// TIA Portal V20 export
// export: Created 2025-12-01T14:56:44.9442204Z, ExportSetting None, DisplayName Totally Integrated Automation Portal, DisplayVersion V20 Update 3, DisplayName TIA Portal Openness, DisplayVersion V20 Update 3, DisplayName TIA Portal Version Control Interface, DisplayVersion V20 Update 3, DisplayName STEP 7 Professional, DisplayVersion V20 Update 3, DisplayName STEP 7 Safety, DisplayVersion V20 Update 2, DisplayName WinCC Basic/Comfort/Advanced, DisplayVersion V20 Update 3, DisplayName WinCC Professional, DisplayVersion V20 Update 3, DisplayName WinCC Unified, DisplayVersion V20 Update 3
FUNCTION_BLOCK "FB261_M_FSS_Carga_V0"   // FB261, LAD
TITLE = FSS_Carga
{ S7_Optimized_Access := 'FALSE' }
AUTHOR : TE_FSS
FAMILY : FSS
NAME : 20160509
VERSION : 3.3
// stored: AutoNumber false, SetENOAutomatically false
   VAR_INPUT
      Mesa : UInt;   // Mesa de la FB
      Error_Tx : Bool;   // Error en el Tx
      EnTension : Bool;   // Existe Tension en la Mesa
      Termico_T1 : Bool;   // Proteccion del T1
      Termico_T2 : Bool;   // Proteccion del T2
      Termico_T3 : Bool;   // Proteccion del T3
      Termico_T4 : Bool;   // Proteccion del T4
      pHsMx_1 : Bool;   // pHs 1 de la Mesa
      pHsMx_2 : Bool;   // pHs 2 de la Mesa
      pHsMx_3 : Bool;   // pHs 3 de la Mesa
      pHsMx_4 : Bool;   // pHs 4 de la Mesa
      Avance_T1 : Bool;   // Avance del T1
      Avance_T2 : Bool;   // Avance del T2
      Avance_T3 : Bool;   // Avance del T3
      Avance_T4 : Bool;   // Avance del T4
      Termico_TR1 : Bool;   // Proteccion del TR1
      Termico_TR2 : Bool;   // Proteccion del TR1
      Avance_TR1 : Bool;   // Avance del TR1
      Avance_TR2 : Bool;   // Avance del TR2
      TR1_Arriba : Bool;   // TR1 >> Arriba
      TR1_Abajo : Bool;   // TR1 >> Abajo
      TR1_EnMovimiento : Bool;   // TR1 >> En Movimiento
      TR2_Arriba : Bool;   // TR2 >> Arriba
      TR2_Abajo : Bool;   // TR2 >> Abajo
      TR2_EnMovimiento : Bool;   // TR2 >> En Movimiento
      TP1_Arriba : Bool;   // TP1 >> Arriba
      TP1_Abajo : Bool;   // TP1 >> Abajo
      TP1_EnMovimiento : Bool;   // TP1 >> En Movimiento
      TP2_Arriba : Bool;   // TP2 >> Arriba
      TP2_Abajo : Bool;   // TP2 >> Abajo
      TP2_EnMovimiento : Bool;   // TP2 >> En Movimiento
      TPS1_Arriba : Bool;   // TPS1 >> Arriba
      TPS1_Abajo : Bool;   // TPS1 >> Abajo
      TPS1_EnMovimiento : Bool;   // TPS1 >> En Movimiento
      TPS3_Arriba : Bool;   // TPS2 >> Arriba
      TPS3_Abajo : Bool;   // TPS2 >> Abajo
      TPS3_EnMovimiento : Bool;   // TPS2 >> En Movimiento
      MAnt_DescargaAct : Bool;   // E2 >> Mesa Anterior DescargaAct
      AVTF_MAnt_Mx_BGrande : Bool;   // E2 >> Mesa Anterior AVTF - Grande
      AVTF_MAnt_Mx_BPequena : Bool;   // E2 >> Mesa Anterior AVTF - Pequeña
      P_Mens_MAnt_Mx : Bool;   // E2 >> Mesa Anterior P_Mens
      S1_Arrival : Bool;   // S1 a FSS >> Arrival
      S1_Rotative : Bool;   // S1 a FSS >> Rotative
      S1_Complete : Bool;   // S1 a FSS >> Complete
      S3_Arrival : Bool;   // S3 a FSS >> Arrival
      S3_Rotative : Bool;   // S3 a FSS >> Rotative
      S3_Complete : Bool;   // S3 a FSS >> Complete
      MAnt_MSig_DesCargaAct : Bool;   // Pasarela >> Descarga Act
      AVTF_MAnt_MSig_BGrande : Bool;   // Pasarela >> AVTF - Grande
      AVTF_MAnt_MSig_BPequena : Bool;   // Pasarela >> AVTF - Pequeña
      PTF_MAnt_MSig : Bool;   // Pasarela >> PTF
      FTF_MAnt_MSig : Bool;   // Pasarela >> FTF
      F_EnvMens_Mx : Bool;   // Fin de Envio de Mensaje
      OrdSal_S01 : Bool;   // Orden de Salida por S1
      OrdSal_S03 : Bool;   // Orden de Salida por S3
      V_CNT_pHsMx : Int := 1000;   // Valor de Presencia
      V_CNT_pHsMx_FTF : Int := 250;   // Valor para activar FTF. Nota: < = V_CNT_pHsMx.
      V_CNTSeg_pHsMx : Int := 2000;   // Valor de Seguriadad para Presencia
      V_CNT_ApHsMx : Int := 200;   // Valor de Ausencia
      V_CNTSeg_ApHsMx : Int := 2000;   // Valor de Seguriadad para Ausencia
      V_TOut_Tx_Mx : Int := 7000;   // TimeOut de Entrada por E2
      V_TOut_TR : Int := 3000;   // TimeOut de Transfer
      V_TOut_TP : Int := 3000;   // TimeOut de Tope
      V_TOut_Interlock : Int := 5000;   // TimeOut de Interlock con el FSS
      V_CNT_PerdidapHs : Int := 1000;   // CNT de Perdida de pHs
      V_CNT_PosicionarCarga : Int := 500;   // Valor de Posicionar la Carga despues de la Entrada
      V_CNT_PresenciaPasarela : Int := 500;   // Valor de Posiconado para Pasarela
      V_TIM_EstabilidadCarga : Time := T#100MS;   // Valor de Eastabilidad de Carga por DCC
   END_VAR
   VAR_OUTPUT
      P_EnvMens_PMx : Bool;   // Permiso de Enviar Mensaje de Presencia
      P_EnvMens_AMx : Bool;   // Permiso de Enviar Mensaje de Ausencia
      P_RecepOK_Mx : Bool;   // Recepcion OK
      PTF_MAnt_Mx : Bool;   // E2 >> Mesa Anterior PTF
      FTF_MAnt_Mx : Bool;   // E2 >> Mesa Anterior FTF
      PMAnt_MSig_DescagaAct : Bool;   // Pasarela >> Descarga Act
      PAVTF_MAnt_MSig_BPequena : Bool;   // Pasarela >> AVTF - Grande
      PAVTF_MAnt_MSig_BGrande : Bool;   // Pasarela >> AVTF - Pequeña
      PPTF_MAnt_MSig : Bool;   // Pasarela >> PTF
      PFTF_MAnt_MSig : Bool;   // Pasarela >> FTF
   END_VAR
   VAR
      Mx_ET00 : Bool;
      Mx_ET01 : Bool;
      Mx_ET02 : Bool;
      Mx_ET07_1PRE : Bool;
      Mx_ET07_1FIN : Bool;
      Mx_ET07_2PRE : Bool;
      Mx_ET07_2FIN : Bool;
      Mx_ET07_3PRE : Bool;
      Mx_ET07_3FIN : Bool;
      Mx_ET07_4PRE : Bool;
      Mx_ET07_4FIN : Bool;
      Mx_ET08 : Bool;
      Mx_ET09 : Bool;
      Mx_ET10 : Bool;
      Mx_ET11 : Bool;
      Mx_ET12 : Bool;
      Mx_ET110 : Bool;
      Mx_ET111 : Bool;
      Mx_ET13 : Bool;
      Mx_ET14 : Bool;
      Mx_ET15 : Bool;
      Mx_ET40 : Bool;
      Mx_ET41 : Bool;
      Mx_ET42 : Bool;
      Mx_ET50 : Bool;
      Mx_ET51 : Bool;
      Mx_ET150 : Bool;
      Mx_ET151 : Bool;
      Mx_ET152 : Bool;
      Mx_ET250 : Bool;
      Mx_ET251 : Bool;
      Mx_ET60 : Bool;
      Mx_ET61 : Bool;
      Mx_ET160 : Bool;
      Mx_ET161 : Bool;
      Mx_ET162 : Bool;
      Mx_ET260 : Bool;
      Mx_ET261 : Bool;
      Mx_ET90 : Bool;
      Mx_ET91 : Bool;
      Mx_ET92 : Bool;
      Mx_AutoArranque : Bool;   // Config >> Fin carga del FSS - Automatico
      FinCargaFSS_Auto : Bool;   // Intena >> AutoRearme Fin Carga del FSS
      Entrando_BGrande : Bool;   // Interna >> Bandeja Grande en Entrada
      Activado_Pasarela : Bool;   // Pasarela >> Activada
      Permiso_Pasarela : Bool;   // Pasarela >> Permiso de Movimiento
      S1_DesCargaAct : Bool;   // Interna >> DesCarga Activa de Salida por S1
      S3_DesCargaAct : Bool;   // Interna >> DesCarga Activa de Salida por S3
      Pos_TROK : Bool;   // Interna >> Posicion Correcta de los TRs
      Pos_TPOK : Bool;   // Interna >> Posicion Correcta de los TPs
      Select_S1 : Bool;   // Interna >> Selecionado Salida por S1
      Select_S3 : Bool;   // Interna >> Selecionado Salida por S3
      MemoriaPos_01 : Bool;   // Interna >> Memoria de Posicion Ocupada pHs_1
      MemoriaPos_02 : Bool;   // Interna >> Memoria de Posicion Ocupada pHs_2
      MemoriaPos_03 : Bool;   // Interna >> Memoria de Posicion Ocupada pHs_3
      MemoriaPos_04 : Bool;   // Interna >> Memoria de Posicion Ocupada pHs_4
      ProtocoloInciado : Bool;   // Iniciado el Envio del Mensaje de Presencia
      CNT_pHsMx_FTF_OK : Bool;   // Enviar ya FTF
      STAT_EnvMens_PMx : Bool;   // Interna >> Envio del Mensaje de Presencia
      STAT_EnvMens_AMx : Bool;   // Interna >> Envio de Mensaje de Ausencia
      STAT_AVTF_MAnt_Mx : Bool;   // Interna >> Aviso de Entrada
      STAT_FTF_MAnt_Mx : Bool;   // Interna >> FTF de MAnt >> Mx
      STAT_AvanceCarga : Bool;   // Interna >> Avance de Entrada de Carga
      STAT_AvanceDescarga : Bool;   // Interna >> Avance de Salida de Carga
      STAT_AvancePasarela : Bool;   // Interna >> Avance de Pasarela
      STAT_Velocidad_TxBO : Bool;   // Interna >> Velocidad Bit 0 de los Rodillos
      STAT_Velocidad_TxB1 : Bool;   // Interna >> Velocidad Bit 1 de los Rodillos
      MA_Avance_T1 : Bool;
      MA_Avance_T2 : Bool;
      MA_Avance_T3 : Bool;
      MA_Avance_T4 : Bool;
      MA_Inversion_Tx : Bool;
      MA_VelocidadAnalogica : Int;
      MA_Avance_TR1 : Bool;
      MA_Avance_TR2 : Bool;
      MA_VelocidaLenta_TRx : Bool;
      MA_Subir_TR1 : Bool;
      MA_Bajar_TR1 : Bool;
      MA_Subir_TR2 : Bool;
      MA_Bajar_TR2 : Bool;
      MA_Subir_TP1 : Bool;
      MA_Bajar_TP1 : Bool;
      MA_Subir_TP2 : Bool;
      MA_Bajar_TP2 : Bool;
      MA_Subir_TPS1 : Bool;
      MA_Bajar_TPS1 : Bool;
      MA_Subir_TPS3 : Bool;
      MA_Bajar_TPS3 : Bool;
      MA_PickUpOK_S1 : Bool;
      MA_PickUpOK_S3 : Bool;
      TIM_Estabilidad_Entrada { S7_SetPoint := 'True'} : TON_TIME;   // TIM De Estabilidad de Carga en la Entrada
      TIM_Estabilidad_S1 { S7_SetPoint := 'True'} : TON_TIME;   // TIM De Estabilidad de Carga en la Salida por S1
      TIM_Estabilidad_S3 { S7_SetPoint := 'True'} : TON_TIME;   // TIM De Estabilidad de Carga en la Salida por S3
      CNT_pHsMx { S7_SetPoint := 'True'} : "FB910_CNT_UHS";   // CNT de la Presencia
      CNTSeg_pHsMx { S7_SetPoint := 'True'} : "FB910_CNT_UHS";   // CNT de Seguridad de la Presencia
      CNT_ApHsMx { S7_SetPoint := 'True'} : "FB910_CNT_UHS";   // CNT de la Ausencia
      CNTSeg_ApHsMx { S7_SetPoint := 'True'} : "FB910_CNT_UHS";   // CNT de Seguridad de la Ausencia
      TMP_EnTension { S7_SetPoint := 'True'} : "FB910_CNT_UHS";
      TOut_Av_Tx { S7_SetPoint := 'True'} : "FB910_CNT_UHS";   // Time Out de Posicionado de la Carga
      TOut_Av_TRx { S7_SetPoint := 'True'} : "FB910_CNT_UHS";   // Time Out de Entrada de E2
      TOut_Subir_TR { S7_SetPoint := 'True'} : "FB910_CNT_UHS";   // Time Out de Subida del TR
      TOut_Bajar_TR { S7_SetPoint := 'True'} : "FB910_CNT_UHS";   // Time Out de Bajada del TR
      TOut_Subir_TP_E1E3 { S7_SetPoint := 'True'} : "FB910_CNT_UHS";   // Time Out de Subida del TP >> E1E3
      TOut_Bajar_TP_E1E3 { S7_SetPoint := 'True'} : "FB910_CNT_UHS";   // Time Out de Bajada del TP >> E1E3
      TOut_Subir_TP_E2E4 { S7_SetPoint := 'True'} : "FB910_CNT_UHS";   // Time Out de Subida del TP >> E2E4
      TOut_Bajar_TP_E2E4 { S7_SetPoint := 'True'} : "FB910_CNT_UHS";   // Time Out de Bajada del TP >> E2E4
      TOut_Interlock { S7_SetPoint := 'True'} : "FB910_CNT_UHS";   // Time Out de Interlock con el FSS
      CNT_PerdidapHs { S7_SetPoint := 'True'} : "FB910_CNT_UHS";   // CNT de Perdida de pHs
      CNT_PosicionarCarga { S7_SetPoint := 'True'} : "FB910_CNT_UHS";   // CNT Posicionar la Carga en la Mesa a la Entrada
      CNT_PrepararS1 { S7_SetPoint := 'True'} : "FB910_CNT_UHS";   // CNT Prepar la Carga en la Mesa en Salida S1
      CNT_PrepararS3 { S7_SetPoint := 'True'} : "FB910_CNT_UHS";   // CNT Prepar la Carga en la Mesa en Salida S3
      CNT_PresenciaPasarela { S7_SetPoint := 'True'} : "FB910_CNT_UHS";   // CNT Presencia de Carga en la Pasarela
      Interlock_manual { S7_SetPoint := 'True'} : "UDT_Interlock_manual_TE_FSS";
      Manual : "MoviManualMesa_FSS";
   END_VAR
   VAR_TEMP
      EstadoZona : "EstadoZona";   // Estado de Zona de la Mesa
      EstadoVI : "EstadosMesa_FSS";   // Estado del Vehiculo Inteliguente de la Mesa
      ConfigFB : "UDT_ConfigFB";   // Configuracion de la FB de la Mesa
      Interlock : "UDT_Interlock_TE_FSS";
      Aux_ET00 : Bool;
      cero : USInt;
      retval : Int;
   END_VAR
   VAR_TEMP   // added for the SCL form of the ladder/FBD networks
      _w1 : Bool;
   END_VAR
BEGIN

REGION Network 1: CONFIGURACION ESPECIAL DE LA FB
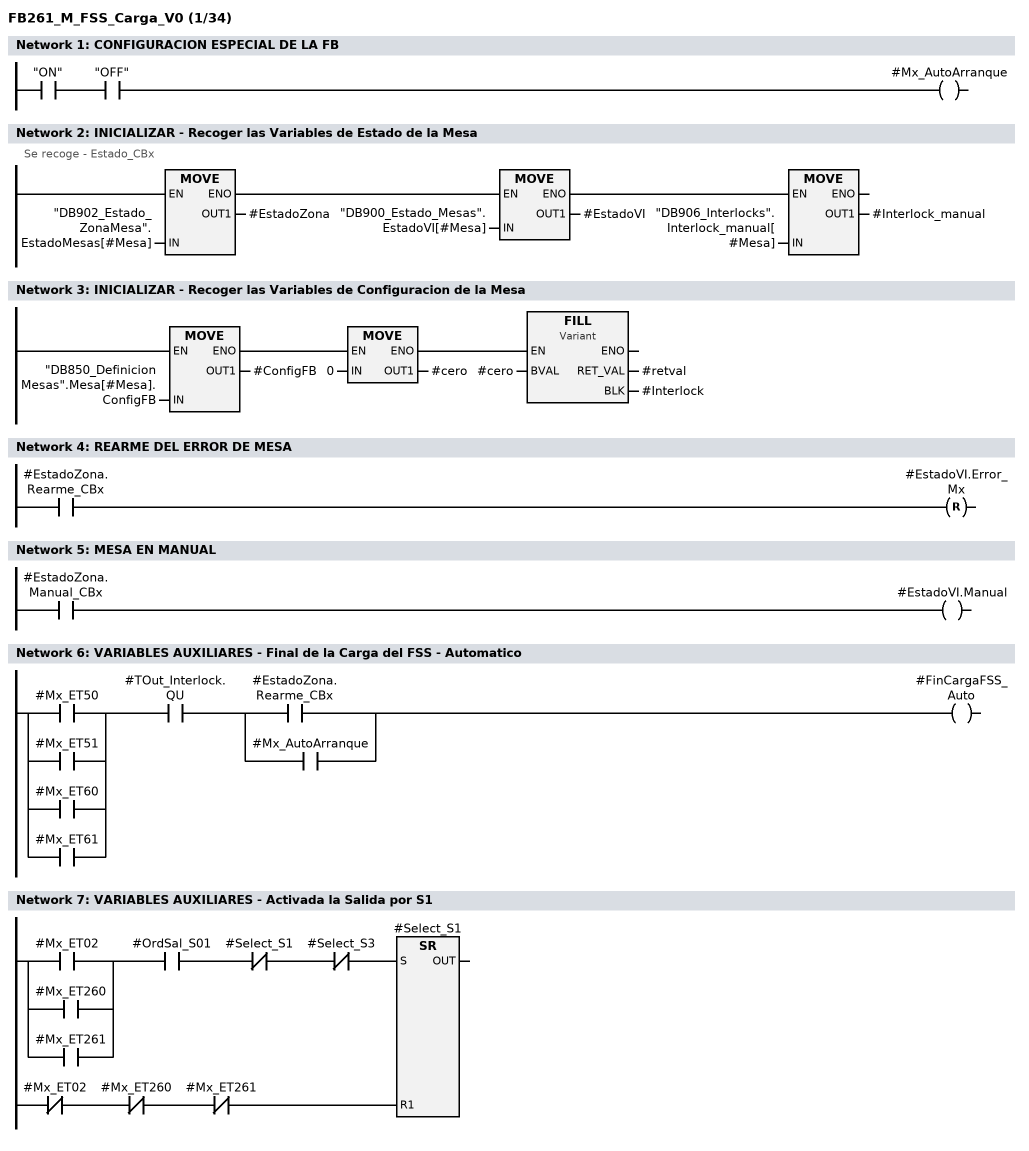
   RUNG wire#powerrail
      Contact( "ON" )
      Contact( "OFF" )
      Coil( #Mx_AutoArranque )
   END_RUNG
   // the same network as SCL:
   #Mx_AutoArranque := "ON" AND "OFF";
END_REGION

REGION Network 2: INICIALIZAR - Recoger las Variables de Estado de la Mesa
   // Se recoge - Estado_CBx
   RUNG wire#powerrail
      Move(in := "DB902_Estado_ZonaMesa".EstadoMesas[#Mesa], out1 => #EstadoZona)
      Move(in := "DB900_Estado_Mesas".EstadoVI[#Mesa], out1 => #EstadoVI)
      Move(in := "DB906_Interlocks".Interlock_manual[#Mesa], out1 => #Interlock_manual)
   END_RUNG
   // the same network as SCL:
   #EstadoZona := "DB902_Estado_ZonaMesa".EstadoMesas[#Mesa];
   #EstadoVI := "DB900_Estado_Mesas".EstadoVI[#Mesa];
   #Interlock_manual := "DB906_Interlocks".Interlock_manual[#Mesa];
END_REGION

REGION Network 3: INICIALIZAR - Recoger las Variables de Configuracion de la Mesa
   RUNG wire#powerrail
      Move(in := "DB850_DefinicionMesas".Mesa[#Mesa].ConfigFB, out1 => #ConfigFB)
      Move(in := 0, out1 => #cero)
      { S7_Templates := "ptr_type := Variant" } FILL(BVAL := #cero, RET_VAL => #retval, BLK => #Interlock)
   END_RUNG
   // the same network as SCL:
   #ConfigFB := "DB850_DefinicionMesas".Mesa[#Mesa].ConfigFB;
   #cero := 0;
   #retval := FILL(BVAL := #cero, BLK => #Interlock);
END_REGION

REGION Network 4: REARME DEL ERROR DE MESA
   RUNG wire#powerrail
      Contact( #EstadoZona.Rearme_CBx )
      R_Coil( #EstadoVI.Error_Mx )
   END_RUNG
   // the same network as SCL:
   IF #EstadoZona.Rearme_CBx THEN #EstadoVI.Error_Mx := FALSE; END_IF;
END_REGION

REGION Network 5: MESA EN MANUAL
   RUNG wire#powerrail
      Contact( #EstadoZona.Manual_CBx )
      Coil( #EstadoVI.Manual )
   END_RUNG
   // the same network as SCL:
   #EstadoVI.Manual := #EstadoZona.Manual_CBx;
END_REGION

REGION Network 6: VARIABLES AUXILIARES - Final de la Carga del FSS - Automatico
   RUNG wire#powerrail
      Contact( #Mx_ET50 )
      wire#w1
      Contact( #TOut_Interlock.QU )
      wire#w2
      Contact( #EstadoZona.Rearme_CBx )
      wire#w3
      Coil( #FinCargaFSS_Auto )
   END_RUNG
   RUNG wire#powerrail
      Contact( #Mx_ET51 )
   END_RUNG wire#w1
   RUNG wire#powerrail
      Contact( #Mx_ET60 )
   END_RUNG wire#w1
   RUNG wire#powerrail
      Contact( #Mx_ET61 )
   END_RUNG wire#w1
   RUNG wire#w2
      Contact( #Mx_AutoArranque )
   END_RUNG wire#w3
   // the same network as SCL:
   #FinCargaFSS_Auto := (#Mx_ET50 OR #Mx_ET51 OR #Mx_ET60 OR #Mx_ET61) AND #TOut_Interlock.QU AND (#EstadoZona.Rearme_CBx OR #Mx_AutoArranque);
END_REGION

REGION Network 7: VARIABLES AUXILIARES - Activada la Salida por S1
   RUNG wire#powerrail
      Contact( #Mx_ET02 )
      wire#w1
      Contact( #OrdSal_S01 )
      I_Contact( #Select_S1 )
      I_Contact( #Select_S3 )
      S_SR(operand := #Select_S1, r1 := wire#w2)
   END_RUNG
   RUNG wire#powerrail
      Contact( #Mx_ET260 )
   END_RUNG wire#w1
   RUNG wire#powerrail
      Contact( #Mx_ET261 )
   END_RUNG wire#w1
   RUNG wire#powerrail
      I_Contact( #Mx_ET02 )
      I_Contact( #Mx_ET260 )
      I_Contact( #Mx_ET261 )
   END_RUNG wire#w2
   // the same network as SCL:
   IF (#Mx_ET02 OR #Mx_ET260 OR #Mx_ET261) AND #OrdSal_S01 AND NOT #Select_S1 AND NOT #Select_S3 THEN
       #Select_S1 := TRUE;   // SR flip-flop
   END_IF;
   IF NOT #Mx_ET02 AND NOT #Mx_ET260 AND NOT #Mx_ET261 THEN #Select_S1 := FALSE; END_IF;
END_REGION

REGION Network 8: VARIABLES AUXILIARES - activada la Salida por S3
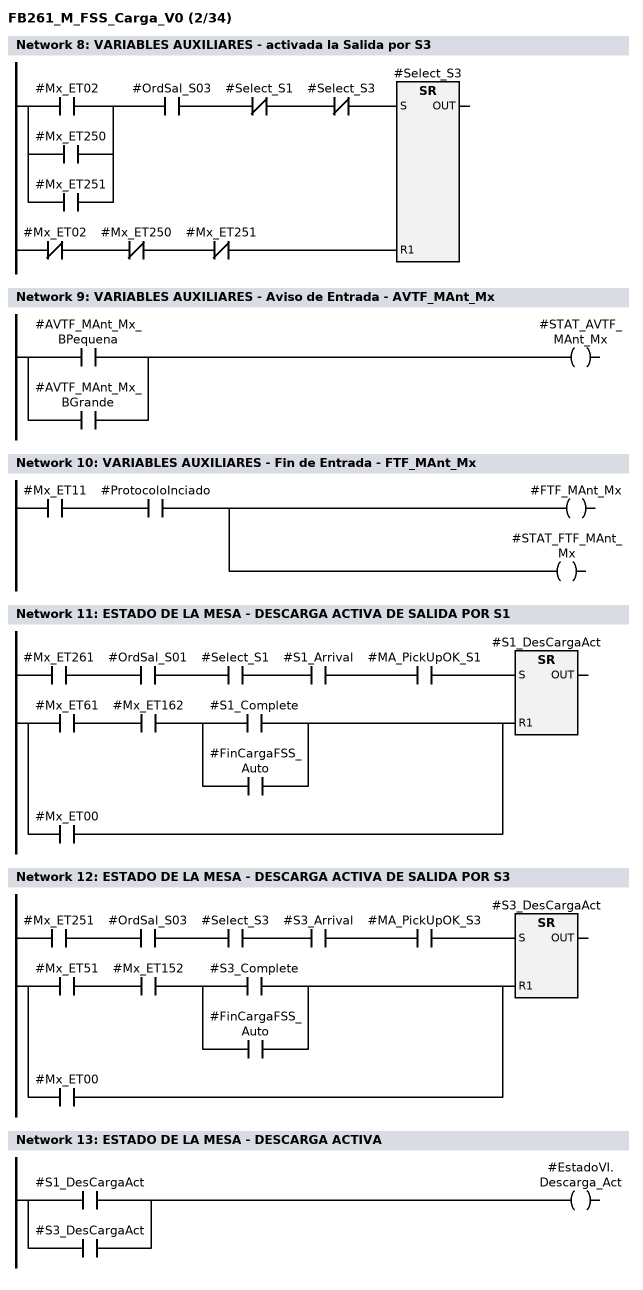
   RUNG wire#powerrail
      Contact( #Mx_ET02 )
      wire#w1
      Contact( #OrdSal_S03 )
      I_Contact( #Select_S1 )
      I_Contact( #Select_S3 )
      S_SR(operand := #Select_S3, r1 := wire#w2)
   END_RUNG
   RUNG wire#powerrail
      Contact( #Mx_ET250 )
   END_RUNG wire#w1
   RUNG wire#powerrail
      Contact( #Mx_ET251 )
   END_RUNG wire#w1
   RUNG wire#powerrail
      I_Contact( #Mx_ET02 )
      I_Contact( #Mx_ET250 )
      I_Contact( #Mx_ET251 )
   END_RUNG wire#w2
   // the same network as SCL:
   IF (#Mx_ET02 OR #Mx_ET250 OR #Mx_ET251) AND #OrdSal_S03 AND NOT #Select_S1 AND NOT #Select_S3 THEN
       #Select_S3 := TRUE;   // SR flip-flop
   END_IF;
   IF NOT #Mx_ET02 AND NOT #Mx_ET250 AND NOT #Mx_ET251 THEN #Select_S3 := FALSE; END_IF;
END_REGION

REGION Network 9: VARIABLES AUXILIARES - Aviso de Entrada - AVTF_MAnt_Mx
   RUNG wire#powerrail
      Contact( #AVTF_MAnt_Mx_BPequena )
      wire#w1
      Coil( #STAT_AVTF_MAnt_Mx )
   END_RUNG
   RUNG wire#powerrail
      Contact( #AVTF_MAnt_Mx_BGrande )
   END_RUNG wire#w1
   // the same network as SCL:
   #STAT_AVTF_MAnt_Mx := #AVTF_MAnt_Mx_BPequena OR #AVTF_MAnt_Mx_BGrande;
END_REGION

REGION Network 10: VARIABLES AUXILIARES - Fin de Entrada - FTF_MAnt_Mx
   RUNG wire#powerrail
      Contact( #Mx_ET11 )
      Contact( #ProtocoloInciado )
      wire#w1
      Coil( #FTF_MAnt_Mx )
   END_RUNG
   RUNG wire#w1
      Coil( #STAT_FTF_MAnt_Mx )
   END_RUNG
   // the same network as SCL:
   #FTF_MAnt_Mx := #Mx_ET11 AND #ProtocoloInciado;
   #STAT_FTF_MAnt_Mx := #FTF_MAnt_Mx;
END_REGION

REGION Network 11: ESTADO DE LA MESA - DESCARGA ACTIVA DE SALIDA POR S1
   RUNG wire#powerrail
      Contact( #Mx_ET261 )
      Contact( #OrdSal_S01 )
      Contact( #Select_S1 )
      Contact( #S1_Arrival )
      Contact( #MA_PickUpOK_S1 )
      S_SR(operand := #S1_DesCargaAct, r1 := wire#w2)
   END_RUNG
   RUNG wire#powerrail
      Contact( #Mx_ET61 )
      Contact( #Mx_ET162 )
      wire#w1
      Contact( #S1_Complete )
   END_RUNG wire#w2
   RUNG wire#w1
      Contact( #FinCargaFSS_Auto )
   END_RUNG wire#w2
   RUNG wire#powerrail
      Contact( #Mx_ET00 )
   END_RUNG wire#w2
   // the same network as SCL:
   IF #Mx_ET261 AND #OrdSal_S01 AND #Select_S1 AND #S1_Arrival AND #MA_PickUpOK_S1 THEN
       #S1_DesCargaAct := TRUE;   // SR flip-flop
   END_IF;
   IF (#Mx_ET61 AND #Mx_ET162 AND (#S1_Complete OR #FinCargaFSS_Auto)) OR #Mx_ET00 THEN
       #S1_DesCargaAct := FALSE;
   END_IF;
END_REGION

REGION Network 12: ESTADO DE LA MESA - DESCARGA ACTIVA DE SALIDA POR S3
   RUNG wire#powerrail
      Contact( #Mx_ET251 )
      Contact( #OrdSal_S03 )
      Contact( #Select_S3 )
      Contact( #S3_Arrival )
      Contact( #MA_PickUpOK_S3 )
      S_SR(operand := #S3_DesCargaAct, r1 := wire#w2)
   END_RUNG
   RUNG wire#powerrail
      Contact( #Mx_ET51 )
      Contact( #Mx_ET152 )
      wire#w1
      Contact( #S3_Complete )
   END_RUNG wire#w2
   RUNG wire#w1
      Contact( #FinCargaFSS_Auto )
   END_RUNG wire#w2
   RUNG wire#powerrail
      Contact( #Mx_ET00 )
   END_RUNG wire#w2
   // the same network as SCL:
   IF #Mx_ET251 AND #OrdSal_S03 AND #Select_S3 AND #S3_Arrival AND #MA_PickUpOK_S3 THEN
       #S3_DesCargaAct := TRUE;   // SR flip-flop
   END_IF;
   IF (#Mx_ET51 AND #Mx_ET152 AND (#S3_Complete OR #FinCargaFSS_Auto)) OR #Mx_ET00 THEN
       #S3_DesCargaAct := FALSE;
   END_IF;
END_REGION

REGION Network 13: ESTADO DE LA MESA - DESCARGA ACTIVA
   RUNG wire#powerrail
      Contact( #S1_DesCargaAct )
      wire#w1
      Coil( #EstadoVI.Descarga_Act )
   END_RUNG
   RUNG wire#powerrail
      Contact( #S3_DesCargaAct )
   END_RUNG wire#w1
   // the same network as SCL:
   #EstadoVI.Descarga_Act := #S1_DesCargaAct OR #S3_DesCargaAct;
END_REGION

REGION Network 14: ET92 - ACTIVACION DE PASARELA - OCUPADA LA MESA
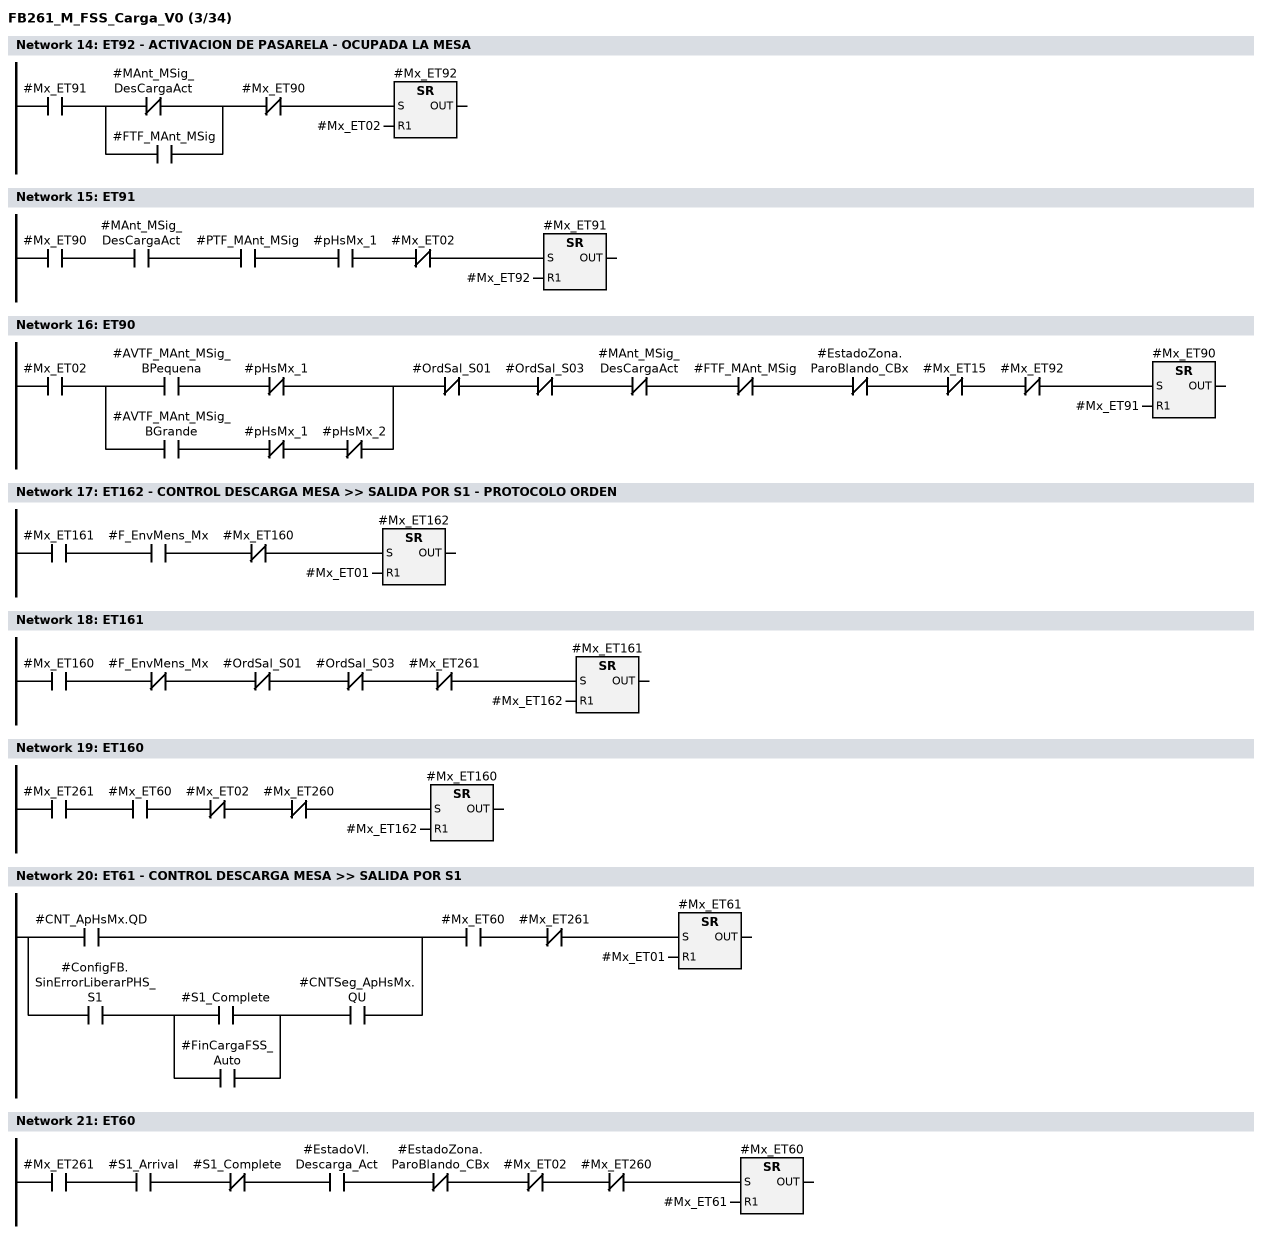
   RUNG wire#powerrail
      Contact( #Mx_ET91 )
      wire#w1
      I_Contact( #MAnt_MSig_DesCargaAct )
      wire#w2
      I_Contact( #Mx_ET90 )
      S_SR(operand := #Mx_ET92, r1 := #Mx_ET02)
   END_RUNG
   RUNG wire#w1
      Contact( #FTF_MAnt_MSig )
   END_RUNG wire#w2
   // the same network as SCL:
   IF #Mx_ET91 AND (NOT #MAnt_MSig_DesCargaAct OR #FTF_MAnt_MSig) AND NOT #Mx_ET90 THEN
       #Mx_ET92 := TRUE;   // SR flip-flop
   END_IF;
   IF #Mx_ET02 THEN #Mx_ET92 := FALSE; END_IF;
END_REGION

REGION Network 15: ET91
   RUNG wire#powerrail
      Contact( #Mx_ET90 )
      Contact( #MAnt_MSig_DesCargaAct )
      Contact( #PTF_MAnt_MSig )
      Contact( #pHsMx_1 )
      I_Contact( #Mx_ET02 )
      S_SR(operand := #Mx_ET91, r1 := #Mx_ET92)
   END_RUNG
   // the same network as SCL:
   IF #Mx_ET90 AND #MAnt_MSig_DesCargaAct AND #PTF_MAnt_MSig AND #pHsMx_1 AND NOT #Mx_ET02 THEN
       #Mx_ET91 := TRUE;   // SR flip-flop
   END_IF;
   IF #Mx_ET92 THEN #Mx_ET91 := FALSE; END_IF;
END_REGION

REGION Network 16: ET90
   RUNG wire#powerrail
      Contact( #Mx_ET02 )
      wire#w1
      Contact( #AVTF_MAnt_MSig_BPequena )
      I_Contact( #pHsMx_1 )
      wire#w2
      I_Contact( #OrdSal_S01 )
      I_Contact( #OrdSal_S03 )
      I_Contact( #MAnt_MSig_DesCargaAct )
      I_Contact( #FTF_MAnt_MSig )
      I_Contact( #EstadoZona.ParoBlando_CBx )
      I_Contact( #Mx_ET15 )
      I_Contact( #Mx_ET92 )
      S_SR(operand := #Mx_ET90, r1 := #Mx_ET91)
   END_RUNG
   RUNG wire#w1
      Contact( #AVTF_MAnt_MSig_BGrande )
      I_Contact( #pHsMx_1 )
      I_Contact( #pHsMx_2 )
   END_RUNG wire#w2
   // the same network as SCL:
   IF #Mx_ET02 AND ((#AVTF_MAnt_MSig_BPequena AND NOT #pHsMx_1) OR (#AVTF_MAnt_MSig_BGrande AND NOT #pHsMx_1 AND NOT #pHsMx_2)) AND NOT #OrdSal_S01 AND NOT #OrdSal_S03 AND NOT #MAnt_MSig_DesCargaAct AND NOT #FTF_MAnt_MSig AND NOT #EstadoZona.ParoBlando_CBx AND NOT #Mx_ET15 AND NOT #Mx_ET92 THEN
       #Mx_ET90 := TRUE;   // SR flip-flop
   END_IF;
   IF #Mx_ET91 THEN #Mx_ET90 := FALSE; END_IF;
END_REGION

REGION Network 17: ET162 - CONTROL DESCARGA MESA >> SALIDA POR S1 - PROTOCOLO ORDEN
   RUNG wire#powerrail
      Contact( #Mx_ET161 )
      Contact( #F_EnvMens_Mx )
      I_Contact( #Mx_ET160 )
      S_SR(operand := #Mx_ET162, r1 := #Mx_ET01)
   END_RUNG
   // the same network as SCL:
   IF #Mx_ET161 AND #F_EnvMens_Mx AND NOT #Mx_ET160 THEN
       #Mx_ET162 := TRUE;   // SR flip-flop
   END_IF;
   IF #Mx_ET01 THEN #Mx_ET162 := FALSE; END_IF;
END_REGION

REGION Network 18: ET161
   RUNG wire#powerrail
      Contact( #Mx_ET160 )
      I_Contact( #F_EnvMens_Mx )
      I_Contact( #OrdSal_S01 )
      I_Contact( #OrdSal_S03 )
      I_Contact( #Mx_ET261 )
      S_SR(operand := #Mx_ET161, r1 := #Mx_ET162)
   END_RUNG
   // the same network as SCL:
   IF #Mx_ET160 AND NOT #F_EnvMens_Mx AND NOT #OrdSal_S01 AND NOT #OrdSal_S03 AND NOT #Mx_ET261 THEN
       #Mx_ET161 := TRUE;   // SR flip-flop
   END_IF;
   IF #Mx_ET162 THEN #Mx_ET161 := FALSE; END_IF;
END_REGION

REGION Network 19: ET160
   RUNG wire#powerrail
      Contact( #Mx_ET261 )
      Contact( #Mx_ET60 )
      I_Contact( #Mx_ET02 )
      I_Contact( #Mx_ET260 )
      S_SR(operand := #Mx_ET160, r1 := #Mx_ET162)
   END_RUNG
   // the same network as SCL:
   IF #Mx_ET261 AND #Mx_ET60 AND NOT #Mx_ET02 AND NOT #Mx_ET260 THEN
       #Mx_ET160 := TRUE;   // SR flip-flop
   END_IF;
   IF #Mx_ET162 THEN #Mx_ET160 := FALSE; END_IF;
END_REGION

REGION Network 20: ET61 - CONTROL DESCARGA MESA >> SALIDA POR S1
   RUNG wire#powerrail
      Contact( #CNT_ApHsMx.QD )
      wire#w1
      Contact( #Mx_ET60 )
      I_Contact( #Mx_ET261 )
      S_SR(operand := #Mx_ET61, r1 := #Mx_ET01)
   END_RUNG
   RUNG wire#powerrail
      Contact( #ConfigFB.SinErrorLiberarPHS_S1 )
      wire#w2
      Contact( #S1_Complete )
      wire#w3
      Contact( #CNTSeg_ApHsMx.QU )
   END_RUNG wire#w1
   RUNG wire#w2
      Contact( #FinCargaFSS_Auto )
   END_RUNG wire#w3
   // the same network as SCL:
   IF (#CNT_ApHsMx.QD OR (#ConfigFB.SinErrorLiberarPHS_S1 AND (#S1_Complete OR #FinCargaFSS_Auto) AND #CNTSeg_ApHsMx.QU)) AND #Mx_ET60 AND NOT #Mx_ET261 THEN
       #Mx_ET61 := TRUE;   // SR flip-flop
   END_IF;
   IF #Mx_ET01 THEN #Mx_ET61 := FALSE; END_IF;
END_REGION

REGION Network 21: ET60
   RUNG wire#powerrail
      Contact( #Mx_ET261 )
      Contact( #S1_Arrival )
      I_Contact( #S1_Complete )
      Contact( #EstadoVI.Descarga_Act )
      I_Contact( #EstadoZona.ParoBlando_CBx )
      I_Contact( #Mx_ET02 )
      I_Contact( #Mx_ET260 )
      S_SR(operand := #Mx_ET60, r1 := #Mx_ET61)
   END_RUNG
   // the same network as SCL:
   IF #Mx_ET261 AND #S1_Arrival AND NOT #S1_Complete AND #EstadoVI.Descarga_Act AND NOT #EstadoZona.ParoBlando_CBx AND NOT #Mx_ET02 AND NOT #Mx_ET260 THEN
       #Mx_ET60 := TRUE;   // SR flip-flop
   END_IF;
   IF #Mx_ET61 THEN #Mx_ET60 := FALSE; END_IF;
END_REGION

REGION Network 22: ET261 - POSICIONAMIENTO PREVIO PARA LA DESCARGA MESA >> SALIDA POR S1
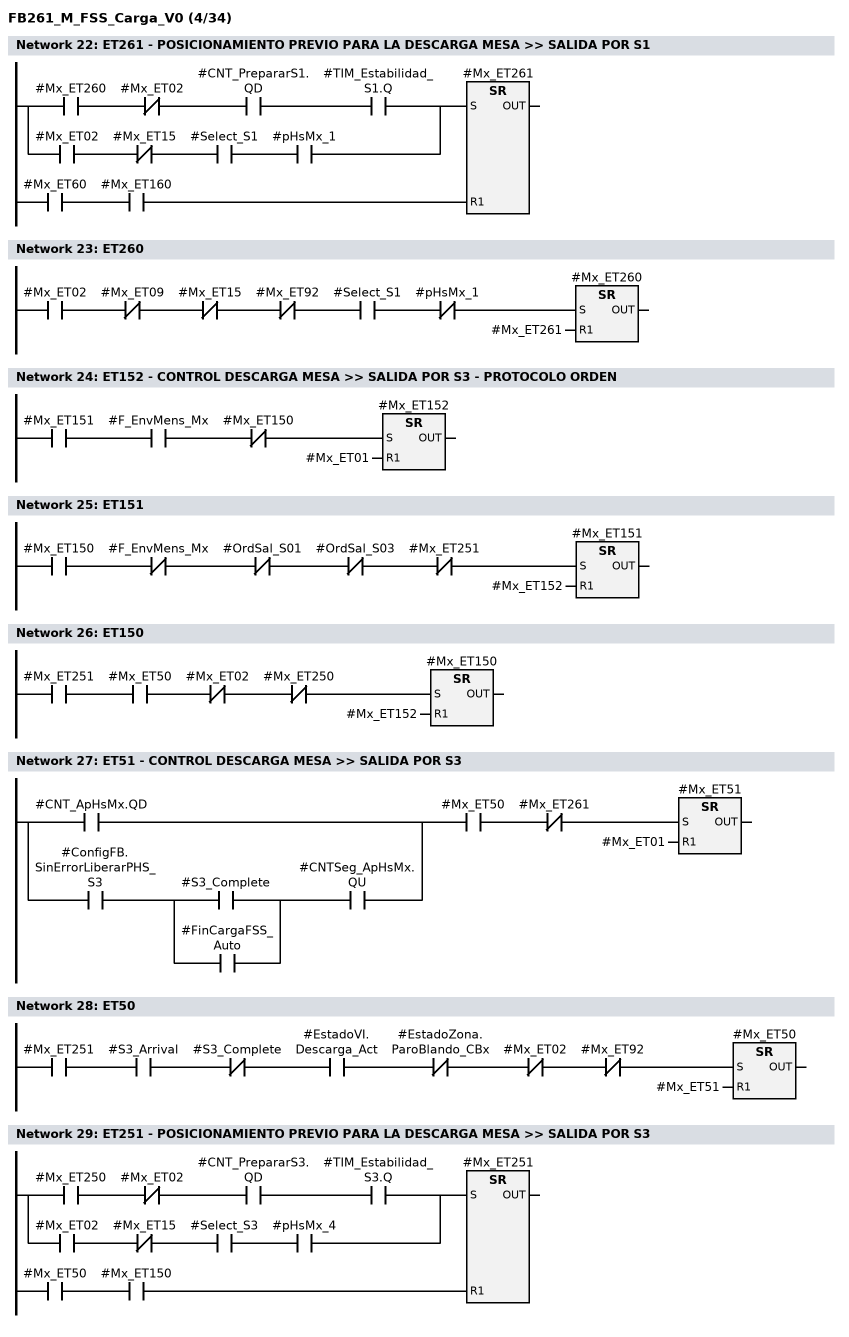
   RUNG wire#powerrail
      Contact( #Mx_ET260 )
      I_Contact( #Mx_ET02 )
      Contact( #CNT_PrepararS1.QD )
      Contact( #TIM_Estabilidad_S1.Q )
      wire#w1
      S_SR(operand := #Mx_ET261, r1 := wire#w2)
   END_RUNG
   RUNG wire#powerrail
      Contact( #Mx_ET02 )
      I_Contact( #Mx_ET15 )
      Contact( #Select_S1 )
      Contact( #pHsMx_1 )
   END_RUNG wire#w1
   RUNG wire#powerrail
      Contact( #Mx_ET60 )
      Contact( #Mx_ET160 )
   END_RUNG wire#w2
   // the same network as SCL:
   IF (#Mx_ET260 AND NOT #Mx_ET02 AND #CNT_PrepararS1.QD AND #TIM_Estabilidad_S1.Q) OR (#Mx_ET02 AND NOT #Mx_ET15 AND #Select_S1 AND #pHsMx_1) THEN
       #Mx_ET261 := TRUE;   // SR flip-flop
   END_IF;
   IF #Mx_ET60 AND #Mx_ET160 THEN #Mx_ET261 := FALSE; END_IF;
END_REGION

REGION Network 23: ET260
   RUNG wire#powerrail
      Contact( #Mx_ET02 )
      I_Contact( #Mx_ET09 )
      I_Contact( #Mx_ET15 )
      I_Contact( #Mx_ET92 )
      Contact( #Select_S1 )
      I_Contact( #pHsMx_1 )
      S_SR(operand := #Mx_ET260, r1 := #Mx_ET261)
   END_RUNG
   // the same network as SCL:
   IF #Mx_ET02 AND NOT #Mx_ET09 AND NOT #Mx_ET15 AND NOT #Mx_ET92 AND #Select_S1 AND NOT #pHsMx_1 THEN
       #Mx_ET260 := TRUE;   // SR flip-flop
   END_IF;
   IF #Mx_ET261 THEN #Mx_ET260 := FALSE; END_IF;
END_REGION

REGION Network 24: ET152 - CONTROL DESCARGA MESA >> SALIDA POR S3 - PROTOCOLO ORDEN
   RUNG wire#powerrail
      Contact( #Mx_ET151 )
      Contact( #F_EnvMens_Mx )
      I_Contact( #Mx_ET150 )
      S_SR(operand := #Mx_ET152, r1 := #Mx_ET01)
   END_RUNG
   // the same network as SCL:
   IF #Mx_ET151 AND #F_EnvMens_Mx AND NOT #Mx_ET150 THEN
       #Mx_ET152 := TRUE;   // SR flip-flop
   END_IF;
   IF #Mx_ET01 THEN #Mx_ET152 := FALSE; END_IF;
END_REGION

REGION Network 25: ET151
   RUNG wire#powerrail
      Contact( #Mx_ET150 )
      I_Contact( #F_EnvMens_Mx )
      I_Contact( #OrdSal_S01 )
      I_Contact( #OrdSal_S03 )
      I_Contact( #Mx_ET251 )
      S_SR(operand := #Mx_ET151, r1 := #Mx_ET152)
   END_RUNG
   // the same network as SCL:
   IF #Mx_ET150 AND NOT #F_EnvMens_Mx AND NOT #OrdSal_S01 AND NOT #OrdSal_S03 AND NOT #Mx_ET251 THEN
       #Mx_ET151 := TRUE;   // SR flip-flop
   END_IF;
   IF #Mx_ET152 THEN #Mx_ET151 := FALSE; END_IF;
END_REGION

REGION Network 26: ET150
   RUNG wire#powerrail
      Contact( #Mx_ET251 )
      Contact( #Mx_ET50 )
      I_Contact( #Mx_ET02 )
      I_Contact( #Mx_ET250 )
      S_SR(operand := #Mx_ET150, r1 := #Mx_ET152)
   END_RUNG
   // the same network as SCL:
   IF #Mx_ET251 AND #Mx_ET50 AND NOT #Mx_ET02 AND NOT #Mx_ET250 THEN
       #Mx_ET150 := TRUE;   // SR flip-flop
   END_IF;
   IF #Mx_ET152 THEN #Mx_ET150 := FALSE; END_IF;
END_REGION

REGION Network 27: ET51 - CONTROL DESCARGA MESA >> SALIDA POR S3
   RUNG wire#powerrail
      Contact( #CNT_ApHsMx.QD )
      wire#w1
      Contact( #Mx_ET50 )
      I_Contact( #Mx_ET261 )
      S_SR(operand := #Mx_ET51, r1 := #Mx_ET01)
   END_RUNG
   RUNG wire#powerrail
      Contact( #ConfigFB.SinErrorLiberarPHS_S3 )
      wire#w2
      Contact( #S3_Complete )
      wire#w3
      Contact( #CNTSeg_ApHsMx.QU )
   END_RUNG wire#w1
   RUNG wire#w2
      Contact( #FinCargaFSS_Auto )
   END_RUNG wire#w3
   // the same network as SCL:
   IF (#CNT_ApHsMx.QD OR (#ConfigFB.SinErrorLiberarPHS_S3 AND (#S3_Complete OR #FinCargaFSS_Auto) AND #CNTSeg_ApHsMx.QU)) AND #Mx_ET50 AND NOT #Mx_ET261 THEN
       #Mx_ET51 := TRUE;   // SR flip-flop
   END_IF;
   IF #Mx_ET01 THEN #Mx_ET51 := FALSE; END_IF;
END_REGION

REGION Network 28: ET50
   RUNG wire#powerrail
      Contact( #Mx_ET251 )
      Contact( #S3_Arrival )
      I_Contact( #S3_Complete )
      Contact( #EstadoVI.Descarga_Act )
      I_Contact( #EstadoZona.ParoBlando_CBx )
      I_Contact( #Mx_ET02 )
      I_Contact( #Mx_ET92 )
      S_SR(operand := #Mx_ET50, r1 := #Mx_ET51)
   END_RUNG
   // the same network as SCL:
   IF #Mx_ET251 AND #S3_Arrival AND NOT #S3_Complete AND #EstadoVI.Descarga_Act AND NOT #EstadoZona.ParoBlando_CBx AND NOT #Mx_ET02 AND NOT #Mx_ET92 THEN
       #Mx_ET50 := TRUE;   // SR flip-flop
   END_IF;
   IF #Mx_ET51 THEN #Mx_ET50 := FALSE; END_IF;
END_REGION

REGION Network 29: ET251 - POSICIONAMIENTO PREVIO PARA LA DESCARGA MESA >> SALIDA POR S3
   RUNG wire#powerrail
      Contact( #Mx_ET250 )
      I_Contact( #Mx_ET02 )
      Contact( #CNT_PrepararS3.QD )
      Contact( #TIM_Estabilidad_S3.Q )
      wire#w1
      S_SR(operand := #Mx_ET251, r1 := wire#w2)
   END_RUNG
   RUNG wire#powerrail
      Contact( #Mx_ET02 )
      I_Contact( #Mx_ET15 )
      Contact( #Select_S3 )
      Contact( #pHsMx_4 )
   END_RUNG wire#w1
   RUNG wire#powerrail
      Contact( #Mx_ET50 )
      Contact( #Mx_ET150 )
   END_RUNG wire#w2
   // the same network as SCL:
   IF (#Mx_ET250 AND NOT #Mx_ET02 AND #CNT_PrepararS3.QD AND #TIM_Estabilidad_S3.Q) OR (#Mx_ET02 AND NOT #Mx_ET15 AND #Select_S3 AND #pHsMx_4) THEN
       #Mx_ET251 := TRUE;   // SR flip-flop
   END_IF;
   IF #Mx_ET50 AND #Mx_ET150 THEN #Mx_ET251 := FALSE; END_IF;
END_REGION

REGION Network 30: ET250
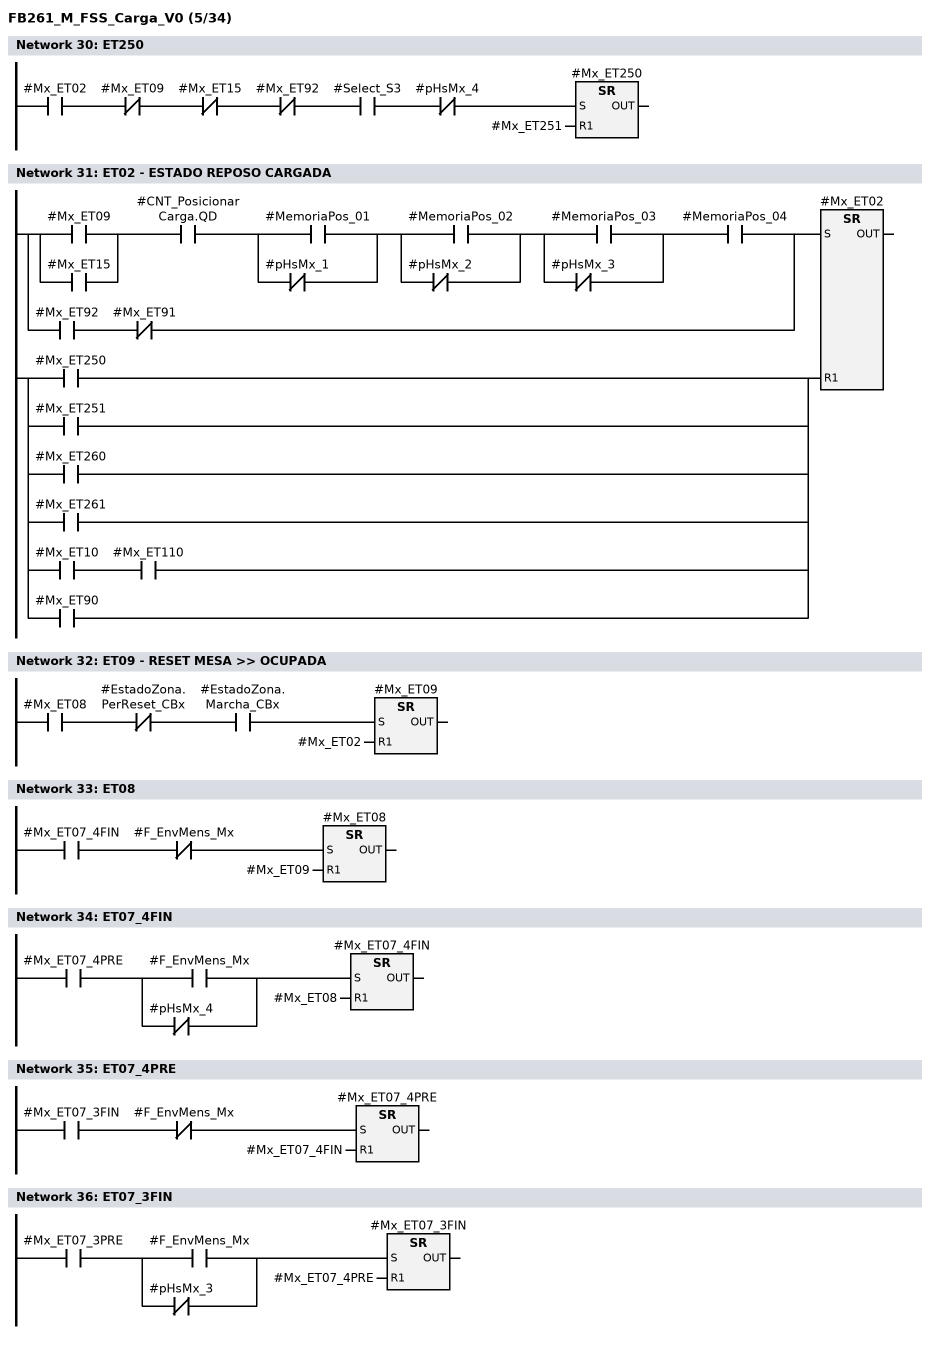
   RUNG wire#powerrail
      Contact( #Mx_ET02 )
      I_Contact( #Mx_ET09 )
      I_Contact( #Mx_ET15 )
      I_Contact( #Mx_ET92 )
      Contact( #Select_S3 )
      I_Contact( #pHsMx_4 )
      S_SR(operand := #Mx_ET250, r1 := #Mx_ET251)
   END_RUNG
   // the same network as SCL:
   IF #Mx_ET02 AND NOT #Mx_ET09 AND NOT #Mx_ET15 AND NOT #Mx_ET92 AND #Select_S3 AND NOT #pHsMx_4 THEN
       #Mx_ET250 := TRUE;   // SR flip-flop
   END_IF;
   IF #Mx_ET251 THEN #Mx_ET250 := FALSE; END_IF;
END_REGION

REGION Network 31: ET02 - ESTADO REPOSO CARGADA
   RUNG wire#powerrail
      Contact( #Mx_ET09 )
      wire#w1
      Contact( #CNT_PosicionarCarga.QD )
      wire#w2
      Contact( #MemoriaPos_01 )
      wire#w3
      Contact( #MemoriaPos_02 )
      wire#w4
      Contact( #MemoriaPos_03 )
      wire#w5
      Contact( #MemoriaPos_04 )
      wire#w6
      S_SR(operand := #Mx_ET02, r1 := wire#w7)
   END_RUNG
   RUNG wire#powerrail
      Contact( #Mx_ET15 )
   END_RUNG wire#w1
   RUNG wire#w2
      I_Contact( #pHsMx_1 )
   END_RUNG wire#w3
   RUNG wire#w3
      I_Contact( #pHsMx_2 )
   END_RUNG wire#w4
   RUNG wire#w4
      I_Contact( #pHsMx_3 )
   END_RUNG wire#w5
   RUNG wire#powerrail
      Contact( #Mx_ET92 )
      I_Contact( #Mx_ET91 )
   END_RUNG wire#w6
   RUNG wire#powerrail
      Contact( #Mx_ET250 )
   END_RUNG wire#w7
   RUNG wire#powerrail
      Contact( #Mx_ET251 )
   END_RUNG wire#w7
   RUNG wire#powerrail
      Contact( #Mx_ET260 )
   END_RUNG wire#w7
   RUNG wire#powerrail
      Contact( #Mx_ET261 )
   END_RUNG wire#w7
   RUNG wire#powerrail
      Contact( #Mx_ET10 )
      Contact( #Mx_ET110 )
   END_RUNG wire#w7
   RUNG wire#powerrail
      Contact( #Mx_ET90 )
   END_RUNG wire#w7
   // the same network as SCL:
   IF ((#Mx_ET09 OR #Mx_ET15) AND #CNT_PosicionarCarga.QD AND (#MemoriaPos_01 OR NOT #pHsMx_1) AND (#MemoriaPos_02 OR NOT #pHsMx_2) AND (#MemoriaPos_03 OR NOT #pHsMx_3) AND #MemoriaPos_04) OR (#Mx_ET92 AND NOT #Mx_ET91) THEN
       #Mx_ET02 := TRUE;   // SR flip-flop
   END_IF;
   IF #Mx_ET250 OR #Mx_ET251 OR #Mx_ET260 OR #Mx_ET261 OR (#Mx_ET10 AND #Mx_ET110) OR #Mx_ET90 THEN
       #Mx_ET02 := FALSE;
   END_IF;
END_REGION

REGION Network 32: ET09 - RESET MESA >> OCUPADA
   RUNG wire#powerrail
      Contact( #Mx_ET08 )
      I_Contact( #EstadoZona.PerReset_CBx )
      Contact( #EstadoZona.Marcha_CBx )
      S_SR(operand := #Mx_ET09, r1 := #Mx_ET02)
   END_RUNG
   // the same network as SCL:
   IF #Mx_ET08 AND NOT #EstadoZona.PerReset_CBx AND #EstadoZona.Marcha_CBx THEN
       #Mx_ET09 := TRUE;   // SR flip-flop
   END_IF;
   IF #Mx_ET02 THEN #Mx_ET09 := FALSE; END_IF;
END_REGION

REGION Network 33: ET08
   RUNG wire#powerrail
      Contact( #Mx_ET07_4FIN )
      I_Contact( #F_EnvMens_Mx )
      S_SR(operand := #Mx_ET08, r1 := #Mx_ET09)
   END_RUNG
   // the same network as SCL:
   IF #Mx_ET07_4FIN AND NOT #F_EnvMens_Mx THEN
       #Mx_ET08 := TRUE;   // SR flip-flop
   END_IF;
   IF #Mx_ET09 THEN #Mx_ET08 := FALSE; END_IF;
END_REGION

REGION Network 34: ET07_4FIN
   RUNG wire#powerrail
      Contact( #Mx_ET07_4PRE )
      wire#w1
      Contact( #F_EnvMens_Mx )
      wire#w2
      S_SR(operand := #Mx_ET07_4FIN, r1 := #Mx_ET08)
   END_RUNG
   RUNG wire#w1
      I_Contact( #pHsMx_4 )
   END_RUNG wire#w2
   // the same network as SCL:
   IF #Mx_ET07_4PRE AND (#F_EnvMens_Mx OR NOT #pHsMx_4) THEN
       #Mx_ET07_4FIN := TRUE;   // SR flip-flop
   END_IF;
   IF #Mx_ET08 THEN #Mx_ET07_4FIN := FALSE; END_IF;
END_REGION

REGION Network 35: ET07_4PRE
   RUNG wire#powerrail
      Contact( #Mx_ET07_3FIN )
      I_Contact( #F_EnvMens_Mx )
      S_SR(operand := #Mx_ET07_4PRE, r1 := #Mx_ET07_4FIN)
   END_RUNG
   // the same network as SCL:
   IF #Mx_ET07_3FIN AND NOT #F_EnvMens_Mx THEN
       #Mx_ET07_4PRE := TRUE;   // SR flip-flop
   END_IF;
   IF #Mx_ET07_4FIN THEN #Mx_ET07_4PRE := FALSE; END_IF;
END_REGION

REGION Network 36: ET07_3FIN
   RUNG wire#powerrail
      Contact( #Mx_ET07_3PRE )
      wire#w1
      Contact( #F_EnvMens_Mx )
      wire#w2
      S_SR(operand := #Mx_ET07_3FIN, r1 := #Mx_ET07_4PRE)
   END_RUNG
   RUNG wire#w1
      I_Contact( #pHsMx_3 )
   END_RUNG wire#w2
   // the same network as SCL:
   IF #Mx_ET07_3PRE AND (#F_EnvMens_Mx OR NOT #pHsMx_3) THEN
       #Mx_ET07_3FIN := TRUE;   // SR flip-flop
   END_IF;
   IF #Mx_ET07_4PRE THEN #Mx_ET07_3FIN := FALSE; END_IF;
END_REGION

REGION Network 37: ET07_3PRE
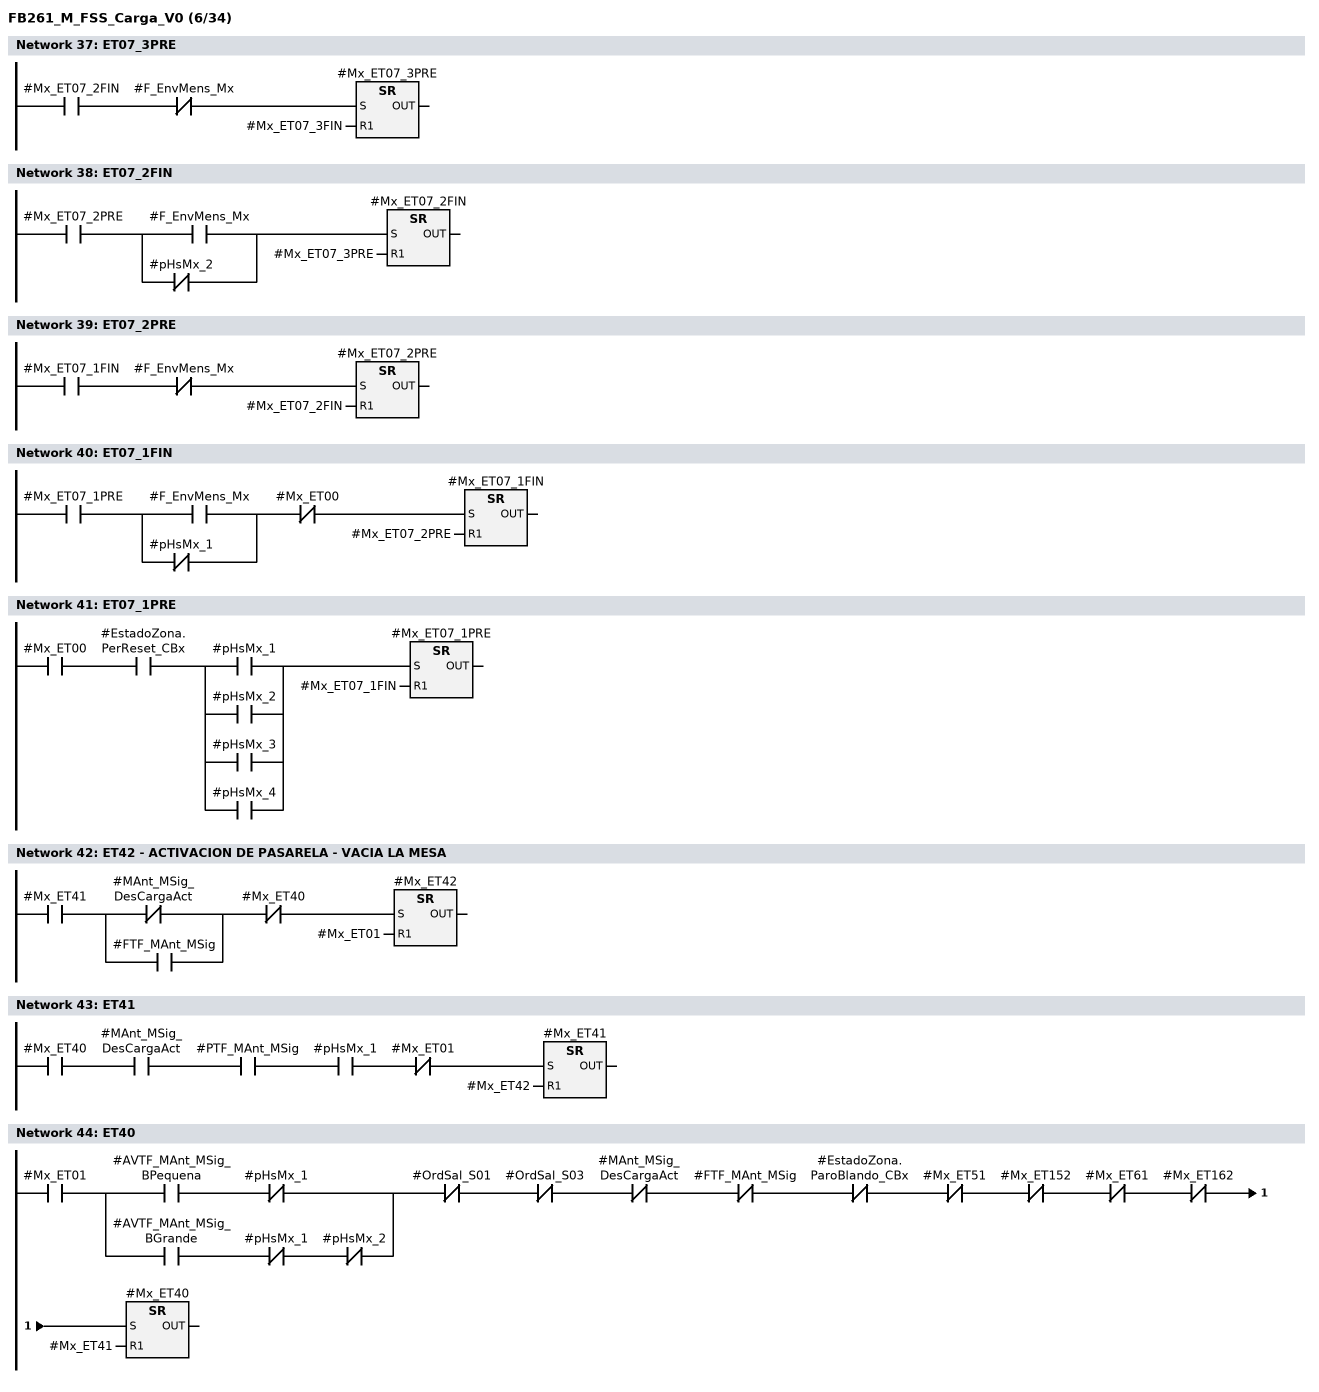
   RUNG wire#powerrail
      Contact( #Mx_ET07_2FIN )
      I_Contact( #F_EnvMens_Mx )
      S_SR(operand := #Mx_ET07_3PRE, r1 := #Mx_ET07_3FIN)
   END_RUNG
   // the same network as SCL:
   IF #Mx_ET07_2FIN AND NOT #F_EnvMens_Mx THEN
       #Mx_ET07_3PRE := TRUE;   // SR flip-flop
   END_IF;
   IF #Mx_ET07_3FIN THEN #Mx_ET07_3PRE := FALSE; END_IF;
END_REGION

REGION Network 38: ET07_2FIN
   RUNG wire#powerrail
      Contact( #Mx_ET07_2PRE )
      wire#w1
      Contact( #F_EnvMens_Mx )
      wire#w2
      S_SR(operand := #Mx_ET07_2FIN, r1 := #Mx_ET07_3PRE)
   END_RUNG
   RUNG wire#w1
      I_Contact( #pHsMx_2 )
   END_RUNG wire#w2
   // the same network as SCL:
   IF #Mx_ET07_2PRE AND (#F_EnvMens_Mx OR NOT #pHsMx_2) THEN
       #Mx_ET07_2FIN := TRUE;   // SR flip-flop
   END_IF;
   IF #Mx_ET07_3PRE THEN #Mx_ET07_2FIN := FALSE; END_IF;
END_REGION

REGION Network 39: ET07_2PRE
   RUNG wire#powerrail
      Contact( #Mx_ET07_1FIN )
      I_Contact( #F_EnvMens_Mx )
      S_SR(operand := #Mx_ET07_2PRE, r1 := #Mx_ET07_2FIN)
   END_RUNG
   // the same network as SCL:
   IF #Mx_ET07_1FIN AND NOT #F_EnvMens_Mx THEN
       #Mx_ET07_2PRE := TRUE;   // SR flip-flop
   END_IF;
   IF #Mx_ET07_2FIN THEN #Mx_ET07_2PRE := FALSE; END_IF;
END_REGION

REGION Network 40: ET07_1FIN
   RUNG wire#powerrail
      Contact( #Mx_ET07_1PRE )
      wire#w1
      Contact( #F_EnvMens_Mx )
      wire#w2
      I_Contact( #Mx_ET00 )
      S_SR(operand := #Mx_ET07_1FIN, r1 := #Mx_ET07_2PRE)
   END_RUNG
   RUNG wire#w1
      I_Contact( #pHsMx_1 )
   END_RUNG wire#w2
   // the same network as SCL:
   IF #Mx_ET07_1PRE AND (#F_EnvMens_Mx OR NOT #pHsMx_1) AND NOT #Mx_ET00 THEN
       #Mx_ET07_1FIN := TRUE;   // SR flip-flop
   END_IF;
   IF #Mx_ET07_2PRE THEN #Mx_ET07_1FIN := FALSE; END_IF;
END_REGION

REGION Network 41: ET07_1PRE
   RUNG wire#powerrail
      Contact( #Mx_ET00 )
      Contact( #EstadoZona.PerReset_CBx )
      wire#w1
      Contact( #pHsMx_1 )
      wire#w2
      S_SR(operand := #Mx_ET07_1PRE, r1 := #Mx_ET07_1FIN)
   END_RUNG
   RUNG wire#w1
      Contact( #pHsMx_2 )
   END_RUNG wire#w2
   RUNG wire#w1
      Contact( #pHsMx_3 )
   END_RUNG wire#w2
   RUNG wire#w1
      Contact( #pHsMx_4 )
   END_RUNG wire#w2
   // the same network as SCL:
   IF #Mx_ET00 AND #EstadoZona.PerReset_CBx AND (#pHsMx_1 OR #pHsMx_2 OR #pHsMx_3 OR #pHsMx_4) THEN
       #Mx_ET07_1PRE := TRUE;   // SR flip-flop
   END_IF;
   IF #Mx_ET07_1FIN THEN #Mx_ET07_1PRE := FALSE; END_IF;
END_REGION

REGION Network 42: ET42 - ACTIVACION DE PASARELA - VACIA LA MESA
   RUNG wire#powerrail
      Contact( #Mx_ET41 )
      wire#w1
      I_Contact( #MAnt_MSig_DesCargaAct )
      wire#w2
      I_Contact( #Mx_ET40 )
      S_SR(operand := #Mx_ET42, r1 := #Mx_ET01)
   END_RUNG
   RUNG wire#w1
      Contact( #FTF_MAnt_MSig )
   END_RUNG wire#w2
   // the same network as SCL:
   IF #Mx_ET41 AND (NOT #MAnt_MSig_DesCargaAct OR #FTF_MAnt_MSig) AND NOT #Mx_ET40 THEN
       #Mx_ET42 := TRUE;   // SR flip-flop
   END_IF;
   IF #Mx_ET01 THEN #Mx_ET42 := FALSE; END_IF;
END_REGION

REGION Network 43: ET41
   RUNG wire#powerrail
      Contact( #Mx_ET40 )
      Contact( #MAnt_MSig_DesCargaAct )
      Contact( #PTF_MAnt_MSig )
      Contact( #pHsMx_1 )
      I_Contact( #Mx_ET01 )
      S_SR(operand := #Mx_ET41, r1 := #Mx_ET42)
   END_RUNG
   // the same network as SCL:
   IF #Mx_ET40 AND #MAnt_MSig_DesCargaAct AND #PTF_MAnt_MSig AND #pHsMx_1 AND NOT #Mx_ET01 THEN
       #Mx_ET41 := TRUE;   // SR flip-flop
   END_IF;
   IF #Mx_ET42 THEN #Mx_ET41 := FALSE; END_IF;
END_REGION

REGION Network 44: ET40
   RUNG wire#powerrail
      Contact( #Mx_ET01 )
      wire#w1
      Contact( #AVTF_MAnt_MSig_BPequena )
      I_Contact( #pHsMx_1 )
      wire#w2
      I_Contact( #OrdSal_S01 )
      I_Contact( #OrdSal_S03 )
      I_Contact( #MAnt_MSig_DesCargaAct )
      I_Contact( #FTF_MAnt_MSig )
      I_Contact( #EstadoZona.ParoBlando_CBx )
      I_Contact( #Mx_ET51 )
      I_Contact( #Mx_ET152 )
      I_Contact( #Mx_ET61 )
      I_Contact( #Mx_ET162 )
      S_SR(operand := #Mx_ET40, r1 := #Mx_ET41)
   END_RUNG
   RUNG wire#w1
      Contact( #AVTF_MAnt_MSig_BGrande )
      I_Contact( #pHsMx_1 )
      I_Contact( #pHsMx_2 )
   END_RUNG wire#w2
   // the same network as SCL:
   IF #Mx_ET01 AND ((#AVTF_MAnt_MSig_BPequena AND NOT #pHsMx_1) OR (#AVTF_MAnt_MSig_BGrande AND NOT #pHsMx_1 AND NOT #pHsMx_2)) AND NOT #OrdSal_S01 AND NOT #OrdSal_S03 AND NOT #MAnt_MSig_DesCargaAct AND NOT #FTF_MAnt_MSig AND NOT #EstadoZona.ParoBlando_CBx AND NOT #Mx_ET51 AND NOT #Mx_ET152 AND NOT #Mx_ET61 AND NOT #Mx_ET162 THEN
       #Mx_ET40 := TRUE;   // SR flip-flop
   END_IF;
   IF #Mx_ET41 THEN #Mx_ET40 := FALSE; END_IF;
END_REGION

REGION Network 45: ET15 - CONTROL DE POSICIONADO DESPUES DE ENTRADA
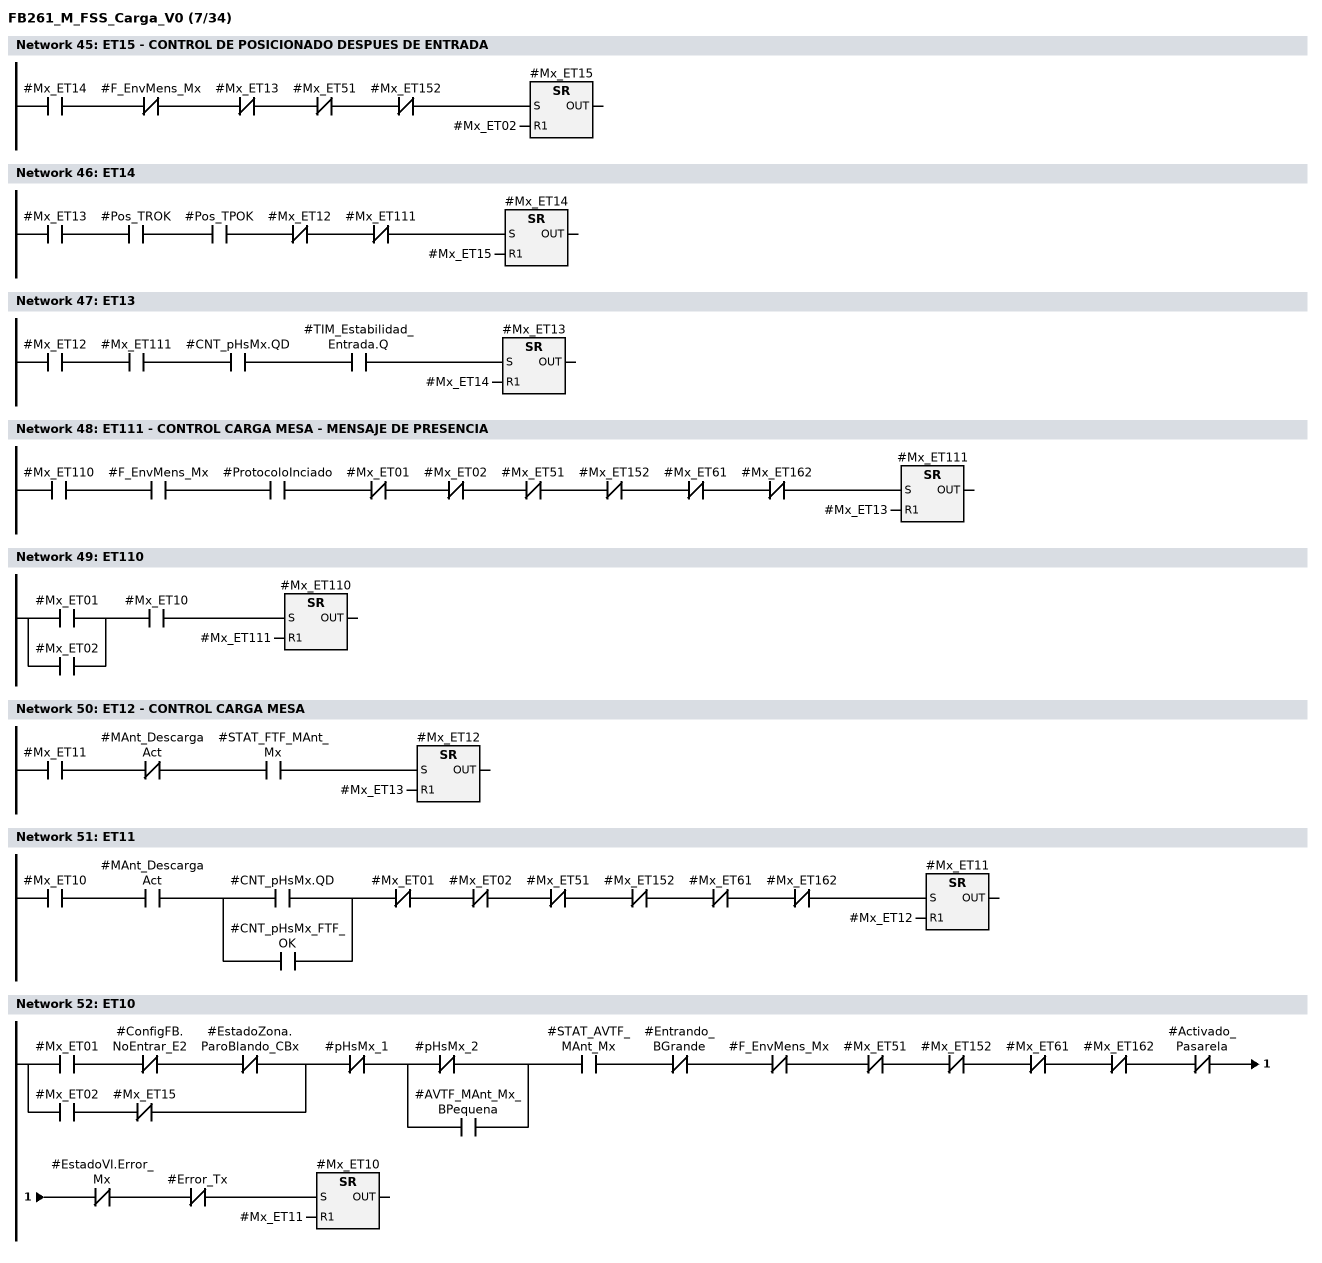
   RUNG wire#powerrail
      Contact( #Mx_ET14 )
      I_Contact( #F_EnvMens_Mx )
      I_Contact( #Mx_ET13 )
      I_Contact( #Mx_ET51 )
      I_Contact( #Mx_ET152 )
      S_SR(operand := #Mx_ET15, r1 := #Mx_ET02)
   END_RUNG
   // the same network as SCL:
   IF #Mx_ET14 AND NOT #F_EnvMens_Mx AND NOT #Mx_ET13 AND NOT #Mx_ET51 AND NOT #Mx_ET152 THEN
       #Mx_ET15 := TRUE;   // SR flip-flop
   END_IF;
   IF #Mx_ET02 THEN #Mx_ET15 := FALSE; END_IF;
END_REGION

REGION Network 46: ET14
   RUNG wire#powerrail
      Contact( #Mx_ET13 )
      Contact( #Pos_TROK )
      Contact( #Pos_TPOK )
      I_Contact( #Mx_ET12 )
      I_Contact( #Mx_ET111 )
      S_SR(operand := #Mx_ET14, r1 := #Mx_ET15)
   END_RUNG
   // the same network as SCL:
   IF #Mx_ET13 AND #Pos_TROK AND #Pos_TPOK AND NOT #Mx_ET12 AND NOT #Mx_ET111 THEN
       #Mx_ET14 := TRUE;   // SR flip-flop
   END_IF;
   IF #Mx_ET15 THEN #Mx_ET14 := FALSE; END_IF;
END_REGION

REGION Network 47: ET13
   RUNG wire#powerrail
      Contact( #Mx_ET12 )
      Contact( #Mx_ET111 )
      Contact( #CNT_pHsMx.QD )
      Contact( #TIM_Estabilidad_Entrada.Q )
      S_SR(operand := #Mx_ET13, r1 := #Mx_ET14)
   END_RUNG
   // the same network as SCL:
   IF #Mx_ET12 AND #Mx_ET111 AND #CNT_pHsMx.QD AND #TIM_Estabilidad_Entrada.Q THEN
       #Mx_ET13 := TRUE;   // SR flip-flop
   END_IF;
   IF #Mx_ET14 THEN #Mx_ET13 := FALSE; END_IF;
END_REGION

REGION Network 48: ET111 - CONTROL CARGA MESA - MENSAJE DE PRESENCIA
   RUNG wire#powerrail
      Contact( #Mx_ET110 )
      Contact( #F_EnvMens_Mx )
      Contact( #ProtocoloInciado )
      I_Contact( #Mx_ET01 )
      I_Contact( #Mx_ET02 )
      I_Contact( #Mx_ET51 )
      I_Contact( #Mx_ET152 )
      I_Contact( #Mx_ET61 )
      I_Contact( #Mx_ET162 )
      S_SR(operand := #Mx_ET111, r1 := #Mx_ET13)
   END_RUNG
   // the same network as SCL:
   IF #Mx_ET110 AND #F_EnvMens_Mx AND #ProtocoloInciado AND NOT #Mx_ET01 AND NOT #Mx_ET02 AND NOT #Mx_ET51 AND NOT #Mx_ET152 AND NOT #Mx_ET61 AND NOT #Mx_ET162 THEN
       #Mx_ET111 := TRUE;   // SR flip-flop
   END_IF;
   IF #Mx_ET13 THEN #Mx_ET111 := FALSE; END_IF;
END_REGION

REGION Network 49: ET110
   RUNG wire#powerrail
      Contact( #Mx_ET01 )
      wire#w1
      Contact( #Mx_ET10 )
      S_SR(operand := #Mx_ET110, r1 := #Mx_ET111)
   END_RUNG
   RUNG wire#powerrail
      Contact( #Mx_ET02 )
   END_RUNG wire#w1
   // the same network as SCL:
   IF (#Mx_ET01 OR #Mx_ET02) AND #Mx_ET10 THEN
       #Mx_ET110 := TRUE;   // SR flip-flop
   END_IF;
   IF #Mx_ET111 THEN #Mx_ET110 := FALSE; END_IF;
END_REGION

REGION Network 50: ET12 - CONTROL CARGA MESA
   RUNG wire#powerrail
      Contact( #Mx_ET11 )
      I_Contact( #MAnt_DescargaAct )
      Contact( #STAT_FTF_MAnt_Mx )
      S_SR(operand := #Mx_ET12, r1 := #Mx_ET13)
   END_RUNG
   // the same network as SCL:
   IF #Mx_ET11 AND NOT #MAnt_DescargaAct AND #STAT_FTF_MAnt_Mx THEN
       #Mx_ET12 := TRUE;   // SR flip-flop
   END_IF;
   IF #Mx_ET13 THEN #Mx_ET12 := FALSE; END_IF;
END_REGION

REGION Network 51: ET11
   RUNG wire#powerrail
      Contact( #Mx_ET10 )
      Contact( #MAnt_DescargaAct )
      wire#w1
      Contact( #CNT_pHsMx.QD )
      wire#w2
      I_Contact( #Mx_ET01 )
      I_Contact( #Mx_ET02 )
      I_Contact( #Mx_ET51 )
      I_Contact( #Mx_ET152 )
      I_Contact( #Mx_ET61 )
      I_Contact( #Mx_ET162 )
      S_SR(operand := #Mx_ET11, r1 := #Mx_ET12)
   END_RUNG
   RUNG wire#w1
      Contact( #CNT_pHsMx_FTF_OK )
   END_RUNG wire#w2
   // the same network as SCL:
   IF #Mx_ET10 AND #MAnt_DescargaAct AND (#CNT_pHsMx.QD OR #CNT_pHsMx_FTF_OK) AND NOT #Mx_ET01 AND NOT #Mx_ET02 AND NOT #Mx_ET51 AND NOT #Mx_ET152 AND NOT #Mx_ET61 AND NOT #Mx_ET162 THEN
       #Mx_ET11 := TRUE;   // SR flip-flop
   END_IF;
   IF #Mx_ET12 THEN #Mx_ET11 := FALSE; END_IF;
END_REGION

REGION Network 52: ET10
   RUNG wire#powerrail
      Contact( #Mx_ET01 )
      I_Contact( #ConfigFB.NoEntrar_E2 )
      I_Contact( #EstadoZona.ParoBlando_CBx )
      wire#w1
      I_Contact( #pHsMx_1 )
      wire#w2
      I_Contact( #pHsMx_2 )
      wire#w3
      Contact( #STAT_AVTF_MAnt_Mx )
      I_Contact( #Entrando_BGrande )
      I_Contact( #F_EnvMens_Mx )
      I_Contact( #Mx_ET51 )
      I_Contact( #Mx_ET152 )
      I_Contact( #Mx_ET61 )
      I_Contact( #Mx_ET162 )
      I_Contact( #Activado_Pasarela )
      I_Contact( #EstadoVI.Error_Mx )
      I_Contact( #Error_Tx )
      S_SR(operand := #Mx_ET10, r1 := #Mx_ET11)
   END_RUNG
   RUNG wire#powerrail
      Contact( #Mx_ET02 )
      I_Contact( #Mx_ET15 )
   END_RUNG wire#w1
   RUNG wire#w2
      Contact( #AVTF_MAnt_Mx_BPequena )
   END_RUNG wire#w3
   // the same network as SCL:
   IF ((#Mx_ET01 AND NOT #ConfigFB.NoEntrar_E2 AND NOT #EstadoZona.ParoBlando_CBx) OR (#Mx_ET02 AND NOT #Mx_ET15)) AND NOT #pHsMx_1 AND (NOT #pHsMx_2 OR #AVTF_MAnt_Mx_BPequena) AND #STAT_AVTF_MAnt_Mx AND NOT #Entrando_BGrande AND NOT #F_EnvMens_Mx AND NOT #Mx_ET51 AND NOT #Mx_ET152 AND NOT #Mx_ET61 AND NOT #Mx_ET162 AND NOT #Activado_Pasarela AND NOT #EstadoVI.Error_Mx AND NOT #Error_Tx THEN
       #Mx_ET10 := TRUE;   // SR flip-flop
   END_IF;
   IF #Mx_ET11 THEN #Mx_ET10 := FALSE; END_IF;
END_REGION

REGION Network 53: ET01 - ESTADO REPOSO VACIO
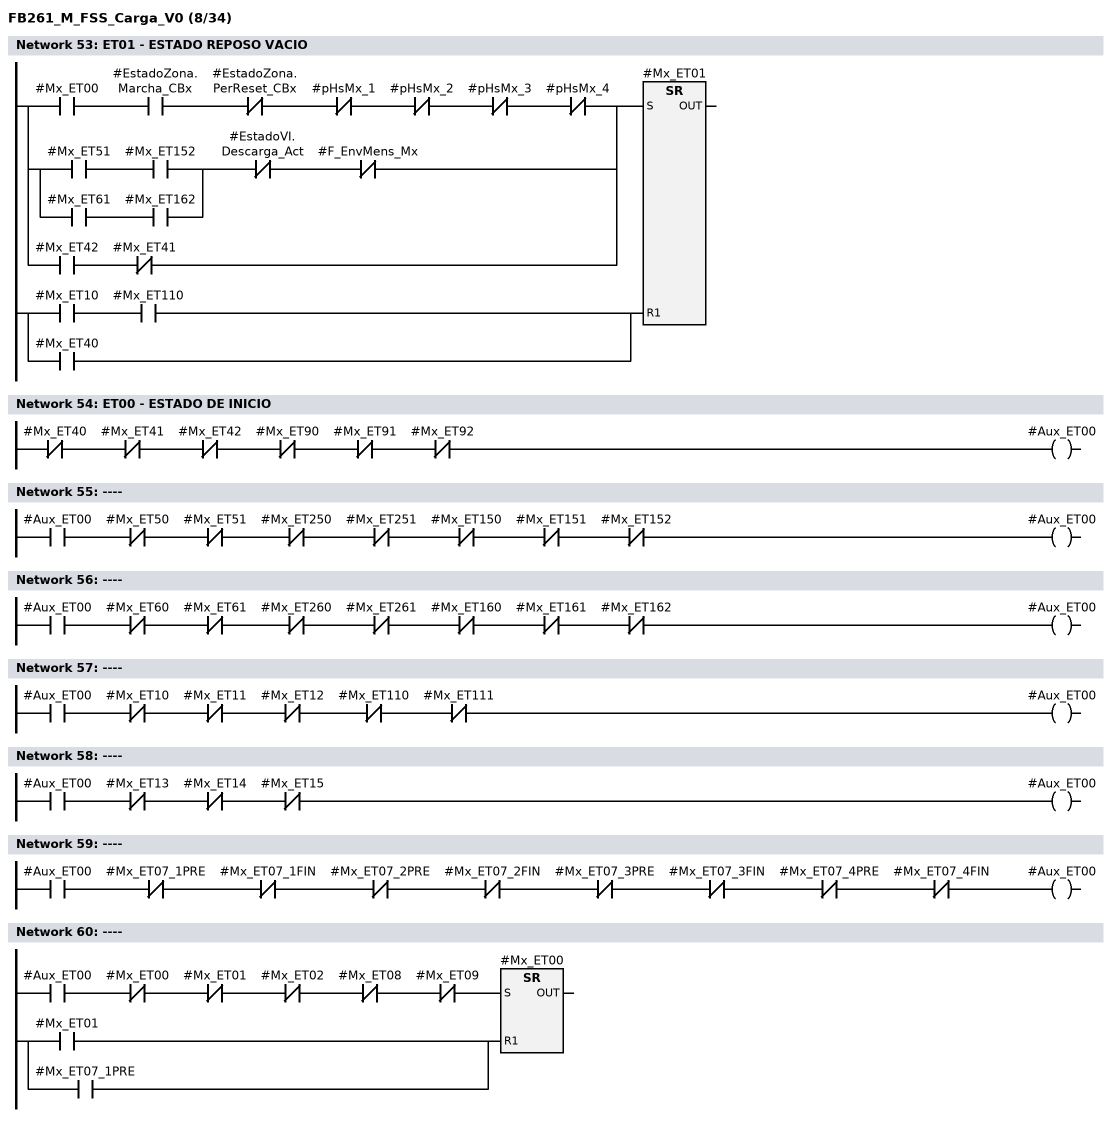
   RUNG wire#powerrail
      Contact( #Mx_ET00 )
      Contact( #EstadoZona.Marcha_CBx )
      I_Contact( #EstadoZona.PerReset_CBx )
      I_Contact( #pHsMx_1 )
      I_Contact( #pHsMx_2 )
      I_Contact( #pHsMx_3 )
      I_Contact( #pHsMx_4 )
      wire#w1
      S_SR(operand := #Mx_ET01, r1 := wire#w3)
   END_RUNG
   RUNG wire#powerrail
      Contact( #Mx_ET51 )
      Contact( #Mx_ET152 )
      wire#w2
      I_Contact( #EstadoVI.Descarga_Act )
      I_Contact( #F_EnvMens_Mx )
   END_RUNG wire#w1
   RUNG wire#powerrail
      Contact( #Mx_ET61 )
      Contact( #Mx_ET162 )
   END_RUNG wire#w2
   RUNG wire#powerrail
      Contact( #Mx_ET42 )
      I_Contact( #Mx_ET41 )
   END_RUNG wire#w1
   RUNG wire#powerrail
      Contact( #Mx_ET10 )
      Contact( #Mx_ET110 )
   END_RUNG wire#w3
   RUNG wire#powerrail
      Contact( #Mx_ET40 )
   END_RUNG wire#w3
   // the same network as SCL:
   IF (#Mx_ET00 AND #EstadoZona.Marcha_CBx AND NOT #EstadoZona.PerReset_CBx AND NOT #pHsMx_1 AND NOT #pHsMx_2 AND NOT #pHsMx_3 AND NOT #pHsMx_4) OR (((#Mx_ET51 AND #Mx_ET152) OR (#Mx_ET61 AND #Mx_ET162)) AND NOT #EstadoVI.Descarga_Act AND NOT #F_EnvMens_Mx) OR (#Mx_ET42 AND NOT #Mx_ET41) THEN
       #Mx_ET01 := TRUE;   // SR flip-flop
   END_IF;
   IF (#Mx_ET10 AND #Mx_ET110) OR #Mx_ET40 THEN #Mx_ET01 := FALSE; END_IF;
END_REGION

REGION Network 54: ET00 - ESTADO DE INICIO
   RUNG wire#powerrail
      I_Contact( #Mx_ET40 )
      I_Contact( #Mx_ET41 )
      I_Contact( #Mx_ET42 )
      I_Contact( #Mx_ET90 )
      I_Contact( #Mx_ET91 )
      I_Contact( #Mx_ET92 )
      Coil( #Aux_ET00 )
   END_RUNG
   // the same network as SCL:
   #Aux_ET00 := NOT #Mx_ET40 AND NOT #Mx_ET41 AND NOT #Mx_ET42 AND NOT #Mx_ET90 AND NOT #Mx_ET91 AND NOT #Mx_ET92;
END_REGION

REGION Network 55: ----
   RUNG wire#powerrail
      Contact( #Aux_ET00 )
      I_Contact( #Mx_ET50 )
      I_Contact( #Mx_ET51 )
      I_Contact( #Mx_ET250 )
      I_Contact( #Mx_ET251 )
      I_Contact( #Mx_ET150 )
      I_Contact( #Mx_ET151 )
      I_Contact( #Mx_ET152 )
      Coil( #Aux_ET00 )
   END_RUNG
   // the same network as SCL:
   #Aux_ET00 := #Aux_ET00 AND NOT #Mx_ET50 AND NOT #Mx_ET51 AND NOT #Mx_ET250 AND NOT #Mx_ET251 AND NOT #Mx_ET150 AND NOT #Mx_ET151 AND NOT #Mx_ET152;
END_REGION

REGION Network 56: ----
   RUNG wire#powerrail
      Contact( #Aux_ET00 )
      I_Contact( #Mx_ET60 )
      I_Contact( #Mx_ET61 )
      I_Contact( #Mx_ET260 )
      I_Contact( #Mx_ET261 )
      I_Contact( #Mx_ET160 )
      I_Contact( #Mx_ET161 )
      I_Contact( #Mx_ET162 )
      Coil( #Aux_ET00 )
   END_RUNG
   // the same network as SCL:
   #Aux_ET00 := #Aux_ET00 AND NOT #Mx_ET60 AND NOT #Mx_ET61 AND NOT #Mx_ET260 AND NOT #Mx_ET261 AND NOT #Mx_ET160 AND NOT #Mx_ET161 AND NOT #Mx_ET162;
END_REGION

REGION Network 57: ----
   RUNG wire#powerrail
      Contact( #Aux_ET00 )
      I_Contact( #Mx_ET10 )
      I_Contact( #Mx_ET11 )
      I_Contact( #Mx_ET12 )
      I_Contact( #Mx_ET110 )
      I_Contact( #Mx_ET111 )
      Coil( #Aux_ET00 )
   END_RUNG
   // the same network as SCL:
   #Aux_ET00 := #Aux_ET00 AND NOT #Mx_ET10 AND NOT #Mx_ET11 AND NOT #Mx_ET12 AND NOT #Mx_ET110 AND NOT #Mx_ET111;
END_REGION

REGION Network 58: ----
   RUNG wire#powerrail
      Contact( #Aux_ET00 )
      I_Contact( #Mx_ET13 )
      I_Contact( #Mx_ET14 )
      I_Contact( #Mx_ET15 )
      Coil( #Aux_ET00 )
   END_RUNG
   // the same network as SCL:
   #Aux_ET00 := #Aux_ET00 AND NOT #Mx_ET13 AND NOT #Mx_ET14 AND NOT #Mx_ET15;
END_REGION

REGION Network 59: ----
   RUNG wire#powerrail
      Contact( #Aux_ET00 )
      I_Contact( #Mx_ET07_1PRE )
      I_Contact( #Mx_ET07_1FIN )
      I_Contact( #Mx_ET07_2PRE )
      I_Contact( #Mx_ET07_2FIN )
      I_Contact( #Mx_ET07_3PRE )
      I_Contact( #Mx_ET07_3FIN )
      I_Contact( #Mx_ET07_4PRE )
      I_Contact( #Mx_ET07_4FIN )
      Coil( #Aux_ET00 )
   END_RUNG
   // the same network as SCL:
   #Aux_ET00 := #Aux_ET00 AND NOT #Mx_ET07_1PRE AND NOT #Mx_ET07_1FIN AND NOT #Mx_ET07_2PRE AND NOT #Mx_ET07_2FIN AND NOT #Mx_ET07_3PRE AND NOT #Mx_ET07_3FIN AND NOT #Mx_ET07_4PRE AND NOT #Mx_ET07_4FIN;
END_REGION

REGION Network 60: ----
   RUNG wire#powerrail
      Contact( #Aux_ET00 )
      I_Contact( #Mx_ET00 )
      I_Contact( #Mx_ET01 )
      I_Contact( #Mx_ET02 )
      I_Contact( #Mx_ET08 )
      I_Contact( #Mx_ET09 )
      S_SR(operand := #Mx_ET00, r1 := wire#w1)
   END_RUNG
   RUNG wire#powerrail
      Contact( #Mx_ET01 )
   END_RUNG wire#w1
   RUNG wire#powerrail
      Contact( #Mx_ET07_1PRE )
   END_RUNG wire#w1
   // the same network as SCL:
   IF #Aux_ET00 AND NOT #Mx_ET00 AND NOT #Mx_ET01 AND NOT #Mx_ET02 AND NOT #Mx_ET08 AND NOT #Mx_ET09 THEN
       #Mx_ET00 := TRUE;   // SR flip-flop
   END_IF;
   IF #Mx_ET01 OR #Mx_ET07_1PRE THEN #Mx_ET00 := FALSE; END_IF;
END_REGION

REGION Network 61: CONTADOR DE SEGURIDAD DE PRESENCIA - CNTSeg_pHsMx
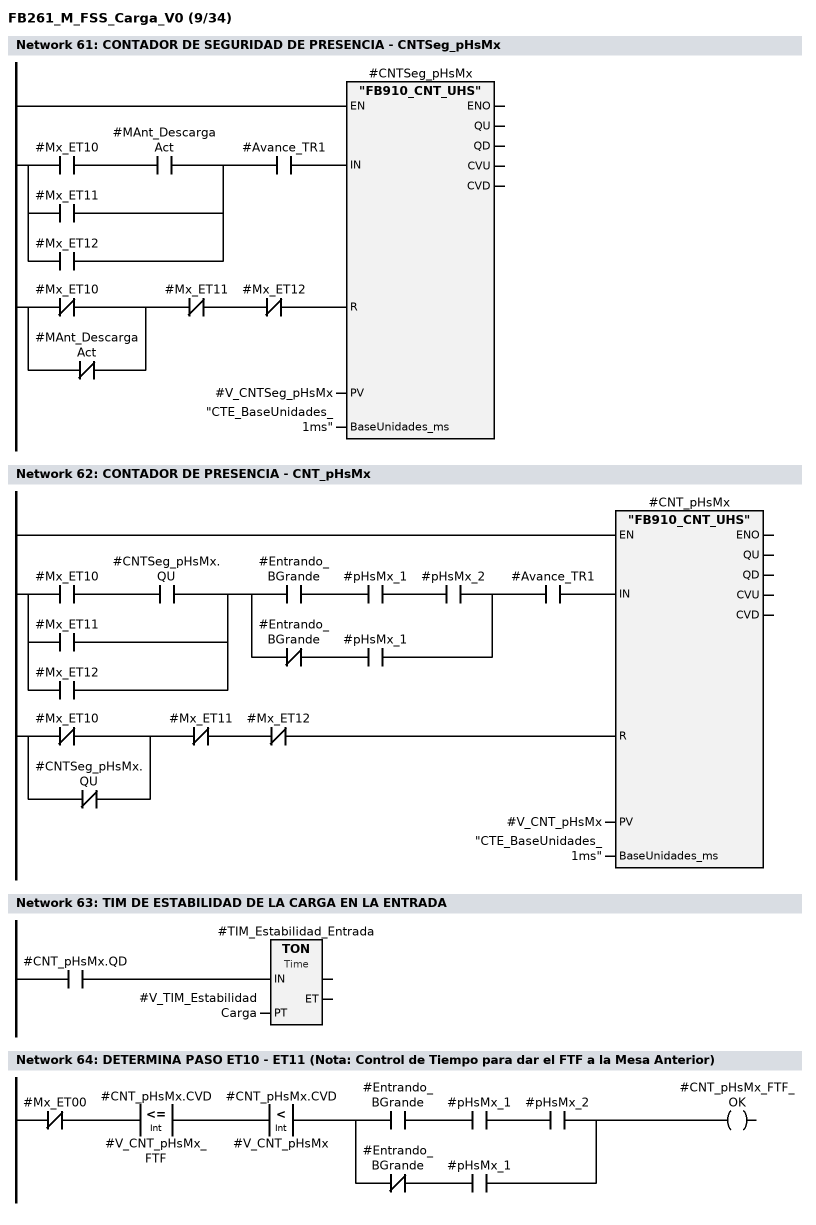
   RUNG wire#powerrail
      #CNTSeg_pHsMx(IN := wire#w2, R := wire#w4, PV := #V_CNTSeg_pHsMx, BaseUnidades_ms := "CTE_BaseUnidades_1ms", QU =>, QD =>, CVU =>, CVD =>)
   END_RUNG
   RUNG wire#powerrail
      Contact( #Mx_ET10 )
      Contact( #MAnt_DescargaAct )
      wire#w1
      Contact( #Avance_TR1 )
   END_RUNG wire#w2
   RUNG wire#powerrail
      Contact( #Mx_ET11 )
   END_RUNG wire#w1
   RUNG wire#powerrail
      Contact( #Mx_ET12 )
   END_RUNG wire#w1
   RUNG wire#powerrail
      I_Contact( #Mx_ET10 )
      wire#w3
      I_Contact( #Mx_ET11 )
      I_Contact( #Mx_ET12 )
   END_RUNG wire#w4
   RUNG wire#powerrail
      I_Contact( #MAnt_DescargaAct )
   END_RUNG wire#w3
   // the same network as SCL:
   #CNTSeg_pHsMx(IN := ((#Mx_ET10 AND #MAnt_DescargaAct) OR #Mx_ET11 OR #Mx_ET12) AND #Avance_TR1,   // "FB910_CNT_UHS"
                 R := (NOT #Mx_ET10 OR NOT #MAnt_DescargaAct) AND NOT #Mx_ET11 AND NOT #Mx_ET12,
                 PV := #V_CNTSeg_pHsMx,
                 BaseUnidades_ms := "CTE_BaseUnidades_1ms");
END_REGION

REGION Network 62: CONTADOR DE PRESENCIA - CNT_pHsMx
   RUNG wire#powerrail
      #CNT_pHsMx(IN := wire#w3, R := wire#w5, PV := #V_CNT_pHsMx, BaseUnidades_ms := "CTE_BaseUnidades_1ms", QU =>, QD =>, CVU =>, CVD =>)
   END_RUNG
   RUNG wire#powerrail
      Contact( #Mx_ET10 )
      Contact( #CNTSeg_pHsMx.QU )
      wire#w1
      Contact( #Entrando_BGrande )
      Contact( #pHsMx_1 )
      Contact( #pHsMx_2 )
      wire#w2
      Contact( #Avance_TR1 )
   END_RUNG wire#w3
   RUNG wire#powerrail
      Contact( #Mx_ET11 )
   END_RUNG wire#w1
   RUNG wire#powerrail
      Contact( #Mx_ET12 )
   END_RUNG wire#w1
   RUNG wire#w1
      I_Contact( #Entrando_BGrande )
      Contact( #pHsMx_1 )
   END_RUNG wire#w2
   RUNG wire#powerrail
      I_Contact( #Mx_ET10 )
      wire#w4
      I_Contact( #Mx_ET11 )
      I_Contact( #Mx_ET12 )
   END_RUNG wire#w5
   RUNG wire#powerrail
      I_Contact( #CNTSeg_pHsMx.QU )
   END_RUNG wire#w4
   // the same network as SCL:
   #CNT_pHsMx(IN := ((#Mx_ET10 AND #CNTSeg_pHsMx.QU) OR #Mx_ET11 OR #Mx_ET12) AND ((#Entrando_BGrande AND #pHsMx_1 AND #pHsMx_2) OR (NOT #Entrando_BGrande AND #pHsMx_1)) AND #Avance_TR1,   // "FB910_CNT_UHS"
              R := (NOT #Mx_ET10 OR NOT #CNTSeg_pHsMx.QU) AND NOT #Mx_ET11 AND NOT #Mx_ET12,
              PV := #V_CNT_pHsMx,
              BaseUnidades_ms := "CTE_BaseUnidades_1ms");
END_REGION

REGION Network 63: TIM DE ESTABILIDAD DE LA CARGA EN LA ENTRADA
   RUNG wire#powerrail
      Contact( #CNT_pHsMx.QD )
      { S7_Templates := "time_type := Time" } #TIM_Estabilidad_Entrada.TON(pt := #V_TIM_EstabilidadCarga, et =>)
   END_RUNG
   // the same network as SCL:
   #TIM_Estabilidad_Entrada(IN := #CNT_pHsMx.QD, PT := #V_TIM_EstabilidadCarga);   // TON
END_REGION

REGION Network 64: DETERMINA PASO ET10 - ET11 (Nota: Control de Tiempo para dar el FTF a la Mesa Anterior)
   RUNG wire#powerrail
      I_Contact( #Mx_ET00 )
      { S7_Templates := "SrcType := Int" } LE_Contact(in1 := #CNT_pHsMx.CVD, in2 := #V_CNT_pHsMx_FTF)
      { S7_Templates := "SrcType := Int" } LT_Contact(in1 := #CNT_pHsMx.CVD, in2 := #V_CNT_pHsMx)
      wire#w1
      Contact( #Entrando_BGrande )
      Contact( #pHsMx_1 )
      Contact( #pHsMx_2 )
      wire#w2
      Coil( #CNT_pHsMx_FTF_OK )
   END_RUNG
   RUNG wire#w1
      I_Contact( #Entrando_BGrande )
      Contact( #pHsMx_1 )
   END_RUNG wire#w2
   // the same network as SCL:
   #CNT_pHsMx_FTF_OK := NOT #Mx_ET00 AND (#CNT_pHsMx.CVD <= #V_CNT_pHsMx_FTF) AND (#CNT_pHsMx.CVD < #V_CNT_pHsMx) AND ((#Entrando_BGrande AND #pHsMx_1 AND #pHsMx_2) OR (NOT #Entrando_BGrande AND #pHsMx_1));
END_REGION

REGION Network 65: CONTADOR SEGURIDAD DE AUSENCIA - CNTSeg_ApHsMx ??????? RESTAR VALOR DE POSICIONAMIENTO
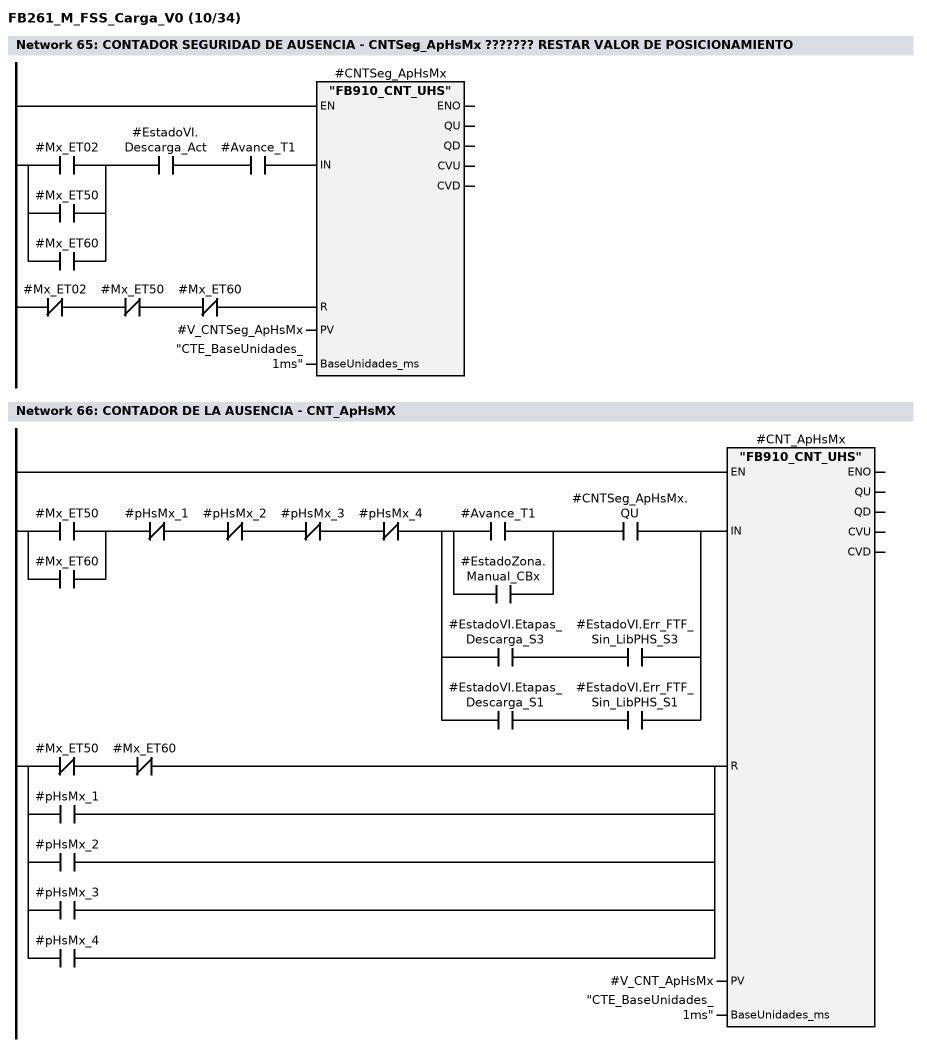
   RUNG wire#powerrail
      #CNTSeg_ApHsMx(IN := wire#w2, R := wire#w3, PV := #V_CNTSeg_ApHsMx, BaseUnidades_ms := "CTE_BaseUnidades_1ms", QU =>, QD =>, CVU =>, CVD =>)
   END_RUNG
   RUNG wire#powerrail
      Contact( #Mx_ET02 )
      wire#w1
      Contact( #EstadoVI.Descarga_Act )
      Contact( #Avance_T1 )
   END_RUNG wire#w2
   RUNG wire#powerrail
      Contact( #Mx_ET50 )
   END_RUNG wire#w1
   RUNG wire#powerrail
      Contact( #Mx_ET60 )
   END_RUNG wire#w1
   RUNG wire#powerrail
      I_Contact( #Mx_ET02 )
      I_Contact( #Mx_ET50 )
      I_Contact( #Mx_ET60 )
   END_RUNG wire#w3
   // the same network as SCL:
   #CNTSeg_ApHsMx(IN := (#Mx_ET02 OR #Mx_ET50 OR #Mx_ET60) AND #EstadoVI.Descarga_Act AND #Avance_T1,   // "FB910_CNT_UHS"
                  R := NOT #Mx_ET02 AND NOT #Mx_ET50 AND NOT #Mx_ET60,
                  PV := #V_CNTSeg_ApHsMx,
                  BaseUnidades_ms := "CTE_BaseUnidades_1ms");
END_REGION

REGION Network 66: CONTADOR DE LA AUSENCIA - CNT_ApHsMX
   RUNG wire#powerrail
      #CNT_ApHsMx(IN := wire#w4, R := wire#w5, PV := #V_CNT_ApHsMx, BaseUnidades_ms := "CTE_BaseUnidades_1ms", QU =>, QD =>, CVU =>, CVD =>)
   END_RUNG
   RUNG wire#powerrail
      Contact( #Mx_ET50 )
      wire#w1
      I_Contact( #pHsMx_1 )
      I_Contact( #pHsMx_2 )
      I_Contact( #pHsMx_3 )
      I_Contact( #pHsMx_4 )
      wire#w2
      Contact( #Avance_T1 )
      wire#w3
      Contact( #CNTSeg_ApHsMx.QU )
   END_RUNG wire#w4
   RUNG wire#powerrail
      Contact( #Mx_ET60 )
   END_RUNG wire#w1
   RUNG wire#w2
      Contact( #EstadoZona.Manual_CBx )
   END_RUNG wire#w3
   RUNG wire#w2
      Contact( #EstadoVI.Etapas_Descarga_S3 )
      Contact( #EstadoVI.Err_FTF_Sin_LibPHS_S3 )
   END_RUNG wire#w4
   RUNG wire#w2
      Contact( #EstadoVI.Etapas_Descarga_S1 )
      Contact( #EstadoVI.Err_FTF_Sin_LibPHS_S1 )
   END_RUNG wire#w4
   RUNG wire#powerrail
      I_Contact( #Mx_ET50 )
      I_Contact( #Mx_ET60 )
   END_RUNG wire#w5
   RUNG wire#powerrail
      Contact( #pHsMx_1 )
   END_RUNG wire#w5
   RUNG wire#powerrail
      Contact( #pHsMx_2 )
   END_RUNG wire#w5
   RUNG wire#powerrail
      Contact( #pHsMx_3 )
   END_RUNG wire#w5
   RUNG wire#powerrail
      Contact( #pHsMx_4 )
   END_RUNG wire#w5
   // the same network as SCL:
   #CNT_ApHsMx(IN := (#Mx_ET50 OR #Mx_ET60) AND NOT #pHsMx_1 AND NOT #pHsMx_2 AND NOT #pHsMx_3 AND NOT #pHsMx_4 AND (((#Avance_T1 OR #EstadoZona.Manual_CBx) AND #CNTSeg_ApHsMx.QU) OR (#EstadoVI.Etapas_Descarga_S3 AND #EstadoVI.Err_FTF_Sin_LibPHS_S3) OR (#EstadoVI.Etapas_Descarga_S1 AND #EstadoVI.Err_FTF_Sin_LibPHS_S1)),   // "FB910_CNT_UHS"
               R := (NOT #Mx_ET50 AND NOT #Mx_ET60) OR #pHsMx_1 OR #pHsMx_2 OR #pHsMx_3 OR #pHsMx_4,
               PV := #V_CNT_ApHsMx,
               BaseUnidades_ms := "CTE_BaseUnidades_1ms");
END_REGION

REGION Network 67: CONTADOR DE POSICIONAMIENTO DE LA CARGA DESPUES DE LA ENTRADA
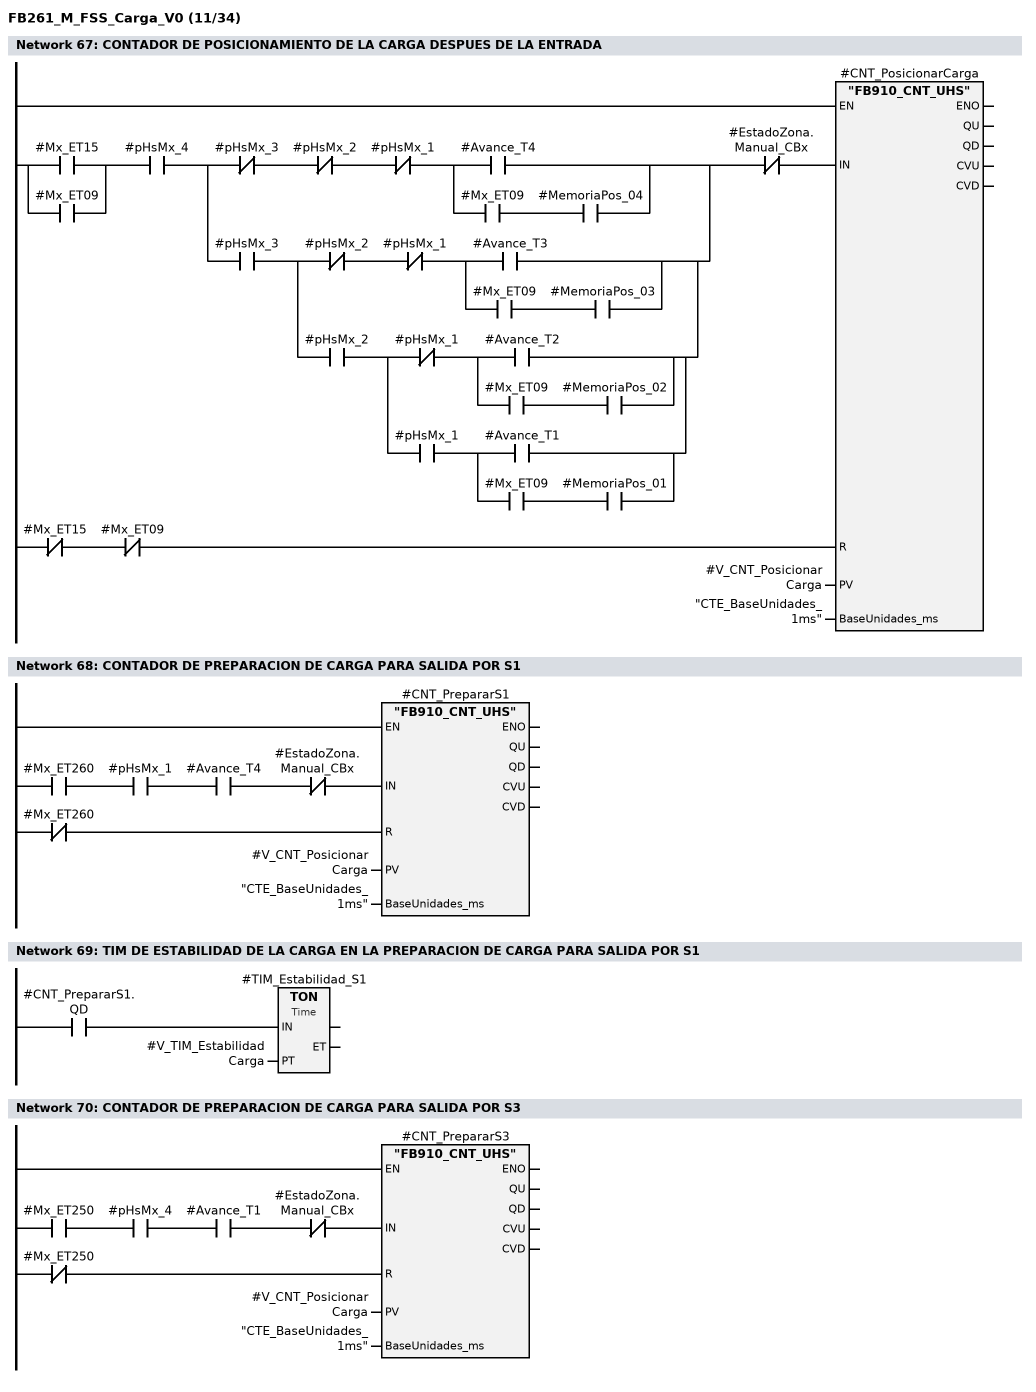
   RUNG wire#powerrail
      #CNT_PosicionarCarga(IN := wire#w10, R := wire#w11, PV := #V_CNT_PosicionarCarga, BaseUnidades_ms := "CTE_BaseUnidades_1ms", QU =>, QD =>, CVU =>, CVD =>)
   END_RUNG
   RUNG wire#powerrail
      Contact( #Mx_ET15 )
      wire#w1
      Contact( #pHsMx_4 )
      wire#w2
      I_Contact( #pHsMx_3 )
      I_Contact( #pHsMx_2 )
      I_Contact( #pHsMx_1 )
      wire#w3
      Contact( #Avance_T4 )
      wire#w4
      I_Contact( #EstadoZona.Manual_CBx )
   END_RUNG wire#w10
   RUNG wire#powerrail
      Contact( #Mx_ET09 )
   END_RUNG wire#w1
   RUNG wire#w3
      Contact( #Mx_ET09 )
      Contact( #MemoriaPos_04 )
   END_RUNG wire#w4
   RUNG wire#w2
      Contact( #pHsMx_3 )
      wire#w5
      I_Contact( #pHsMx_2 )
      I_Contact( #pHsMx_1 )
      wire#w6
      Contact( #Avance_T3 )
   END_RUNG wire#w4
   RUNG wire#w6
      Contact( #Mx_ET09 )
      Contact( #MemoriaPos_03 )
   END_RUNG wire#w4
   RUNG wire#w5
      Contact( #pHsMx_2 )
      wire#w7
      I_Contact( #pHsMx_1 )
      wire#w8
      Contact( #Avance_T2 )
   END_RUNG wire#w4
   RUNG wire#w8
      Contact( #Mx_ET09 )
      Contact( #MemoriaPos_02 )
   END_RUNG wire#w4
   RUNG wire#w7
      Contact( #pHsMx_1 )
      wire#w9
      Contact( #Avance_T1 )
   END_RUNG wire#w4
   RUNG wire#w9
      Contact( #Mx_ET09 )
      Contact( #MemoriaPos_01 )
   END_RUNG wire#w4
   RUNG wire#powerrail
      I_Contact( #Mx_ET15 )
      I_Contact( #Mx_ET09 )
   END_RUNG wire#w11
   // the same network as SCL:
   #CNT_PosicionarCarga(IN := (#Mx_ET15 OR #Mx_ET09) AND #pHsMx_4 AND ((NOT #pHsMx_3 AND NOT #pHsMx_2 AND NOT #pHsMx_1 AND (#Avance_T4 OR (#Mx_ET09 AND #MemoriaPos_04))) OR (#pHsMx_3 AND ((NOT #pHsMx_2 AND NOT #pHsMx_1 AND (#Avance_T3 OR (#Mx_ET09 AND #MemoriaPos_03))) OR (#pHsMx_2 AND ((NOT #pHsMx_1 AND (#Avance_T2 OR (#Mx_ET09 AND #MemoriaPos_02))) OR (#pHsMx_1 AND (#Avance_T1 OR (#Mx_ET09 AND #MemoriaPos_01)))))))) AND NOT #EstadoZona.Manual_CBx,   // "FB910_CNT_UHS"
                        R := NOT #Mx_ET15 AND NOT #Mx_ET09,
                        PV := #V_CNT_PosicionarCarga,
                        BaseUnidades_ms := "CTE_BaseUnidades_1ms");
END_REGION

REGION Network 68: CONTADOR DE PREPARACION DE CARGA PARA SALIDA POR S1
   RUNG wire#powerrail
      #CNT_PrepararS1(IN := wire#w1, R := wire#w2, PV := #V_CNT_PosicionarCarga, BaseUnidades_ms := "CTE_BaseUnidades_1ms", QU =>, QD =>, CVU =>, CVD =>)
   END_RUNG
   RUNG wire#powerrail
      Contact( #Mx_ET260 )
      Contact( #pHsMx_1 )
      Contact( #Avance_T4 )
      I_Contact( #EstadoZona.Manual_CBx )
   END_RUNG wire#w1
   RUNG wire#powerrail
      I_Contact( #Mx_ET260 )
   END_RUNG wire#w2
   // the same network as SCL:
   #CNT_PrepararS1(IN := #Mx_ET260 AND #pHsMx_1 AND #Avance_T4 AND NOT #EstadoZona.Manual_CBx,   // "FB910_CNT_UHS"
                   R := NOT #Mx_ET260,
                   PV := #V_CNT_PosicionarCarga,
                   BaseUnidades_ms := "CTE_BaseUnidades_1ms");
END_REGION

REGION Network 69: TIM DE ESTABILIDAD DE LA CARGA EN LA PREPARACION DE CARGA PARA SALIDA POR S1
   RUNG wire#powerrail
      Contact( #CNT_PrepararS1.QD )
      { S7_Templates := "time_type := Time" } #TIM_Estabilidad_S1.TON(pt := #V_TIM_EstabilidadCarga, et =>)
   END_RUNG
   // the same network as SCL:
   #TIM_Estabilidad_S1(IN := #CNT_PrepararS1.QD, PT := #V_TIM_EstabilidadCarga);   // TON
END_REGION

REGION Network 70: CONTADOR DE PREPARACION DE CARGA PARA SALIDA POR S3
   RUNG wire#powerrail
      #CNT_PrepararS3(IN := wire#w1, R := wire#w2, PV := #V_CNT_PosicionarCarga, BaseUnidades_ms := "CTE_BaseUnidades_1ms", QU =>, QD =>, CVU =>, CVD =>)
   END_RUNG
   RUNG wire#powerrail
      Contact( #Mx_ET250 )
      Contact( #pHsMx_4 )
      Contact( #Avance_T1 )
      I_Contact( #EstadoZona.Manual_CBx )
   END_RUNG wire#w1
   RUNG wire#powerrail
      I_Contact( #Mx_ET250 )
   END_RUNG wire#w2
   // the same network as SCL:
   #CNT_PrepararS3(IN := #Mx_ET250 AND #pHsMx_4 AND #Avance_T1 AND NOT #EstadoZona.Manual_CBx,   // "FB910_CNT_UHS"
                   R := NOT #Mx_ET250,
                   PV := #V_CNT_PosicionarCarga,
                   BaseUnidades_ms := "CTE_BaseUnidades_1ms");
END_REGION

REGION Network 71: TIM DE ESTABILIDAD DE LA CARGA EN LA PREPARACION DE CARGA PARA SALIDA POR S1
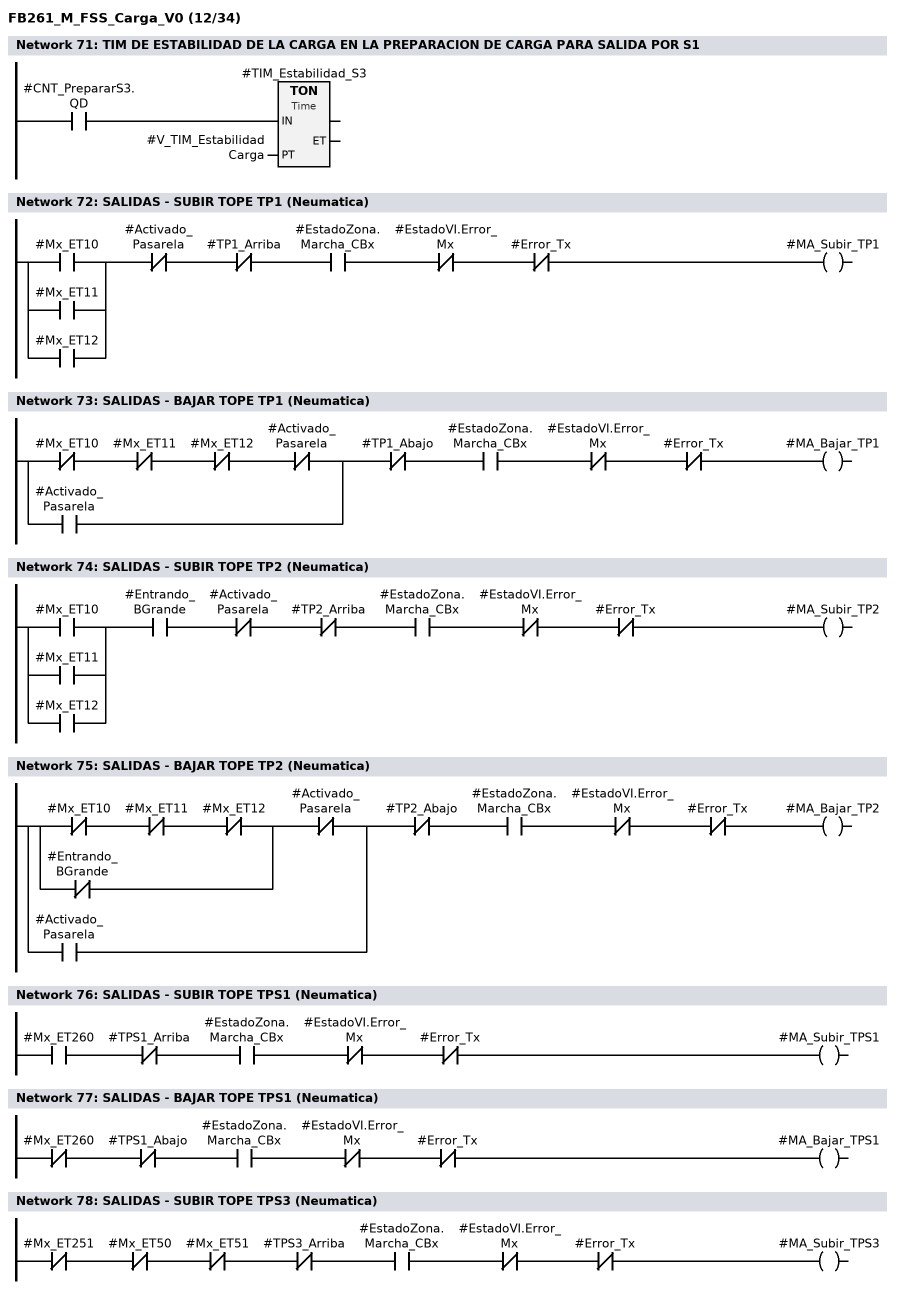
   RUNG wire#powerrail
      Contact( #CNT_PrepararS3.QD )
      { S7_Templates := "time_type := Time" } #TIM_Estabilidad_S3.TON(pt := #V_TIM_EstabilidadCarga, et =>)
   END_RUNG
   // the same network as SCL:
   #TIM_Estabilidad_S3(IN := #CNT_PrepararS3.QD, PT := #V_TIM_EstabilidadCarga);   // TON
END_REGION

REGION Network 72: SALIDAS - SUBIR TOPE TP1 (Neumatica)
   RUNG wire#powerrail
      Contact( #Mx_ET10 )
      wire#w1
      I_Contact( #Activado_Pasarela )
      I_Contact( #TP1_Arriba )
      Contact( #EstadoZona.Marcha_CBx )
      I_Contact( #EstadoVI.Error_Mx )
      I_Contact( #Error_Tx )
      Coil( #MA_Subir_TP1 )
   END_RUNG
   RUNG wire#powerrail
      Contact( #Mx_ET11 )
   END_RUNG wire#w1
   RUNG wire#powerrail
      Contact( #Mx_ET12 )
   END_RUNG wire#w1
   // the same network as SCL:
   #MA_Subir_TP1 := (#Mx_ET10 OR #Mx_ET11 OR #Mx_ET12) AND NOT #Activado_Pasarela AND NOT #TP1_Arriba AND #EstadoZona.Marcha_CBx AND NOT #EstadoVI.Error_Mx AND NOT #Error_Tx;
END_REGION

REGION Network 73: SALIDAS - BAJAR TOPE TP1 (Neumatica)
   RUNG wire#powerrail
      I_Contact( #Mx_ET10 )
      I_Contact( #Mx_ET11 )
      I_Contact( #Mx_ET12 )
      I_Contact( #Activado_Pasarela )
      wire#w1
      I_Contact( #TP1_Abajo )
      Contact( #EstadoZona.Marcha_CBx )
      I_Contact( #EstadoVI.Error_Mx )
      I_Contact( #Error_Tx )
      Coil( #MA_Bajar_TP1 )
   END_RUNG
   RUNG wire#powerrail
      Contact( #Activado_Pasarela )
   END_RUNG wire#w1
   // the same network as SCL:
   #MA_Bajar_TP1 := ((NOT #Mx_ET10 AND NOT #Mx_ET11 AND NOT #Mx_ET12 AND NOT #Activado_Pasarela) OR #Activado_Pasarela) AND NOT #TP1_Abajo AND #EstadoZona.Marcha_CBx AND NOT #EstadoVI.Error_Mx AND NOT #Error_Tx;
END_REGION

REGION Network 74: SALIDAS - SUBIR TOPE TP2 (Neumatica)
   RUNG wire#powerrail
      Contact( #Mx_ET10 )
      wire#w1
      Contact( #Entrando_BGrande )
      I_Contact( #Activado_Pasarela )
      I_Contact( #TP2_Arriba )
      Contact( #EstadoZona.Marcha_CBx )
      I_Contact( #EstadoVI.Error_Mx )
      I_Contact( #Error_Tx )
      Coil( #MA_Subir_TP2 )
   END_RUNG
   RUNG wire#powerrail
      Contact( #Mx_ET11 )
   END_RUNG wire#w1
   RUNG wire#powerrail
      Contact( #Mx_ET12 )
   END_RUNG wire#w1
   // the same network as SCL:
   #MA_Subir_TP2 := (#Mx_ET10 OR #Mx_ET11 OR #Mx_ET12) AND #Entrando_BGrande AND NOT #Activado_Pasarela AND NOT #TP2_Arriba AND #EstadoZona.Marcha_CBx AND NOT #EstadoVI.Error_Mx AND NOT #Error_Tx;
END_REGION

REGION Network 75: SALIDAS - BAJAR TOPE TP2 (Neumatica)
   RUNG wire#powerrail
      I_Contact( #Mx_ET10 )
      I_Contact( #Mx_ET11 )
      I_Contact( #Mx_ET12 )
      wire#w1
      I_Contact( #Activado_Pasarela )
      wire#w2
      I_Contact( #TP2_Abajo )
      Contact( #EstadoZona.Marcha_CBx )
      I_Contact( #EstadoVI.Error_Mx )
      I_Contact( #Error_Tx )
      Coil( #MA_Bajar_TP2 )
   END_RUNG
   RUNG wire#powerrail
      I_Contact( #Entrando_BGrande )
   END_RUNG wire#w1
   RUNG wire#powerrail
      Contact( #Activado_Pasarela )
   END_RUNG wire#w2
   // the same network as SCL:
   #MA_Bajar_TP2 := ((((NOT #Mx_ET10 AND NOT #Mx_ET11 AND NOT #Mx_ET12) OR NOT #Entrando_BGrande) AND NOT #Activado_Pasarela) OR #Activado_Pasarela) AND NOT #TP2_Abajo AND #EstadoZona.Marcha_CBx AND NOT #EstadoVI.Error_Mx AND NOT #Error_Tx;
END_REGION

REGION Network 76: SALIDAS - SUBIR TOPE TPS1 (Neumatica)
   RUNG wire#powerrail
      Contact( #Mx_ET260 )
      I_Contact( #TPS1_Arriba )
      Contact( #EstadoZona.Marcha_CBx )
      I_Contact( #EstadoVI.Error_Mx )
      I_Contact( #Error_Tx )
      Coil( #MA_Subir_TPS1 )
   END_RUNG
   // the same network as SCL:
   #MA_Subir_TPS1 := #Mx_ET260 AND NOT #TPS1_Arriba AND #EstadoZona.Marcha_CBx AND NOT #EstadoVI.Error_Mx AND NOT #Error_Tx;
END_REGION

REGION Network 77: SALIDAS - BAJAR TOPE TPS1 (Neumatica)
   RUNG wire#powerrail
      I_Contact( #Mx_ET260 )
      I_Contact( #TPS1_Abajo )
      Contact( #EstadoZona.Marcha_CBx )
      I_Contact( #EstadoVI.Error_Mx )
      I_Contact( #Error_Tx )
      Coil( #MA_Bajar_TPS1 )
   END_RUNG
   // the same network as SCL:
   #MA_Bajar_TPS1 := NOT #Mx_ET260 AND NOT #TPS1_Abajo AND #EstadoZona.Marcha_CBx AND NOT #EstadoVI.Error_Mx AND NOT #Error_Tx;
END_REGION

REGION Network 78: SALIDAS - SUBIR TOPE TPS3 (Neumatica)
   RUNG wire#powerrail
      I_Contact( #Mx_ET251 )
      I_Contact( #Mx_ET50 )
      I_Contact( #Mx_ET51 )
      I_Contact( #TPS3_Arriba )
      Contact( #EstadoZona.Marcha_CBx )
      I_Contact( #EstadoVI.Error_Mx )
      I_Contact( #Error_Tx )
      Coil( #MA_Subir_TPS3 )
   END_RUNG
   // the same network as SCL:
   #MA_Subir_TPS3 := NOT #Mx_ET251 AND NOT #Mx_ET50 AND NOT #Mx_ET51 AND NOT #TPS3_Arriba AND #EstadoZona.Marcha_CBx AND NOT #EstadoVI.Error_Mx AND NOT #Error_Tx;
END_REGION

REGION Network 79: SALIDAS - BAJAR TOPE TPS3 (Neumatica)
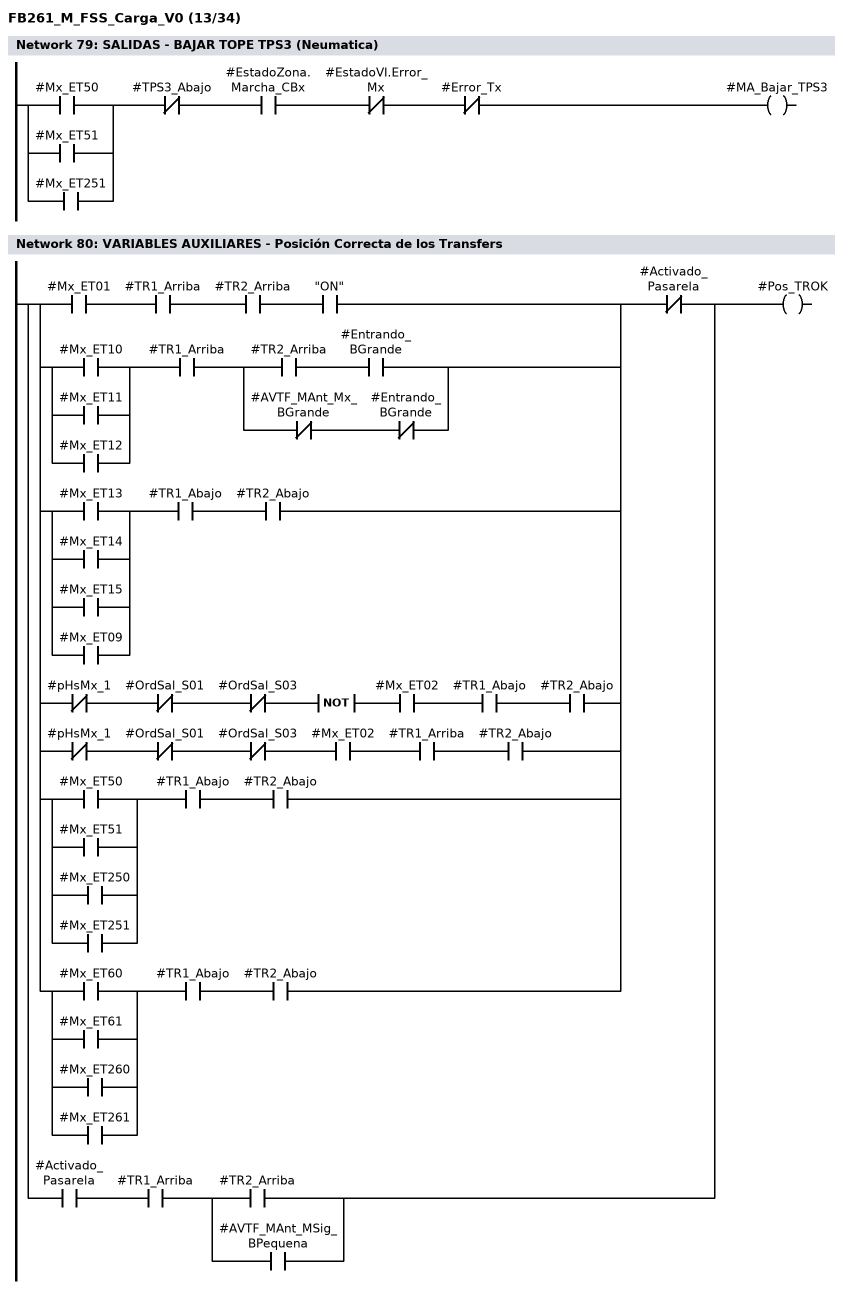
   RUNG wire#powerrail
      Contact( #Mx_ET50 )
      wire#w1
      I_Contact( #TPS3_Abajo )
      Contact( #EstadoZona.Marcha_CBx )
      I_Contact( #EstadoVI.Error_Mx )
      I_Contact( #Error_Tx )
      Coil( #MA_Bajar_TPS3 )
   END_RUNG
   RUNG wire#powerrail
      Contact( #Mx_ET51 )
   END_RUNG wire#w1
   RUNG wire#powerrail
      Contact( #Mx_ET251 )
   END_RUNG wire#w1
   // the same network as SCL:
   #MA_Bajar_TPS3 := (#Mx_ET50 OR #Mx_ET51 OR #Mx_ET251) AND NOT #TPS3_Abajo AND #EstadoZona.Marcha_CBx AND NOT #EstadoVI.Error_Mx AND NOT #Error_Tx;
END_REGION

REGION Network 80: VARIABLES AUXILIARES - Posición Correcta de los Transfers
   RUNG wire#powerrail
      Contact( #Mx_ET01 )
      Contact( #TR1_Arriba )
      Contact( #TR2_Arriba )
      Contact( "ON" )
      wire#w1
      I_Contact( #Activado_Pasarela )
      wire#w7
      Coil( #Pos_TROK )
   END_RUNG
   RUNG wire#powerrail
      Contact( #Mx_ET10 )
      wire#w2
      Contact( #TR1_Arriba )
      wire#w3
      Contact( #TR2_Arriba )
      Contact( #Entrando_BGrande )
   END_RUNG wire#w1
   RUNG wire#powerrail
      Contact( #Mx_ET11 )
   END_RUNG wire#w2
   RUNG wire#powerrail
      Contact( #Mx_ET12 )
   END_RUNG wire#w2
   RUNG wire#w3
      I_Contact( #AVTF_MAnt_Mx_BGrande )
      I_Contact( #Entrando_BGrande )
   END_RUNG wire#w1
   RUNG wire#powerrail
      Contact( #Mx_ET13 )
      wire#w4
      Contact( #TR1_Abajo )
      Contact( #TR2_Abajo )
   END_RUNG wire#w1
   RUNG wire#powerrail
      Contact( #Mx_ET14 )
   END_RUNG wire#w4
   RUNG wire#powerrail
      Contact( #Mx_ET15 )
   END_RUNG wire#w4
   RUNG wire#powerrail
      Contact( #Mx_ET09 )
   END_RUNG wire#w4
   RUNG wire#powerrail
      I_Contact( #pHsMx_1 )
      I_Contact( #OrdSal_S01 )
      I_Contact( #OrdSal_S03 )
      Not()
      Contact( #Mx_ET02 )
      Contact( #TR1_Abajo )
      Contact( #TR2_Abajo )
   END_RUNG wire#w1
   RUNG wire#powerrail
      I_Contact( #pHsMx_1 )
      I_Contact( #OrdSal_S01 )
      I_Contact( #OrdSal_S03 )
      Contact( #Mx_ET02 )
      Contact( #TR1_Arriba )
      Contact( #TR2_Abajo )
   END_RUNG wire#w1
   RUNG wire#powerrail
      Contact( #Mx_ET50 )
      wire#w5
      Contact( #TR1_Abajo )
      Contact( #TR2_Abajo )
   END_RUNG wire#w1
   RUNG wire#powerrail
      Contact( #Mx_ET51 )
   END_RUNG wire#w5
   RUNG wire#powerrail
      Contact( #Mx_ET250 )
   END_RUNG wire#w5
   RUNG wire#powerrail
      Contact( #Mx_ET251 )
   END_RUNG wire#w5
   RUNG wire#powerrail
      Contact( #Mx_ET60 )
      wire#w6
      Contact( #TR1_Abajo )
      Contact( #TR2_Abajo )
   END_RUNG wire#w1
   RUNG wire#powerrail
      Contact( #Mx_ET61 )
   END_RUNG wire#w6
   RUNG wire#powerrail
      Contact( #Mx_ET260 )
   END_RUNG wire#w6
   RUNG wire#powerrail
      Contact( #Mx_ET261 )
   END_RUNG wire#w6
   RUNG wire#powerrail
      Contact( #Activado_Pasarela )
      Contact( #TR1_Arriba )
      wire#w8
      Contact( #TR2_Arriba )
   END_RUNG wire#w7
   RUNG wire#w8
      Contact( #AVTF_MAnt_MSig_BPequena )
   END_RUNG wire#w7
   // the same network as SCL:
   #Pos_TROK := (((#Mx_ET01 AND #TR1_Arriba AND #TR2_Arriba AND "ON") OR ((#Mx_ET10 OR #Mx_ET11 OR #Mx_ET12) AND #TR1_Arriba AND ((#TR2_Arriba AND #Entrando_BGrande) OR (NOT #AVTF_MAnt_Mx_BGrande AND NOT #Entrando_BGrande))) OR ((#Mx_ET13 OR #Mx_ET14 OR #Mx_ET15 OR #Mx_ET09) AND #TR1_Abajo AND #TR2_Abajo) OR (NOT (NOT #pHsMx_1 AND NOT #OrdSal_S01 AND NOT #OrdSal_S03) AND #Mx_ET02 AND #TR1_Abajo AND #TR2_Abajo) OR (NOT #pHsMx_1 AND NOT #OrdSal_S01 AND NOT #OrdSal_S03 AND #Mx_ET02 AND #TR1_Arriba AND #TR2_Abajo) OR ((#Mx_ET50 OR #Mx_ET51 OR #Mx_ET250 OR #Mx_ET251) AND #TR1_Abajo AND #TR2_Abajo) OR ((#Mx_ET60 OR #Mx_ET61 OR #Mx_ET260 OR #Mx_ET261) AND #TR1_Abajo AND #TR2_Abajo)) AND NOT #Activado_Pasarela) OR (#Activado_Pasarela AND #TR1_Arriba AND (#TR2_Arriba OR #AVTF_MAnt_MSig_BPequena));
END_REGION

REGION Network 81: VARIABLES AUXILIARES - Posición Correcta de los Topes
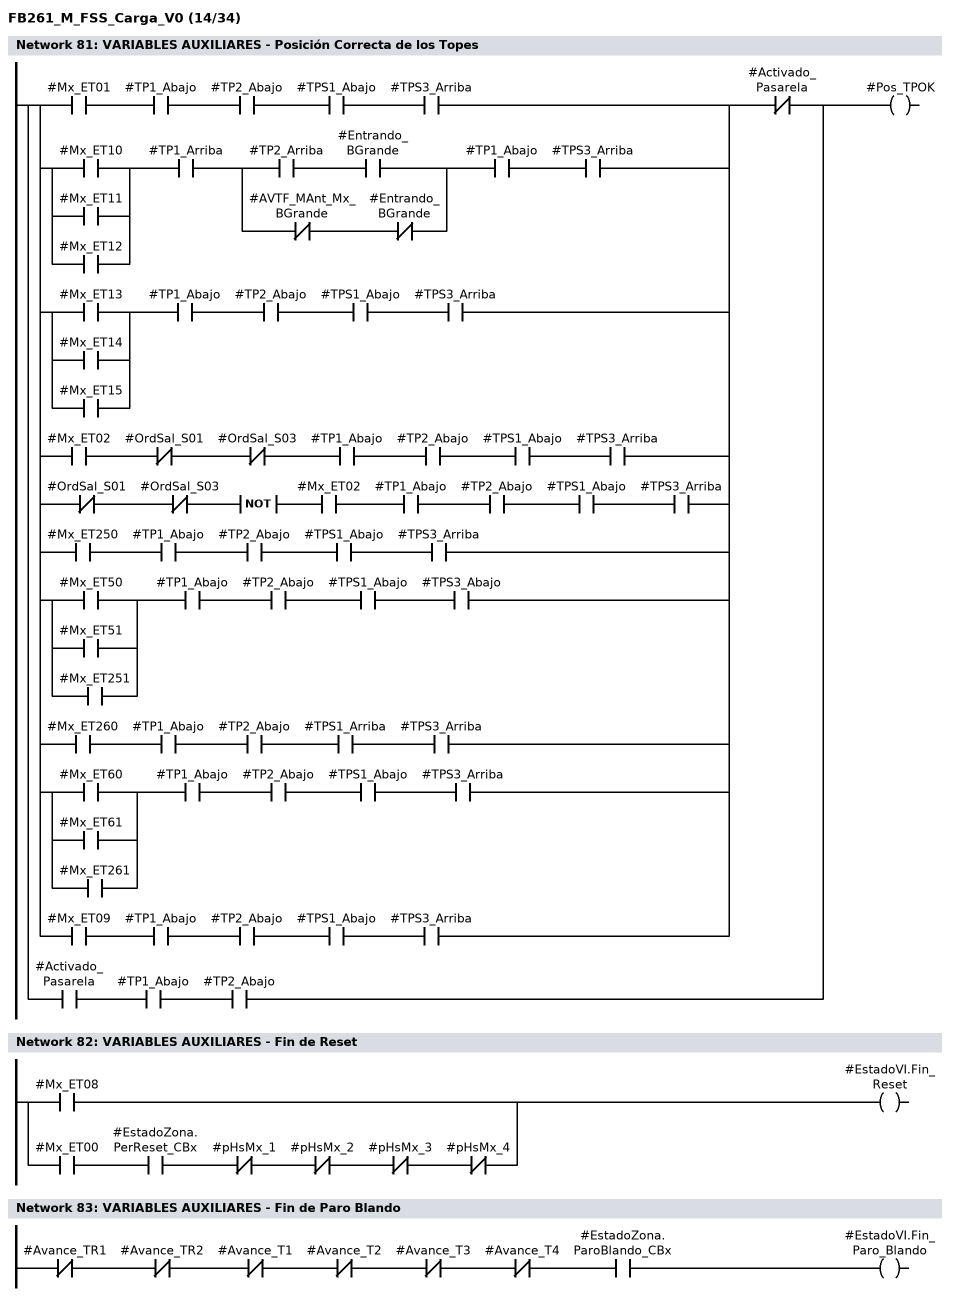
   RUNG wire#powerrail
      Contact( #Mx_ET01 )
      Contact( #TP1_Abajo )
      Contact( #TP2_Abajo )
      Contact( #TPS1_Abajo )
      Contact( #TPS3_Arriba )
      wire#w1
      I_Contact( #Activado_Pasarela )
      wire#w8
      Coil( #Pos_TPOK )
   END_RUNG
   RUNG wire#powerrail
      Contact( #Mx_ET10 )
      wire#w2
      Contact( #TP1_Arriba )
      wire#w3
      Contact( #TP2_Arriba )
      Contact( #Entrando_BGrande )
      wire#w4
      Contact( #TP1_Abajo )
      Contact( #TPS3_Arriba )
   END_RUNG wire#w1
   RUNG wire#powerrail
      Contact( #Mx_ET11 )
   END_RUNG wire#w2
   RUNG wire#powerrail
      Contact( #Mx_ET12 )
   END_RUNG wire#w2
   RUNG wire#w3
      I_Contact( #AVTF_MAnt_Mx_BGrande )
      I_Contact( #Entrando_BGrande )
   END_RUNG wire#w4
   RUNG wire#powerrail
      Contact( #Mx_ET13 )
      wire#w5
      Contact( #TP1_Abajo )
      Contact( #TP2_Abajo )
      Contact( #TPS1_Abajo )
      Contact( #TPS3_Arriba )
   END_RUNG wire#w1
   RUNG wire#powerrail
      Contact( #Mx_ET14 )
   END_RUNG wire#w5
   RUNG wire#powerrail
      Contact( #Mx_ET15 )
   END_RUNG wire#w5
   RUNG wire#powerrail
      Contact( #Mx_ET02 )
      I_Contact( #OrdSal_S01 )
      I_Contact( #OrdSal_S03 )
      Contact( #TP1_Abajo )
      Contact( #TP2_Abajo )
      Contact( #TPS1_Abajo )
      Contact( #TPS3_Arriba )
   END_RUNG wire#w1
   RUNG wire#powerrail
      I_Contact( #OrdSal_S01 )
      I_Contact( #OrdSal_S03 )
      Not()
      Contact( #Mx_ET02 )
      Contact( #TP1_Abajo )
      Contact( #TP2_Abajo )
      Contact( #TPS1_Abajo )
      Contact( #TPS3_Arriba )
   END_RUNG wire#w1
   RUNG wire#powerrail
      Contact( #Mx_ET250 )
      Contact( #TP1_Abajo )
      Contact( #TP2_Abajo )
      Contact( #TPS1_Abajo )
      Contact( #TPS3_Arriba )
   END_RUNG wire#w1
   RUNG wire#powerrail
      Contact( #Mx_ET50 )
      wire#w6
      Contact( #TP1_Abajo )
      Contact( #TP2_Abajo )
      Contact( #TPS1_Abajo )
      Contact( #TPS3_Abajo )
   END_RUNG wire#w1
   RUNG wire#powerrail
      Contact( #Mx_ET51 )
   END_RUNG wire#w6
   RUNG wire#powerrail
      Contact( #Mx_ET251 )
   END_RUNG wire#w6
   RUNG wire#powerrail
      Contact( #Mx_ET260 )
      Contact( #TP1_Abajo )
      Contact( #TP2_Abajo )
      Contact( #TPS1_Arriba )
      Contact( #TPS3_Arriba )
   END_RUNG wire#w1
   RUNG wire#powerrail
      Contact( #Mx_ET60 )
      wire#w7
      Contact( #TP1_Abajo )
      Contact( #TP2_Abajo )
      Contact( #TPS1_Abajo )
      Contact( #TPS3_Arriba )
   END_RUNG wire#w1
   RUNG wire#powerrail
      Contact( #Mx_ET61 )
   END_RUNG wire#w7
   RUNG wire#powerrail
      Contact( #Mx_ET261 )
   END_RUNG wire#w7
   RUNG wire#powerrail
      Contact( #Mx_ET09 )
      Contact( #TP1_Abajo )
      Contact( #TP2_Abajo )
      Contact( #TPS1_Abajo )
      Contact( #TPS3_Arriba )
   END_RUNG wire#w1
   RUNG wire#powerrail
      Contact( #Activado_Pasarela )
      Contact( #TP1_Abajo )
      Contact( #TP2_Abajo )
   END_RUNG wire#w8
   // the same network as SCL:
   #Pos_TPOK := (((#Mx_ET01 AND #TP1_Abajo AND #TP2_Abajo AND #TPS1_Abajo AND #TPS3_Arriba) OR ((#Mx_ET10 OR #Mx_ET11 OR #Mx_ET12) AND #TP1_Arriba AND ((#TP2_Arriba AND #Entrando_BGrande) OR (NOT #AVTF_MAnt_Mx_BGrande AND NOT #Entrando_BGrande)) AND #TP1_Abajo AND #TPS3_Arriba) OR ((#Mx_ET13 OR #Mx_ET14 OR #Mx_ET15) AND #TP1_Abajo AND #TP2_Abajo AND #TPS1_Abajo AND #TPS3_Arriba) OR (#Mx_ET02 AND NOT #OrdSal_S01 AND NOT #OrdSal_S03 AND #TP1_Abajo AND #TP2_Abajo AND #TPS1_Abajo AND #TPS3_Arriba) OR (NOT (NOT #OrdSal_S01 AND NOT #OrdSal_S03) AND #Mx_ET02 AND #TP1_Abajo AND #TP2_Abajo AND #TPS1_Abajo AND #TPS3_Arriba) OR (#Mx_ET250 AND #TP1_Abajo AND #TP2_Abajo AND #TPS1_Abajo AND #TPS3_Arriba) OR ((#Mx_ET50 OR #Mx_ET51 OR #Mx_ET251) AND #TP1_Abajo AND #TP2_Abajo AND #TPS1_Abajo AND #TPS3_Abajo) OR (#Mx_ET260 AND #TP1_Abajo AND #TP2_Abajo AND #TPS1_Arriba AND #TPS3_Arriba) OR ((#Mx_ET60 OR #Mx_ET61 OR #Mx_ET261) AND #TP1_Abajo AND #TP2_Abajo AND #TPS1_Abajo AND #TPS3_Arriba) OR (#Mx_ET09 AND #TP1_Abajo AND #TP2_Abajo AND #TPS1_Abajo AND #TPS3_Arriba)) AND NOT #Activado_Pasarela) OR (#Activado_Pasarela AND #TP1_Abajo AND #TP2_Abajo);
END_REGION

REGION Network 82: VARIABLES AUXILIARES - Fin de Reset
   RUNG wire#powerrail
      Contact( #Mx_ET08 )
      wire#w1
      Coil( #EstadoVI.Fin_Reset )
   END_RUNG
   RUNG wire#powerrail
      Contact( #Mx_ET00 )
      Contact( #EstadoZona.PerReset_CBx )
      I_Contact( #pHsMx_1 )
      I_Contact( #pHsMx_2 )
      I_Contact( #pHsMx_3 )
      I_Contact( #pHsMx_4 )
   END_RUNG wire#w1
   // the same network as SCL:
   #EstadoVI.Fin_Reset := #Mx_ET08 OR (#Mx_ET00 AND #EstadoZona.PerReset_CBx AND NOT #pHsMx_1 AND NOT #pHsMx_2 AND NOT #pHsMx_3 AND NOT #pHsMx_4);
END_REGION

REGION Network 83: VARIABLES AUXILIARES - Fin de Paro Blando
   RUNG wire#powerrail
      I_Contact( #Avance_TR1 )
      I_Contact( #Avance_TR2 )
      I_Contact( #Avance_T1 )
      I_Contact( #Avance_T2 )
      I_Contact( #Avance_T3 )
      I_Contact( #Avance_T4 )
      Contact( #EstadoZona.ParoBlando_CBx )
      Coil( #EstadoVI.Fin_Paro_Blando )
   END_RUNG
   // the same network as SCL:
   #EstadoVI.Fin_Paro_Blando := NOT #Avance_TR1 AND NOT #Avance_TR2 AND NOT #Avance_T1 AND NOT #Avance_T2 AND NOT #Avance_T3 AND NOT #Avance_T4 AND #EstadoZona.ParoBlando_CBx;
END_REGION

REGION Network 84: VARIABLES AUXILIARES - Permiso de Entrada - PTF_MAnt_Mx
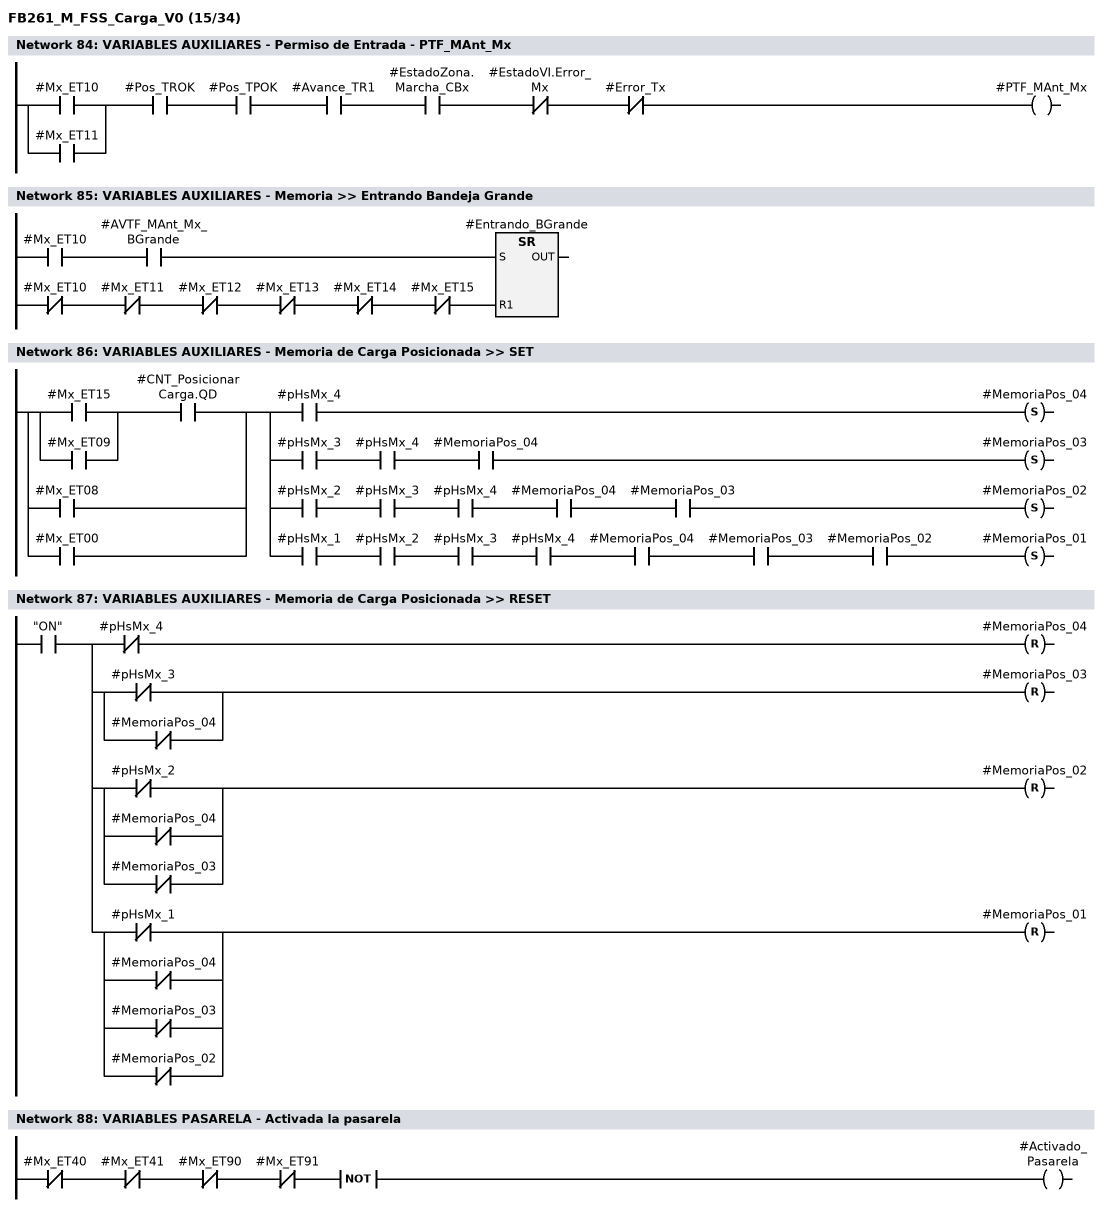
   RUNG wire#powerrail
      Contact( #Mx_ET10 )
      wire#w1
      Contact( #Pos_TROK )
      Contact( #Pos_TPOK )
      Contact( #Avance_TR1 )
      Contact( #EstadoZona.Marcha_CBx )
      I_Contact( #EstadoVI.Error_Mx )
      I_Contact( #Error_Tx )
      Coil( #PTF_MAnt_Mx )
   END_RUNG
   RUNG wire#powerrail
      Contact( #Mx_ET11 )
   END_RUNG wire#w1
   // the same network as SCL:
   #PTF_MAnt_Mx := (#Mx_ET10 OR #Mx_ET11) AND #Pos_TROK AND #Pos_TPOK AND #Avance_TR1 AND #EstadoZona.Marcha_CBx AND NOT #EstadoVI.Error_Mx AND NOT #Error_Tx;
END_REGION

REGION Network 85: VARIABLES AUXILIARES - Memoria >> Entrando Bandeja Grande
   RUNG wire#powerrail
      Contact( #Mx_ET10 )
      Contact( #AVTF_MAnt_Mx_BGrande )
      S_SR(operand := #Entrando_BGrande, r1 := wire#w1)
   END_RUNG
   RUNG wire#powerrail
      I_Contact( #Mx_ET10 )
      I_Contact( #Mx_ET11 )
      I_Contact( #Mx_ET12 )
      I_Contact( #Mx_ET13 )
      I_Contact( #Mx_ET14 )
      I_Contact( #Mx_ET15 )
   END_RUNG wire#w1
   // the same network as SCL:
   IF #Mx_ET10 AND #AVTF_MAnt_Mx_BGrande THEN
       #Entrando_BGrande := TRUE;   // SR flip-flop
   END_IF;
   IF NOT #Mx_ET10 AND NOT #Mx_ET11 AND NOT #Mx_ET12 AND NOT #Mx_ET13 AND NOT #Mx_ET14 AND NOT #Mx_ET15 THEN
       #Entrando_BGrande := FALSE;
   END_IF;
END_REGION

REGION Network 86: VARIABLES AUXILIARES - Memoria de Carga Posicionada >> SET
   RUNG wire#powerrail
      Contact( #Mx_ET15 )
      wire#w1
      Contact( #CNT_PosicionarCarga.QD )
      wire#w2
      Contact( #pHsMx_4 )
      S_Coil( #MemoriaPos_04 )
   END_RUNG
   RUNG wire#powerrail
      Contact( #Mx_ET09 )
   END_RUNG wire#w1
   RUNG wire#powerrail
      Contact( #Mx_ET08 )
   END_RUNG wire#w2
   RUNG wire#powerrail
      Contact( #Mx_ET00 )
   END_RUNG wire#w2
   RUNG wire#w2
      Contact( #pHsMx_3 )
      Contact( #pHsMx_4 )
      Contact( #MemoriaPos_04 )
      S_Coil( #MemoriaPos_03 )
   END_RUNG
   RUNG wire#w2
      Contact( #pHsMx_2 )
      Contact( #pHsMx_3 )
      Contact( #pHsMx_4 )
      Contact( #MemoriaPos_04 )
      Contact( #MemoriaPos_03 )
      S_Coil( #MemoriaPos_02 )
   END_RUNG
   RUNG wire#w2
      Contact( #pHsMx_1 )
      Contact( #pHsMx_2 )
      Contact( #pHsMx_3 )
      Contact( #pHsMx_4 )
      Contact( #MemoriaPos_04 )
      Contact( #MemoriaPos_03 )
      Contact( #MemoriaPos_02 )
      S_Coil( #MemoriaPos_01 )
   END_RUNG
   // the same network as SCL:
   #_w1 := ((#Mx_ET15 OR #Mx_ET09) AND #CNT_PosicionarCarga.QD) OR #Mx_ET08 OR #Mx_ET00;
   IF #_w1 AND #pHsMx_4 THEN #MemoriaPos_04 := TRUE; END_IF;
   IF #_w1 AND #pHsMx_3 AND #pHsMx_4 AND #MemoriaPos_04 THEN #MemoriaPos_03 := TRUE; END_IF;
   IF #_w1 AND #pHsMx_2 AND #pHsMx_3 AND #pHsMx_4 AND #MemoriaPos_04 AND #MemoriaPos_03 THEN
       #MemoriaPos_02 := TRUE;
   END_IF;
   IF #_w1 AND #pHsMx_1 AND #pHsMx_2 AND #pHsMx_3 AND #pHsMx_4 AND #MemoriaPos_04 AND #MemoriaPos_03 AND #MemoriaPos_02 THEN
       #MemoriaPos_01 := TRUE;
   END_IF;
END_REGION

REGION Network 87: VARIABLES AUXILIARES - Memoria de Carga Posicionada >> RESET
   RUNG wire#powerrail
      Contact( "ON" )
      wire#w1
      I_Contact( #pHsMx_4 )
      R_Coil( #MemoriaPos_04 )
   END_RUNG
   RUNG wire#w1
      I_Contact( #pHsMx_3 )
      wire#w2
      R_Coil( #MemoriaPos_03 )
   END_RUNG
   RUNG wire#w1
      I_Contact( #MemoriaPos_04 )
   END_RUNG wire#w2
   RUNG wire#w1
      I_Contact( #pHsMx_2 )
      wire#w3
      R_Coil( #MemoriaPos_02 )
   END_RUNG
   RUNG wire#w1
      I_Contact( #MemoriaPos_04 )
   END_RUNG wire#w3
   RUNG wire#w1
      I_Contact( #MemoriaPos_03 )
   END_RUNG wire#w3
   RUNG wire#w1
      I_Contact( #pHsMx_1 )
      wire#w4
      R_Coil( #MemoriaPos_01 )
   END_RUNG
   RUNG wire#w1
      I_Contact( #MemoriaPos_04 )
   END_RUNG wire#w4
   RUNG wire#w1
      I_Contact( #MemoriaPos_03 )
   END_RUNG wire#w4
   RUNG wire#w1
      I_Contact( #MemoriaPos_02 )
   END_RUNG wire#w4
   // the same network as SCL:
   IF "ON" AND NOT #pHsMx_4 THEN #MemoriaPos_04 := FALSE; END_IF;
   IF "ON" AND (NOT #pHsMx_3 OR NOT #MemoriaPos_04) THEN #MemoriaPos_03 := FALSE; END_IF;
   IF "ON" AND (NOT #pHsMx_2 OR NOT #MemoriaPos_04 OR NOT #MemoriaPos_03) THEN
       #MemoriaPos_02 := FALSE;
   END_IF;
   IF "ON" AND (NOT #pHsMx_1 OR NOT #MemoriaPos_04 OR NOT #MemoriaPos_03 OR NOT #MemoriaPos_02) THEN
       #MemoriaPos_01 := FALSE;
   END_IF;
END_REGION

REGION Network 88: VARIABLES PASARELA - Activada la pasarela
   RUNG wire#powerrail
      I_Contact( #Mx_ET40 )
      I_Contact( #Mx_ET41 )
      I_Contact( #Mx_ET90 )
      I_Contact( #Mx_ET91 )
      Not()
      Coil( #Activado_Pasarela )
   END_RUNG
   // the same network as SCL:
   #Activado_Pasarela := NOT (NOT #Mx_ET40 AND NOT #Mx_ET41 AND NOT #Mx_ET90 AND NOT #Mx_ET91);
END_REGION

REGION Network 89: CONTADOR DE PRESENCIA EN PASARELA - CENTRADO DE LA CARGA >>> CNT_PresenciaPasarela
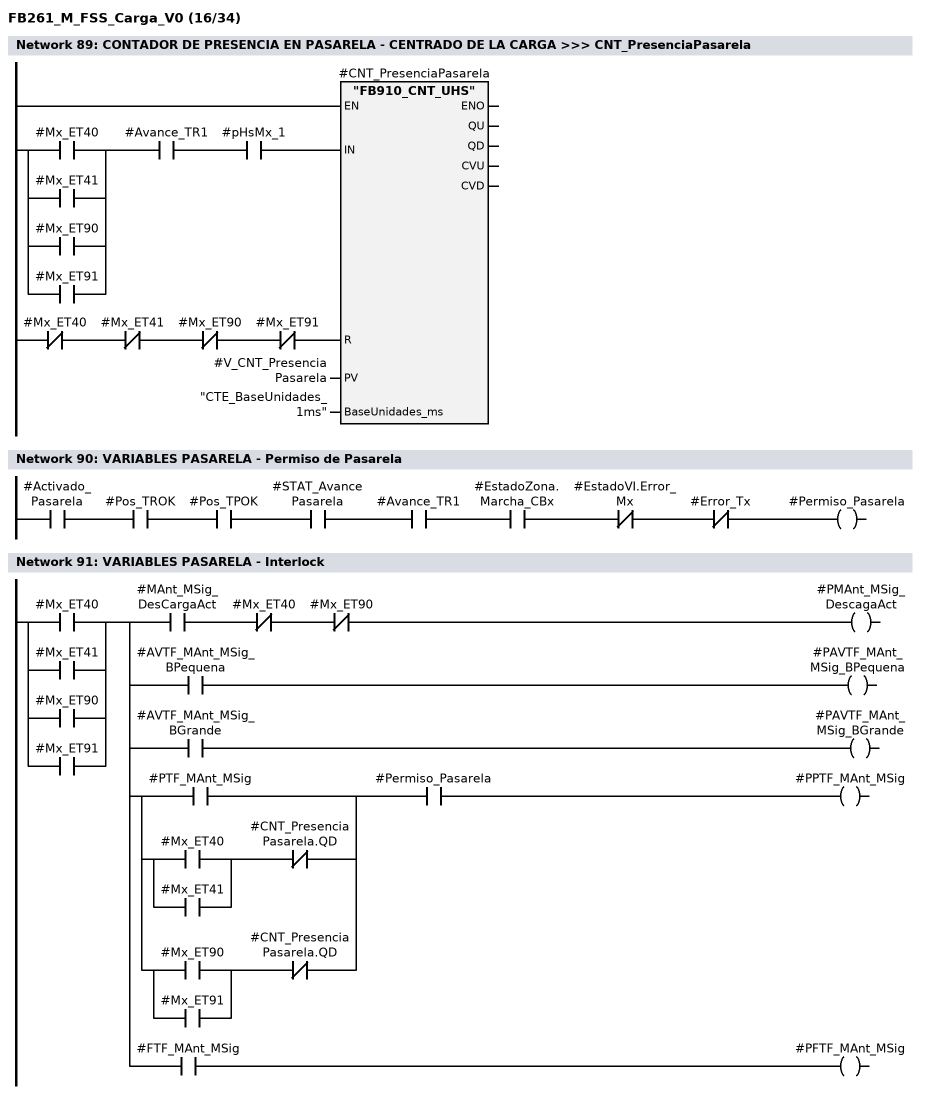
   RUNG wire#powerrail
      #CNT_PresenciaPasarela(IN := wire#w2, R := wire#w3, PV := #V_CNT_PresenciaPasarela, BaseUnidades_ms := "CTE_BaseUnidades_1ms", QU =>, QD =>, CVU =>, CVD =>)
   END_RUNG
   RUNG wire#powerrail
      Contact( #Mx_ET40 )
      wire#w1
      Contact( #Avance_TR1 )
      Contact( #pHsMx_1 )
   END_RUNG wire#w2
   RUNG wire#powerrail
      Contact( #Mx_ET41 )
   END_RUNG wire#w1
   RUNG wire#powerrail
      Contact( #Mx_ET90 )
   END_RUNG wire#w1
   RUNG wire#powerrail
      Contact( #Mx_ET91 )
   END_RUNG wire#w1
   RUNG wire#powerrail
      I_Contact( #Mx_ET40 )
      I_Contact( #Mx_ET41 )
      I_Contact( #Mx_ET90 )
      I_Contact( #Mx_ET91 )
   END_RUNG wire#w3
   // the same network as SCL:
   #CNT_PresenciaPasarela(IN := (#Mx_ET40 OR #Mx_ET41 OR #Mx_ET90 OR #Mx_ET91) AND #Avance_TR1 AND #pHsMx_1,   // "FB910_CNT_UHS"
                          R := NOT #Mx_ET40 AND NOT #Mx_ET41 AND NOT #Mx_ET90 AND NOT #Mx_ET91,
                          PV := #V_CNT_PresenciaPasarela,
                          BaseUnidades_ms := "CTE_BaseUnidades_1ms");
END_REGION

REGION Network 90: VARIABLES PASARELA - Permiso de Pasarela
   RUNG wire#powerrail
      Contact( #Activado_Pasarela )
      Contact( #Pos_TROK )
      Contact( #Pos_TPOK )
      Contact( #STAT_AvancePasarela )
      Contact( #Avance_TR1 )
      Contact( #EstadoZona.Marcha_CBx )
      I_Contact( #EstadoVI.Error_Mx )
      I_Contact( #Error_Tx )
      Coil( #Permiso_Pasarela )
   END_RUNG
   // the same network as SCL:
   #Permiso_Pasarela := #Activado_Pasarela AND #Pos_TROK AND #Pos_TPOK AND #STAT_AvancePasarela AND #Avance_TR1 AND #EstadoZona.Marcha_CBx AND NOT #EstadoVI.Error_Mx AND NOT #Error_Tx;
END_REGION

REGION Network 91: VARIABLES PASARELA - Interlock
   RUNG wire#powerrail
      Contact( #Mx_ET40 )
      wire#w1
      Contact( #MAnt_MSig_DesCargaAct )
      I_Contact( #Mx_ET40 )
      I_Contact( #Mx_ET90 )
      Coil( #PMAnt_MSig_DescagaAct )
   END_RUNG
   RUNG wire#powerrail
      Contact( #Mx_ET41 )
   END_RUNG wire#w1
   RUNG wire#powerrail
      Contact( #Mx_ET90 )
   END_RUNG wire#w1
   RUNG wire#powerrail
      Contact( #Mx_ET91 )
   END_RUNG wire#w1
   RUNG wire#w1
      Contact( #AVTF_MAnt_MSig_BPequena )
      Coil( #PAVTF_MAnt_MSig_BPequena )
   END_RUNG
   RUNG wire#w1
      Contact( #AVTF_MAnt_MSig_BGrande )
      Coil( #PAVTF_MAnt_MSig_BGrande )
   END_RUNG
   RUNG wire#w1
      Contact( #PTF_MAnt_MSig )
      wire#w2
      Contact( #Permiso_Pasarela )
      Coil( #PPTF_MAnt_MSig )
   END_RUNG
   RUNG wire#w1
      Contact( #Mx_ET40 )
      wire#w3
      I_Contact( #CNT_PresenciaPasarela.QD )
   END_RUNG wire#w2
   RUNG wire#w1
      Contact( #Mx_ET41 )
   END_RUNG wire#w3
   RUNG wire#w1
      Contact( #Mx_ET90 )
      wire#w4
      I_Contact( #CNT_PresenciaPasarela.QD )
   END_RUNG wire#w2
   RUNG wire#w1
      Contact( #Mx_ET91 )
   END_RUNG wire#w4
   RUNG wire#w1
      Contact( #FTF_MAnt_MSig )
      Coil( #PFTF_MAnt_MSig )
   END_RUNG
   // the same network as SCL:
   #_w1 := #Mx_ET40 OR #Mx_ET41 OR #Mx_ET90 OR #Mx_ET91;
   #PMAnt_MSig_DescagaAct := #_w1 AND #MAnt_MSig_DesCargaAct AND NOT #Mx_ET40 AND NOT #Mx_ET90;
   #PAVTF_MAnt_MSig_BPequena := #_w1 AND #AVTF_MAnt_MSig_BPequena;
   #PAVTF_MAnt_MSig_BGrande := #_w1 AND #AVTF_MAnt_MSig_BGrande;
   #PPTF_MAnt_MSig := #_w1 AND (#PTF_MAnt_MSig OR ((#Mx_ET40 OR #Mx_ET41) AND NOT #CNT_PresenciaPasarela.QD) OR ((#Mx_ET90 OR #Mx_ET91) AND NOT #CNT_PresenciaPasarela.QD)) AND #Permiso_Pasarela;
   #PFTF_MAnt_MSig := #_w1 AND #FTF_MAnt_MSig;
END_REGION

REGION Network 92: MENSAJES - PRESENCIA
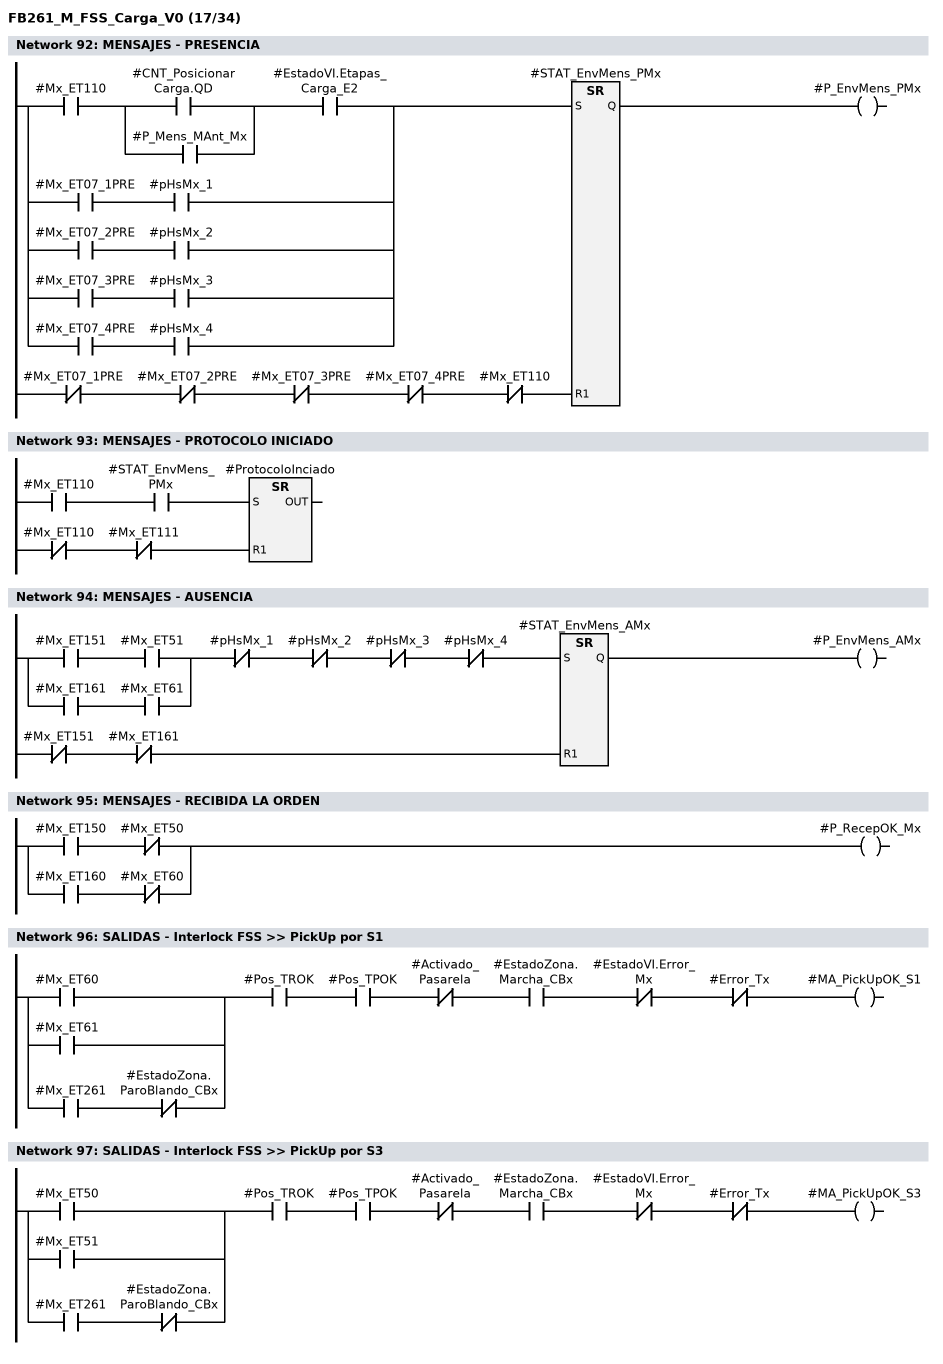
   RUNG wire#powerrail
      Contact( #Mx_ET110 )
      wire#w1
      Contact( #CNT_PosicionarCarga.QD )
      wire#w2
      Contact( #EstadoVI.Etapas_Carga_E2 )
      wire#w3
      S_SR(operand := #STAT_EnvMens_PMx, r1 := wire#w4)
      Coil( #P_EnvMens_PMx )
   END_RUNG
   RUNG wire#w1
      Contact( #P_Mens_MAnt_Mx )
   END_RUNG wire#w2
   RUNG wire#powerrail
      Contact( #Mx_ET07_1PRE )
      Contact( #pHsMx_1 )
   END_RUNG wire#w3
   RUNG wire#powerrail
      Contact( #Mx_ET07_2PRE )
      Contact( #pHsMx_2 )
   END_RUNG wire#w3
   RUNG wire#powerrail
      Contact( #Mx_ET07_3PRE )
      Contact( #pHsMx_3 )
   END_RUNG wire#w3
   RUNG wire#powerrail
      Contact( #Mx_ET07_4PRE )
      Contact( #pHsMx_4 )
   END_RUNG wire#w3
   RUNG wire#powerrail
      I_Contact( #Mx_ET07_1PRE )
      I_Contact( #Mx_ET07_2PRE )
      I_Contact( #Mx_ET07_3PRE )
      I_Contact( #Mx_ET07_4PRE )
      I_Contact( #Mx_ET110 )
   END_RUNG wire#w4
   // the same network as SCL:
   IF (#Mx_ET110 AND (#CNT_PosicionarCarga.QD OR #P_Mens_MAnt_Mx) AND #EstadoVI.Etapas_Carga_E2) OR (#Mx_ET07_1PRE AND #pHsMx_1) OR (#Mx_ET07_2PRE AND #pHsMx_2) OR (#Mx_ET07_3PRE AND #pHsMx_3) OR (#Mx_ET07_4PRE AND #pHsMx_4) THEN
       #STAT_EnvMens_PMx := TRUE;   // SR flip-flop
   END_IF;
   IF NOT #Mx_ET07_1PRE AND NOT #Mx_ET07_2PRE AND NOT #Mx_ET07_3PRE AND NOT #Mx_ET07_4PRE AND NOT #Mx_ET110 THEN
       #STAT_EnvMens_PMx := FALSE;
   END_IF;
   #P_EnvMens_PMx := #STAT_EnvMens_PMx;
END_REGION

REGION Network 93: MENSAJES - PROTOCOLO INICIADO
   RUNG wire#powerrail
      Contact( #Mx_ET110 )
      Contact( #STAT_EnvMens_PMx )
      S_SR(operand := #ProtocoloInciado, r1 := wire#w1)
   END_RUNG
   RUNG wire#powerrail
      I_Contact( #Mx_ET110 )
      I_Contact( #Mx_ET111 )
   END_RUNG wire#w1
   // the same network as SCL:
   IF #Mx_ET110 AND #STAT_EnvMens_PMx THEN
       #ProtocoloInciado := TRUE;   // SR flip-flop
   END_IF;
   IF NOT #Mx_ET110 AND NOT #Mx_ET111 THEN #ProtocoloInciado := FALSE; END_IF;
END_REGION

REGION Network 94: MENSAJES - AUSENCIA
   RUNG wire#powerrail
      Contact( #Mx_ET151 )
      Contact( #Mx_ET51 )
      wire#w1
      I_Contact( #pHsMx_1 )
      I_Contact( #pHsMx_2 )
      I_Contact( #pHsMx_3 )
      I_Contact( #pHsMx_4 )
      S_SR(operand := #STAT_EnvMens_AMx, r1 := wire#w2)
      Coil( #P_EnvMens_AMx )
   END_RUNG
   RUNG wire#powerrail
      Contact( #Mx_ET161 )
      Contact( #Mx_ET61 )
   END_RUNG wire#w1
   RUNG wire#powerrail
      I_Contact( #Mx_ET151 )
      I_Contact( #Mx_ET161 )
   END_RUNG wire#w2
   // the same network as SCL:
   IF ((#Mx_ET151 AND #Mx_ET51) OR (#Mx_ET161 AND #Mx_ET61)) AND NOT #pHsMx_1 AND NOT #pHsMx_2 AND NOT #pHsMx_3 AND NOT #pHsMx_4 THEN
       #STAT_EnvMens_AMx := TRUE;   // SR flip-flop
   END_IF;
   IF NOT #Mx_ET151 AND NOT #Mx_ET161 THEN #STAT_EnvMens_AMx := FALSE; END_IF;
   #P_EnvMens_AMx := #STAT_EnvMens_AMx;
END_REGION

REGION Network 95: MENSAJES - RECIBIDA LA ORDEN
   RUNG wire#powerrail
      Contact( #Mx_ET150 )
      I_Contact( #Mx_ET50 )
      wire#w1
      Coil( #P_RecepOK_Mx )
   END_RUNG
   RUNG wire#powerrail
      Contact( #Mx_ET160 )
      I_Contact( #Mx_ET60 )
   END_RUNG wire#w1
   // the same network as SCL:
   #P_RecepOK_Mx := (#Mx_ET150 AND NOT #Mx_ET50) OR (#Mx_ET160 AND NOT #Mx_ET60);
END_REGION

REGION Network 96: SALIDAS - Interlock FSS >> PickUp por S1
   RUNG wire#powerrail
      Contact( #Mx_ET60 )
      wire#w1
      Contact( #Pos_TROK )
      Contact( #Pos_TPOK )
      I_Contact( #Activado_Pasarela )
      Contact( #EstadoZona.Marcha_CBx )
      I_Contact( #EstadoVI.Error_Mx )
      I_Contact( #Error_Tx )
      Coil( #MA_PickUpOK_S1 )
   END_RUNG
   RUNG wire#powerrail
      Contact( #Mx_ET61 )
   END_RUNG wire#w1
   RUNG wire#powerrail
      Contact( #Mx_ET261 )
      I_Contact( #EstadoZona.ParoBlando_CBx )
   END_RUNG wire#w1
   // the same network as SCL:
   #MA_PickUpOK_S1 := (#Mx_ET60 OR #Mx_ET61 OR (#Mx_ET261 AND NOT #EstadoZona.ParoBlando_CBx)) AND #Pos_TROK AND #Pos_TPOK AND NOT #Activado_Pasarela AND #EstadoZona.Marcha_CBx AND NOT #EstadoVI.Error_Mx AND NOT #Error_Tx;
END_REGION

REGION Network 97: SALIDAS - Interlock FSS >> PickUp por S3
   RUNG wire#powerrail
      Contact( #Mx_ET50 )
      wire#w1
      Contact( #Pos_TROK )
      Contact( #Pos_TPOK )
      I_Contact( #Activado_Pasarela )
      Contact( #EstadoZona.Marcha_CBx )
      I_Contact( #EstadoVI.Error_Mx )
      I_Contact( #Error_Tx )
      Coil( #MA_PickUpOK_S3 )
   END_RUNG
   RUNG wire#powerrail
      Contact( #Mx_ET51 )
   END_RUNG wire#w1
   RUNG wire#powerrail
      Contact( #Mx_ET261 )
      I_Contact( #EstadoZona.ParoBlando_CBx )
   END_RUNG wire#w1
   // the same network as SCL:
   #MA_PickUpOK_S3 := (#Mx_ET50 OR #Mx_ET51 OR (#Mx_ET261 AND NOT #EstadoZona.ParoBlando_CBx)) AND #Pos_TROK AND #Pos_TPOK AND NOT #Activado_Pasarela AND #EstadoZona.Marcha_CBx AND NOT #EstadoVI.Error_Mx AND NOT #Error_Tx;
END_REGION

REGION Network 98: VARIABLES INTERNAS - AVANCE DE CARGA
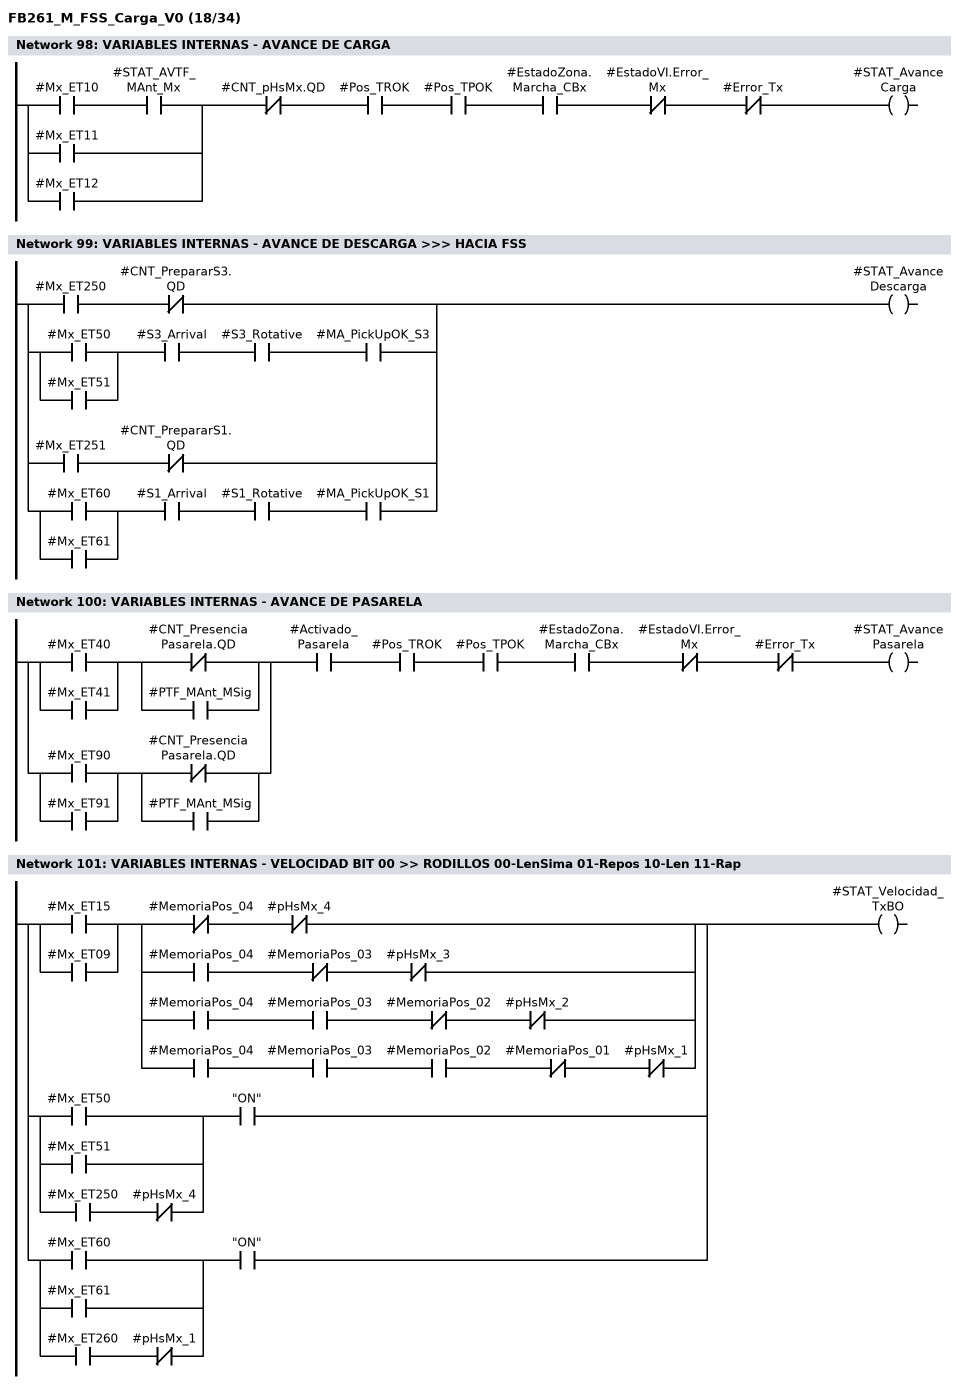
   RUNG wire#powerrail
      Contact( #Mx_ET10 )
      Contact( #STAT_AVTF_MAnt_Mx )
      wire#w1
      I_Contact( #CNT_pHsMx.QD )
      Contact( #Pos_TROK )
      Contact( #Pos_TPOK )
      Contact( #EstadoZona.Marcha_CBx )
      I_Contact( #EstadoVI.Error_Mx )
      I_Contact( #Error_Tx )
      Coil( #STAT_AvanceCarga )
   END_RUNG
   RUNG wire#powerrail
      Contact( #Mx_ET11 )
   END_RUNG wire#w1
   RUNG wire#powerrail
      Contact( #Mx_ET12 )
   END_RUNG wire#w1
   // the same network as SCL:
   #STAT_AvanceCarga := ((#Mx_ET10 AND #STAT_AVTF_MAnt_Mx) OR #Mx_ET11 OR #Mx_ET12) AND NOT #CNT_pHsMx.QD AND #Pos_TROK AND #Pos_TPOK AND #EstadoZona.Marcha_CBx AND NOT #EstadoVI.Error_Mx AND NOT #Error_Tx;
END_REGION

REGION Network 99: VARIABLES INTERNAS - AVANCE DE DESCARGA >>> HACIA FSS
   RUNG wire#powerrail
      Contact( #Mx_ET250 )
      I_Contact( #CNT_PrepararS3.QD )
      wire#w1
      Coil( #STAT_AvanceDescarga )
   END_RUNG
   RUNG wire#powerrail
      Contact( #Mx_ET50 )
      wire#w2
      Contact( #S3_Arrival )
      Contact( #S3_Rotative )
      Contact( #MA_PickUpOK_S3 )
   END_RUNG wire#w1
   RUNG wire#powerrail
      Contact( #Mx_ET51 )
   END_RUNG wire#w2
   RUNG wire#powerrail
      Contact( #Mx_ET251 )
      I_Contact( #CNT_PrepararS1.QD )
   END_RUNG wire#w1
   RUNG wire#powerrail
      Contact( #Mx_ET60 )
      wire#w3
      Contact( #S1_Arrival )
      Contact( #S1_Rotative )
      Contact( #MA_PickUpOK_S1 )
   END_RUNG wire#w1
   RUNG wire#powerrail
      Contact( #Mx_ET61 )
   END_RUNG wire#w3
   // the same network as SCL:
   #STAT_AvanceDescarga := (#Mx_ET250 AND NOT #CNT_PrepararS3.QD) OR ((#Mx_ET50 OR #Mx_ET51) AND #S3_Arrival AND #S3_Rotative AND #MA_PickUpOK_S3) OR (#Mx_ET251 AND NOT #CNT_PrepararS1.QD) OR ((#Mx_ET60 OR #Mx_ET61) AND #S1_Arrival AND #S1_Rotative AND #MA_PickUpOK_S1);
END_REGION

REGION Network 100: VARIABLES INTERNAS - AVANCE DE PASARELA
   RUNG wire#powerrail
      Contact( #Mx_ET40 )
      wire#w1
      I_Contact( #CNT_PresenciaPasarela.QD )
      wire#w2
      Contact( #Activado_Pasarela )
      Contact( #Pos_TROK )
      Contact( #Pos_TPOK )
      Contact( #EstadoZona.Marcha_CBx )
      I_Contact( #EstadoVI.Error_Mx )
      I_Contact( #Error_Tx )
      Coil( #STAT_AvancePasarela )
   END_RUNG
   RUNG wire#powerrail
      Contact( #Mx_ET41 )
   END_RUNG wire#w1
   RUNG wire#w1
      Contact( #PTF_MAnt_MSig )
   END_RUNG wire#w2
   RUNG wire#powerrail
      Contact( #Mx_ET90 )
      wire#w3
      I_Contact( #CNT_PresenciaPasarela.QD )
   END_RUNG wire#w2
   RUNG wire#powerrail
      Contact( #Mx_ET91 )
   END_RUNG wire#w3
   RUNG wire#w3
      Contact( #PTF_MAnt_MSig )
   END_RUNG wire#w2
   // the same network as SCL:
   #STAT_AvancePasarela := (((#Mx_ET40 OR #Mx_ET41) AND (NOT #CNT_PresenciaPasarela.QD OR #PTF_MAnt_MSig)) OR ((#Mx_ET90 OR #Mx_ET91) AND (NOT #CNT_PresenciaPasarela.QD OR #PTF_MAnt_MSig))) AND #Activado_Pasarela AND #Pos_TROK AND #Pos_TPOK AND #EstadoZona.Marcha_CBx AND NOT #EstadoVI.Error_Mx AND NOT #Error_Tx;
END_REGION

REGION Network 101: VARIABLES INTERNAS - VELOCIDAD BIT 00 >> RODILLOS 00-LenSima 01-Repos 10-Len 11-Rap
   RUNG wire#powerrail
      Contact( #Mx_ET15 )
      wire#w1
      I_Contact( #MemoriaPos_04 )
      I_Contact( #pHsMx_4 )
      wire#w2
      Coil( #STAT_Velocidad_TxBO )
   END_RUNG
   RUNG wire#powerrail
      Contact( #Mx_ET09 )
   END_RUNG wire#w1
   RUNG wire#w1
      Contact( #MemoriaPos_04 )
      I_Contact( #MemoriaPos_03 )
      I_Contact( #pHsMx_3 )
   END_RUNG wire#w2
   RUNG wire#w1
      Contact( #MemoriaPos_04 )
      Contact( #MemoriaPos_03 )
      I_Contact( #MemoriaPos_02 )
      I_Contact( #pHsMx_2 )
   END_RUNG wire#w2
   RUNG wire#w1
      Contact( #MemoriaPos_04 )
      Contact( #MemoriaPos_03 )
      Contact( #MemoriaPos_02 )
      I_Contact( #MemoriaPos_01 )
      I_Contact( #pHsMx_1 )
   END_RUNG wire#w2
   RUNG wire#powerrail
      Contact( #Mx_ET50 )
      wire#w3
      Contact( "ON" )
   END_RUNG wire#w2
   RUNG wire#powerrail
      Contact( #Mx_ET51 )
   END_RUNG wire#w3
   RUNG wire#powerrail
      Contact( #Mx_ET250 )
      I_Contact( #pHsMx_4 )
   END_RUNG wire#w3
   RUNG wire#powerrail
      Contact( #Mx_ET60 )
      wire#w4
      Contact( "ON" )
   END_RUNG wire#w2
   RUNG wire#powerrail
      Contact( #Mx_ET61 )
   END_RUNG wire#w4
   RUNG wire#powerrail
      Contact( #Mx_ET260 )
      I_Contact( #pHsMx_1 )
   END_RUNG wire#w4
   // the same network as SCL:
   #STAT_Velocidad_TxBO := ((#Mx_ET15 OR #Mx_ET09) AND ((NOT #MemoriaPos_04 AND NOT #pHsMx_4) OR (#MemoriaPos_04 AND NOT #MemoriaPos_03 AND NOT #pHsMx_3) OR (#MemoriaPos_04 AND #MemoriaPos_03 AND NOT #MemoriaPos_02 AND NOT #pHsMx_2) OR (#MemoriaPos_04 AND #MemoriaPos_03 AND #MemoriaPos_02 AND NOT #MemoriaPos_01 AND NOT #pHsMx_1))) OR ((#Mx_ET50 OR #Mx_ET51 OR (#Mx_ET250 AND NOT #pHsMx_4)) AND "ON") OR ((#Mx_ET60 OR #Mx_ET61 OR (#Mx_ET260 AND NOT #pHsMx_1)) AND "ON");
END_REGION

REGION Network 102: VARIABLES INTERNAS - VELOCIDAD BIT 01 >> RODILLOS 00-LenSima 01-Repos 10-Len 11-Rap
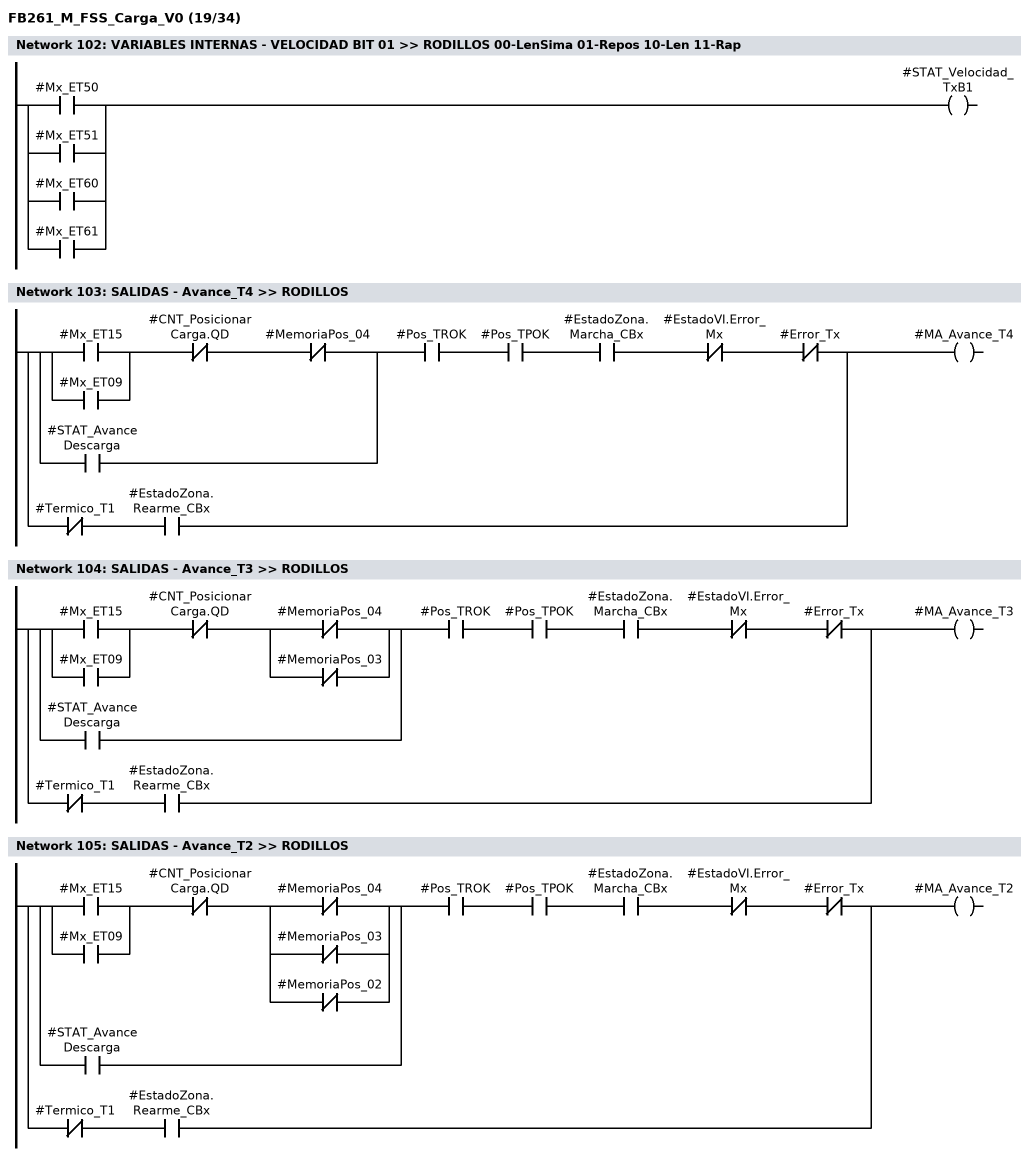
   RUNG wire#powerrail
      Contact( #Mx_ET50 )
      wire#w1
      Coil( #STAT_Velocidad_TxB1 )
   END_RUNG
   RUNG wire#powerrail
      Contact( #Mx_ET51 )
   END_RUNG wire#w1
   RUNG wire#powerrail
      Contact( #Mx_ET60 )
   END_RUNG wire#w1
   RUNG wire#powerrail
      Contact( #Mx_ET61 )
   END_RUNG wire#w1
   // the same network as SCL:
   #STAT_Velocidad_TxB1 := #Mx_ET50 OR #Mx_ET51 OR #Mx_ET60 OR #Mx_ET61;
END_REGION

REGION Network 103: SALIDAS - Avance_T4 >> RODILLOS
   RUNG wire#powerrail
      Contact( #Mx_ET15 )
      wire#w1
      I_Contact( #CNT_PosicionarCarga.QD )
      I_Contact( #MemoriaPos_04 )
      wire#w2
      Contact( #Pos_TROK )
      Contact( #Pos_TPOK )
      Contact( #EstadoZona.Marcha_CBx )
      I_Contact( #EstadoVI.Error_Mx )
      I_Contact( #Error_Tx )
      wire#w3
      Coil( #MA_Avance_T4 )
   END_RUNG
   RUNG wire#powerrail
      Contact( #Mx_ET09 )
   END_RUNG wire#w1
   RUNG wire#powerrail
      Contact( #STAT_AvanceDescarga )
   END_RUNG wire#w2
   RUNG wire#powerrail
      I_Contact( #Termico_T1 )
      Contact( #EstadoZona.Rearme_CBx )
   END_RUNG wire#w3
   // the same network as SCL:
   #MA_Avance_T4 := ((((#Mx_ET15 OR #Mx_ET09) AND NOT #CNT_PosicionarCarga.QD AND NOT #MemoriaPos_04) OR #STAT_AvanceDescarga) AND #Pos_TROK AND #Pos_TPOK AND #EstadoZona.Marcha_CBx AND NOT #EstadoVI.Error_Mx AND NOT #Error_Tx) OR (NOT #Termico_T1 AND #EstadoZona.Rearme_CBx);
END_REGION

REGION Network 104: SALIDAS - Avance_T3 >> RODILLOS
   RUNG wire#powerrail
      Contact( #Mx_ET15 )
      wire#w1
      I_Contact( #CNT_PosicionarCarga.QD )
      wire#w2
      I_Contact( #MemoriaPos_04 )
      wire#w3
      Contact( #Pos_TROK )
      Contact( #Pos_TPOK )
      Contact( #EstadoZona.Marcha_CBx )
      I_Contact( #EstadoVI.Error_Mx )
      I_Contact( #Error_Tx )
      wire#w4
      Coil( #MA_Avance_T3 )
   END_RUNG
   RUNG wire#powerrail
      Contact( #Mx_ET09 )
   END_RUNG wire#w1
   RUNG wire#w2
      I_Contact( #MemoriaPos_03 )
   END_RUNG wire#w3
   RUNG wire#powerrail
      Contact( #STAT_AvanceDescarga )
   END_RUNG wire#w3
   RUNG wire#powerrail
      I_Contact( #Termico_T1 )
      Contact( #EstadoZona.Rearme_CBx )
   END_RUNG wire#w4
   // the same network as SCL:
   #MA_Avance_T3 := ((((#Mx_ET15 OR #Mx_ET09) AND NOT #CNT_PosicionarCarga.QD AND (NOT #MemoriaPos_04 OR NOT #MemoriaPos_03)) OR #STAT_AvanceDescarga) AND #Pos_TROK AND #Pos_TPOK AND #EstadoZona.Marcha_CBx AND NOT #EstadoVI.Error_Mx AND NOT #Error_Tx) OR (NOT #Termico_T1 AND #EstadoZona.Rearme_CBx);
END_REGION

REGION Network 105: SALIDAS - Avance_T2 >> RODILLOS
   RUNG wire#powerrail
      Contact( #Mx_ET15 )
      wire#w1
      I_Contact( #CNT_PosicionarCarga.QD )
      wire#w2
      I_Contact( #MemoriaPos_04 )
      wire#w3
      Contact( #Pos_TROK )
      Contact( #Pos_TPOK )
      Contact( #EstadoZona.Marcha_CBx )
      I_Contact( #EstadoVI.Error_Mx )
      I_Contact( #Error_Tx )
      wire#w4
      Coil( #MA_Avance_T2 )
   END_RUNG
   RUNG wire#powerrail
      Contact( #Mx_ET09 )
   END_RUNG wire#w1
   RUNG wire#w2
      I_Contact( #MemoriaPos_03 )
   END_RUNG wire#w3
   RUNG wire#w2
      I_Contact( #MemoriaPos_02 )
   END_RUNG wire#w3
   RUNG wire#powerrail
      Contact( #STAT_AvanceDescarga )
   END_RUNG wire#w3
   RUNG wire#powerrail
      I_Contact( #Termico_T1 )
      Contact( #EstadoZona.Rearme_CBx )
   END_RUNG wire#w4
   // the same network as SCL:
   #MA_Avance_T2 := ((((#Mx_ET15 OR #Mx_ET09) AND NOT #CNT_PosicionarCarga.QD AND (NOT #MemoriaPos_04 OR NOT #MemoriaPos_03 OR NOT #MemoriaPos_02)) OR #STAT_AvanceDescarga) AND #Pos_TROK AND #Pos_TPOK AND #EstadoZona.Marcha_CBx AND NOT #EstadoVI.Error_Mx AND NOT #Error_Tx) OR (NOT #Termico_T1 AND #EstadoZona.Rearme_CBx);
END_REGION

REGION Network 106: SALIDAS - Avance_T1 >> RODILLOS
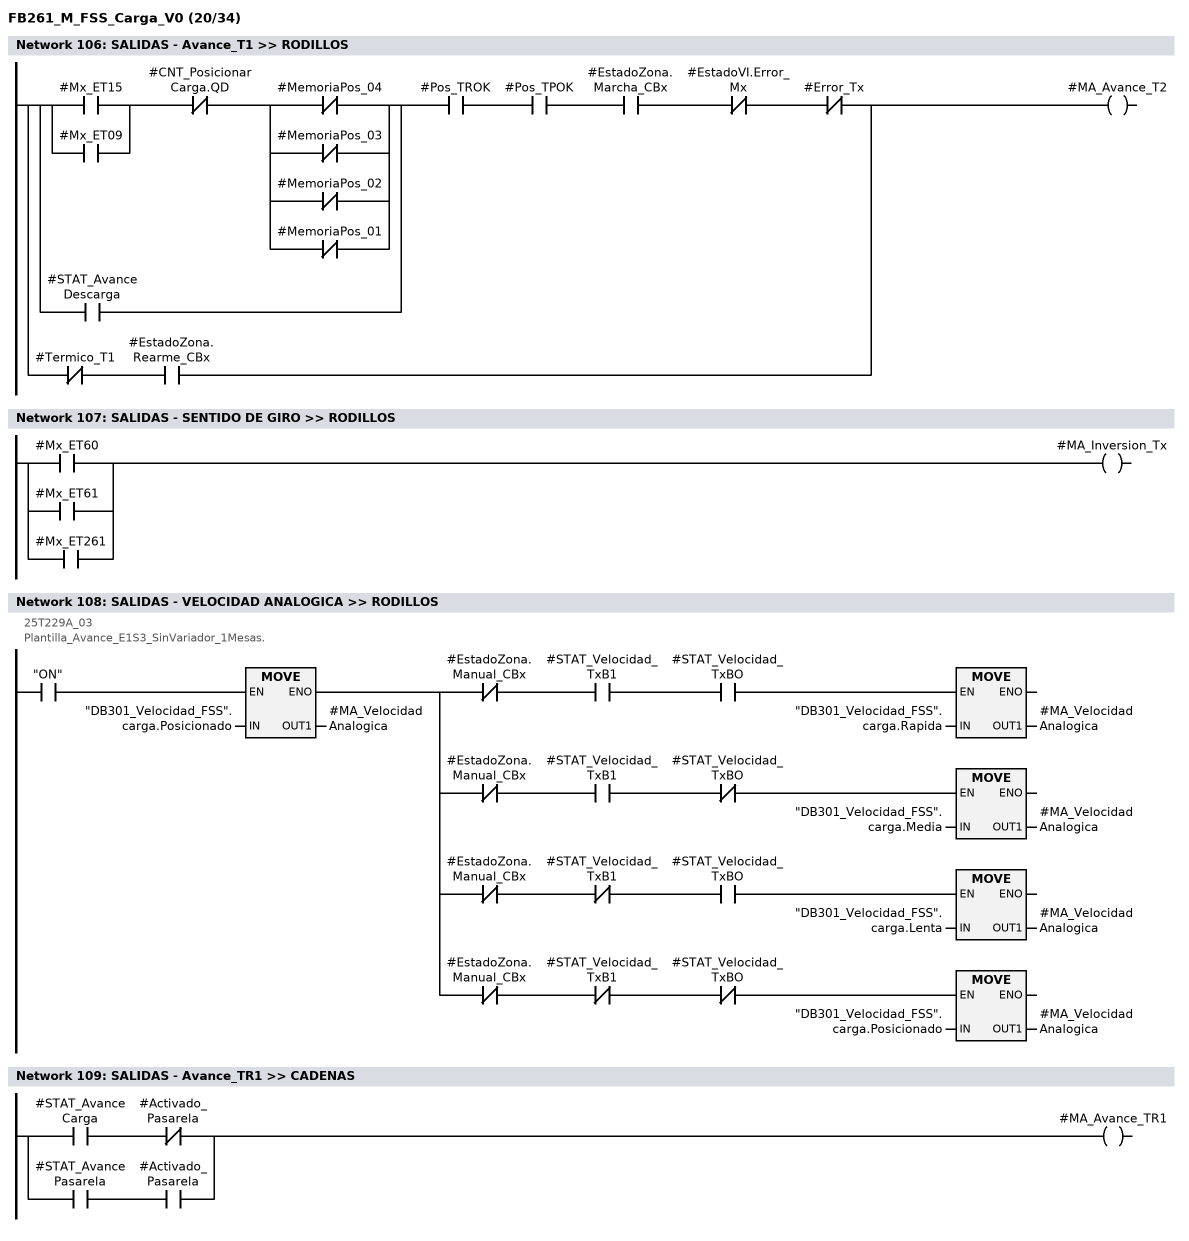
   RUNG wire#powerrail
      Contact( #Mx_ET15 )
      wire#w1
      I_Contact( #CNT_PosicionarCarga.QD )
      wire#w2
      I_Contact( #MemoriaPos_04 )
      wire#w3
      Contact( #Pos_TROK )
      Contact( #Pos_TPOK )
      Contact( #EstadoZona.Marcha_CBx )
      I_Contact( #EstadoVI.Error_Mx )
      I_Contact( #Error_Tx )
      wire#w4
      Coil( #MA_Avance_T2 )
   END_RUNG
   RUNG wire#powerrail
      Contact( #Mx_ET09 )
   END_RUNG wire#w1
   RUNG wire#w2
      I_Contact( #MemoriaPos_03 )
   END_RUNG wire#w3
   RUNG wire#w2
      I_Contact( #MemoriaPos_02 )
   END_RUNG wire#w3
   RUNG wire#w2
      I_Contact( #MemoriaPos_01 )
   END_RUNG wire#w3
   RUNG wire#powerrail
      Contact( #STAT_AvanceDescarga )
   END_RUNG wire#w3
   RUNG wire#powerrail
      I_Contact( #Termico_T1 )
      Contact( #EstadoZona.Rearme_CBx )
   END_RUNG wire#w4
   // the same network as SCL:
   #MA_Avance_T2 := ((((#Mx_ET15 OR #Mx_ET09) AND NOT #CNT_PosicionarCarga.QD AND (NOT #MemoriaPos_04 OR NOT #MemoriaPos_03 OR NOT #MemoriaPos_02 OR NOT #MemoriaPos_01)) OR #STAT_AvanceDescarga) AND #Pos_TROK AND #Pos_TPOK AND #EstadoZona.Marcha_CBx AND NOT #EstadoVI.Error_Mx AND NOT #Error_Tx) OR (NOT #Termico_T1 AND #EstadoZona.Rearme_CBx);
END_REGION

REGION Network 107: SALIDAS - SENTIDO DE GIRO >> RODILLOS
   RUNG wire#powerrail
      Contact( #Mx_ET60 )
      wire#w1
      Coil( #MA_Inversion_Tx )
   END_RUNG
   RUNG wire#powerrail
      Contact( #Mx_ET61 )
   END_RUNG wire#w1
   RUNG wire#powerrail
      Contact( #Mx_ET261 )
   END_RUNG wire#w1
   // the same network as SCL:
   #MA_Inversion_Tx := #Mx_ET60 OR #Mx_ET61 OR #Mx_ET261;
END_REGION

